D20512 CHANNEL  ; RK_13 U4_U #1移载Y轴轴正软限位
D20513 CHANNEL  ; RK_13 U4_U #1移载Y轴轴为PCU保留
D20514 CHANNEL  ; RK_13 U4_U #1移载Y轴轴为PCU保留
D20515 CHANNEL  ; RK_13 U4_U #1移载Y轴轴初始脉冲定义
D20600 CHANNEL  ; U6- 操作数据区域定义
D20601 CHANNEL  ; U6- 操作数据区域开始字
D20602 CHANNEL  ; U6- 轴参数定义
D20603 CHANNEL  ; U6- 未被使用
D20604 CHANNEL  ; RK_13 U6_X #2移载Y轴轴输入输出设定
D20605 CHANNEL  ; RK_13 U6_X #2移载Y轴轴操作模式选择
D20606 CHANNEL  ; RK_13 U6_X #2移载Y轴轴最高速度
D20607 CHANNEL  ; RK_13 U6_X #2移载Y轴轴最高速度
D20608 CHANNEL  ; RK_13 U6_X #2移载Y轴轴初始速度
D20609 CHANNEL  ; RK_13 U6_X #2移载Y轴轴初始速度
D20610 CHANNEL  ; RK_13 U6_X #2移载Y轴轴原点搜索高速
D20611 CHANNEL  ; RK_13 U6_X #2移载Y轴轴原点搜索高速
D20612 CHANNEL  ; RK_13 U6_X #2移载Y轴轴原点搜索接近速度
D20613 CHANNEL  ; RK_13 U6_X #2移载Y轴轴原点搜索接近速度
D20614 CHANNEL  ; RK_13 U6_X #2移载Y轴轴原点补偿值
D20615 CHANNEL  ; RK_13 U6_X #2移载Y轴轴原点补偿值
D20616 CHANNEL  ; RK_13 U6_X #2移载Y轴轴间隙补偿
D20617 CHANNEL  ; RK_13 U6_X #2移载Y轴轴间隙补偿速度
D20618 CHANNEL  ; RK_13 U6_X #2移载Y轴轴间隙补偿速度
D20619 CHANNEL  ; RK_13 U6_X #2移载Y轴轴加减速曲线
D20620 CHANNEL  ; RK_13 U6_X #2移载Y轴轴原点搜索加速时间
D20621 CHANNEL  ; RK_13 U6_X #2移载Y轴轴原点搜索加速时间
D20622 CHANNEL  ; RK_13 U6_X #2移载Y轴轴原点搜索减速时间
D20623 CHANNEL  ; RK_13 U6_X #2移载Y轴轴原点搜索减速时间
D20624 CHANNEL  ; RK_13 U6_X #2移载Y轴轴定位监测时间
D20625 CHANNEL  ; RK_13 U6_X #2移载Y轴轴负软限位
D20626 CHANNEL  ; RK_13 U6_X #2移载Y轴轴负软限位
D20627 CHANNEL  ; RK_13 U6_X #2移载Y轴轴正软限位
D20628 CHANNEL  ; RK_13 U6_X #2移载Y轴轴正软限位
D20629 CHANNEL  ; RK_13 U6_X #2移载Y轴轴为PCU保留
D20630 CHANNEL  ; RK_13 U6_X #2移载Y轴轴为PCU保留
D20631 CHANNEL  ; RK_13 U6_X #2移载Y轴轴初始脉冲定义
D20632 CHANNEL  ; RK_16 U6_Y 激光焊接X轴轴输入输出设定
D20633 CHANNEL  ; RK_16 U6_Y 激光焊接X轴轴操作模式选择
D20634 CHANNEL  ; RK_16 U6_Y 激光焊接X轴轴最高速度
D20635 CHANNEL  ; RK_16 U6_Y 激光焊接X轴轴最高速度
D20636 CHANNEL  ; RK_16 U6_Y 激光焊接X轴轴初始速度
D20637 CHANNEL  ; RK_16 U6_Y 激光焊接X轴轴初始速度
D20638 CHANNEL  ; RK_16 U6_Y 激光焊接X轴轴原点搜索高速
D20639 CHANNEL  ; RK_16 U6_Y 激光焊接X轴轴原点搜索高速
D20640 CHANNEL  ; RK_16 U6_Y 激光焊接X轴轴原点搜索接近速度
D20641 CHANNEL  ; RK_16 U6_Y 激光焊接X轴轴原点搜索接近速度
D20642 CHANNEL  ; RK_16 U6_Y 激光焊接X轴轴原点补偿值
D20643 CHANNEL  ; RK_16 U6_Y 激光焊接X轴轴原点补偿值
D20644 CHANNEL  ; RK_16 U6_Y 激光焊接X轴轴间隙补偿
D20645 CHANNEL  ; RK_16 U6_Y 激光焊接X轴轴间隙补偿速度
D20646 CHANNEL  ; RK_16 U6_Y 激光焊接X轴轴间隙补偿速度
D20647 CHANNEL  ; RK_16 U6_Y 激光焊接X轴轴加减速曲线
D20648 CHANNEL  ; RK_16 U6_Y 激光焊接X轴轴原点搜索加速时间
D20649 CHANNEL  ; RK_16 U6_Y 激光焊接X轴轴原点搜索加速时间
D20650 CHANNEL  ; RK_16 U6_Y 激光焊接X轴轴原点搜索减速时间
D20651 CHANNEL  ; RK_16 U6_Y 激光焊接X轴轴原点搜索减速时间
D20652 CHANNEL  ; RK_16 U6_Y 激光焊接X轴轴定位监测时间
D20653 CHANNEL  ; RK_16 U6_Y 激光焊接X轴轴负软限位
D20654 CHANNEL  ; RK_16 U6_Y 激光焊接X轴轴负软限位
D20655 CHANNEL  ; RK_16 U6_Y 激光焊接X轴轴正软限位
D20656 CHANNEL  ; RK_16 U6_Y 激光焊接X轴轴正软限位
D20657 CHANNEL  ; RK_16 U6_Y 激光焊接X轴轴为PCU保留
D20658 CHANNEL  ; RK_16 U6_Y 激光焊接X轴轴为PCU保留
D20659 CHANNEL  ; RK_16 U6_Y 激光焊接X轴轴初始脉冲定义
D20660 CHANNEL  ; RK_16 U6_Z 激光焊接Z轴轴输入输出设定
D20661 CHANNEL  ; RK_16 U6_Z 激光焊接Z轴轴操作模式选择
D20662 CHANNEL  ; RK_16 U6_Z 激光焊接Z轴轴最高速度
D20663 CHANNEL  ; RK_16 U6_Z 激光焊接Z轴轴最高速度
D20664 CHANNEL  ; RK_16 U6_Z 激光焊接Z轴轴初始速度
D20665 CHANNEL  ; RK_16 U6_Z 激光焊接Z轴轴初始速度
D20666 CHANNEL  ; RK_16 U6_Z 激光焊接Z轴轴原点搜索高速
D20667 CHANNEL  ; RK_16 U6_Z 激光焊接Z轴轴原点搜索高速
D20668 CHANNEL  ; RK_16 U6_Z 激光焊接Z轴轴原点搜索接近速度
D20669 CHANNEL  ; RK_16 U6_Z 激光焊接Z轴轴原点搜索接近速度
D20670 CHANNEL  ; RK_16 U6_Z 激光焊接Z轴轴原点补偿值
D20671 CHANNEL  ; RK_16 U6_Z 激光焊接Z轴轴原点补偿值
D20672 CHANNEL  ; RK_16 U6_Z 激光焊接Z轴轴间隙补偿
D20673 CHANNEL  ; RK_16 U6_Z 激光焊接Z轴轴间隙补偿速度
D20674 CHANNEL  ; RK_16 U6_Z 激光焊接Z轴轴间隙补偿速度
D20675 CHANNEL  ; RK_16 U6_Z 激光焊接Z轴轴加减速曲线
D20676 CHANNEL  ; RK_16 U6_Z 激光焊接Z轴轴原点搜索加速时间
D20677 CHANNEL  ; RK_16 U6_Z 激光焊接Z轴轴原点搜索加速时间
D20678 CHANNEL  ; RK_16 U6_Z 激光焊接Z轴轴原点搜索减速时间
D20679 CHANNEL  ; RK_16 U6_Z 激光焊接Z轴轴原点搜索减速时间
D20680 CHANNEL  ; RK_16 U6_Z 激光焊接Z轴轴定位监测时间
D20681 CHANNEL  ; RK_16 U6_Z 激光焊接Z轴轴负软限位
D20682 CHANNEL  ; RK_16 U6_Z 激光焊接Z轴轴负软限位
D20683 CHANNEL  ; RK_16 U6_Z 激光焊接Z轴轴正软限位
D20684 CHANNEL  ; RK_16 U6_Z 激光焊接Z轴轴正软限位
D20685 CHANNEL  ; RK_16 U6_Z 激光焊接Z轴轴为PCU保留
D20686 CHANNEL  ; RK_16 U6_Z 激光焊接Z轴轴为PCU保留
D20687 CHANNEL  ; RK_16 U6_Z 激光焊接Z轴轴初始脉冲定义
D20800 CHANNEL  ; U8- 操作数据区域定义
D20801 CHANNEL  ; U8- 操作数据区域开始字
D20802 CHANNEL  ; U8- 轴参数定义
D20803 CHANNEL  ; U8- 未被使用
D20804 CHANNEL  ; RK_06 U8_X 电池上下料X轴轴输入输出设定
D20805 CHANNEL  ; RK_06 U8_X 电池上下料X轴轴操作模式选择
D20806 CHANNEL  ; RK_06 U8_X 电池上下料X轴轴最高速度
D20807 CHANNEL  ; RK_06 U8_X 电池上下料X轴轴最高速度
D20808 CHANNEL  ; RK_06 U8_X 电池上下料X轴轴初始速度
D20809 CHANNEL  ; RK_06 U8_X 电池上下料X轴轴初始速度
D20810 CHANNEL  ; RK_06 U8_X 电池上下料X轴轴原点搜索高速
D20811 CHANNEL  ; RK_06 U8_X 电池上下料X轴轴原点搜索高速
D20812 CHANNEL  ; RK_06 U8_X 电池上下料X轴轴原点搜索接近速度
D20813 CHANNEL  ; RK_06 U8_X 电池上下料X轴轴原点搜索接近速度
D20814 CHANNEL  ; RK_06 U8_X 电池上下料X轴轴原点补偿值
D20815 CHANNEL  ; RK_06 U8_X 电池上下料X轴轴原点补偿值
D20816 CHANNEL  ; RK_06 U8_X 电池上下料X轴轴间隙补偿
D20817 CHANNEL  ; RK_06 U8_X 电池上下料X轴轴间隙补偿速度
D20818 CHANNEL  ; RK_06 U8_X 电池上下料X轴轴间隙补偿速度
D20819 CHANNEL  ; RK_06 U8_X 电池上下料X轴轴加减速曲线
D20820 CHANNEL  ; RK_06 U8_X 电池上下料X轴轴原点搜索加速时间
D20821 CHANNEL  ; RK_06 U8_X 电池上下料X轴轴原点搜索加速时间
D20822 CHANNEL  ; RK_06 U8_X 电池上下料X轴轴原点搜索减速时间
D20823 CHANNEL  ; RK_06 U8_X 电池上下料X轴轴原点搜索减速时间
D20824 CHANNEL  ; RK_06 U8_X 电池上下料X轴轴定位监测时间
D20825 CHANNEL  ; RK_06 U8_X 电池上下料X轴轴负软限位
D20826 CHANNEL  ; RK_06 U8_X 电池上下料X轴轴负软限位
D20827 CHANNEL  ; RK_06 U8_X 电池上下料X轴轴正软限位
D20828 CHANNEL  ; RK_06 U8_X 电池上下料X轴轴正软限位
D20829 CHANNEL  ; RK_06 U8_X 电池上下料X轴轴为PCU保留
D20830 CHANNEL  ; RK_06 U8_X 电池上下料X轴轴为PCU保留
D20831 CHANNEL  ; RK_06 U8_X 电池上下料X轴轴初始脉冲定义
D20832 CHANNEL  ; RK_07 U8_Y 铝壳进料X轴轴输入输出设定
D20833 CHANNEL  ; RK_07 U8_Y 铝壳进料X轴轴操作模式选择
D20834 CHANNEL  ; RK_07 U8_Y 铝壳进料X轴轴最高速度
D20835 CHANNEL  ; RK_07 U8_Y 铝壳进料X轴轴最高速度
D20836 CHANNEL  ; RK_07 U8_Y 铝壳进料X轴轴初始速度
D20837 CHANNEL  ; RK_07 U8_Y 铝壳进料X轴轴初始速度
D20838 CHANNEL  ; RK_07 U8_Y 铝壳进料X轴轴原点搜索高速
D20839 CHANNEL  ; RK_07 U8_Y 铝壳进料X轴轴原点搜索高速
D20840 CHANNEL  ; RK_07 U8_Y 铝壳进料X轴轴原点搜索接近速度
D20841 CHANNEL  ; RK_07 U8_Y 铝壳进料X轴轴原点搜索接近速度
D20842 CHANNEL  ; RK_07 U8_Y 铝壳进料X轴轴原点补偿值
D20843 CHANNEL  ; RK_07 U8_Y 铝壳进料X轴轴原点补偿值
D20844 CHANNEL  ; RK_07 U8_Y 铝壳进料X轴轴间隙补偿
D20845 CHANNEL  ; RK_07 U8_Y 铝壳进料X轴轴间隙补偿速度
D20846 CHANNEL  ; RK_07 U8_Y 铝壳进料X轴轴间隙补偿速度
D20847 CHANNEL  ; RK_07 U8_Y 铝壳进料X轴轴加减速曲线
D20848 CHANNEL  ; RK_07 U8_Y 铝壳进料X轴轴原点搜索加速时间
D20849 CHANNEL  ; RK_07 U8_Y 铝壳进料X轴轴原点搜索加速时间
D20850 CHANNEL  ; RK_07 U8_Y 铝壳进料X轴轴原点搜索减速时间
D20851 CHANNEL  ; RK_07 U8_Y 铝壳进料X轴轴原点搜索减速时间
D20852 CHANNEL  ; RK_07 U8_Y 铝壳进料X轴轴定位监测时间
D20853 CHANNEL  ; RK_07 U8_Y 铝壳进料X轴轴负软限位
D20854 CHANNEL  ; RK_07 U8_Y 铝壳进料X轴轴负软限位
D20855 CHANNEL  ; RK_07 U8_Y 铝壳进料X轴轴正软限位
D20856 CHANNEL  ; RK_07 U8_Y 铝壳进料X轴轴正软限位
D20857 CHANNEL  ; RK_07 U8_Y 铝壳进料X轴轴为PCU保留
D20858 CHANNEL  ; RK_07 U8_Y 铝壳进料X轴轴为PCU保留
D20859 CHANNEL  ; RK_07 U8_Y 铝壳进料X轴轴初始脉冲定义
D20860 CHANNEL  ; RK_07 U8_Z 铝壳上料移载Y轴轴输入输出设定
D20861 CHANNEL  ; RK_07 U8_Z 铝壳上料移载Y轴轴操作模式选择
D20862 CHANNEL  ; RK_07 U8_Z 铝壳上料移载Y轴轴最高速度
D20863 CHANNEL  ; RK_07 U8_Z 铝壳上料移载Y轴轴最高速度
D20864 CHANNEL  ; RK_07 U8_Z 铝壳上料移载Y轴轴初始速度
D20865 CHANNEL  ; RK_07 U8_Z 铝壳上料移载Y轴轴初始速度
D20866 CHANNEL  ; RK_07 U8_Z 铝壳上料移载Y轴轴原点搜索高速
D20867 CHANNEL  ; RK_07 U8_Z 铝壳上料移载Y轴轴原点搜索高速
D20868 CHANNEL  ; RK_07 U8_Z 铝壳上料移载Y轴轴原点搜索接近速度
D20869 CHANNEL  ; RK_07 U8_Z 铝壳上料移载Y轴轴原点搜索接近速度
D20870 CHANNEL  ; RK_07 U8_Z 铝壳上料移载Y轴轴原点补偿值
D20871 CHANNEL  ; RK_07 U8_Z 铝壳上料移载Y轴轴原点补偿值
D20872 CHANNEL  ; RK_07 U8_Z 铝壳上料移载Y轴轴间隙补偿
D20873 CHANNEL  ; RK_07 U8_Z 铝壳上料移载Y轴轴间隙补偿速度
D20874 CHANNEL  ; RK_07 U8_Z 铝壳上料移载Y轴轴间隙补偿速度
D20875 CHANNEL  ; RK_07 U8_Z 铝壳上料移载Y轴轴加减速曲线
D20876 CHANNEL  ; RK_07 U8_Z 铝壳上料移载Y轴轴原点搜索加速时间
D20877 CHANNEL  ; RK_07 U8_Z 铝壳上料移载Y轴轴原点搜索加速时间
D20878 CHANNEL  ; RK_07 U8_Z 铝壳上料移载Y轴轴原点搜索减速时间
D20879 CHANNEL  ; RK_07 U8_Z 铝壳上料移载Y轴轴原点搜索减速时间
D20880 CHANNEL  ; RK_07 U8_Z 铝壳上料移载Y轴轴定位监测时间
D20881 CHANNEL  ; RK_07 U8_Z 铝壳上料移载Y轴轴负软限位
D20882 CHANNEL  ; RK_07 U8_Z 铝壳上料移载Y轴轴负软限位
D20883 CHANNEL  ; RK_07 U8_Z 铝壳上料移载Y轴轴正软限位
D20884 CHANNEL  ; RK_07 U8_Z 铝壳上料移载Y轴轴正软限位
D20885 CHANNEL  ; RK_07 U8_Z 铝壳上料移载Y轴轴为PCU保留
D20886 CHANNEL  ; RK_07 U8_Z 铝壳上料移载Y轴轴为PCU保留
D20887 CHANNEL  ; RK_07 U8_Z 铝壳上料移载Y轴轴初始脉冲定义
D20888 CHANNEL  ; RK_10 U8_U 电池除尘上料X轴轴输入输出设定
D20889 CHANNEL  ; RK_10 U8_U 电池除尘上料X轴轴操作模式选择
D20890 CHANNEL  ; RK_10 U8_U 电池除尘上料X轴轴最高速度
D20891 CHANNEL  ; RK_10 U8_U 电池除尘上料X轴轴最高速度
D20892 CHANNEL  ; RK_10 U8_U 电池除尘上料X轴轴初始速度
D20893 CHANNEL  ; RK_10 U8_U 电池除尘上料X轴轴初始速度
D20894 CHANNEL  ; RK_10 U8_U 电池除尘上料X轴轴原点搜索高速
D20895 CHANNEL  ; RK_10 U8_U 电池除尘上料X轴轴原点搜索高速
D20896 CHANNEL  ; RK_10 U8_U 电池除尘上料X轴轴原点搜索接近速度
D20897 CHANNEL  ; RK_10 U8_U 电池除尘上料X轴轴原点搜索接近速度
D20898 CHANNEL  ; RK_10 U8_U 电池除尘上料X轴轴原点补偿值
D20899 CHANNEL  ; RK_10 U8_U 电池除尘上料X轴轴原点补偿值
D20900 CHANNEL  ; RK_10 U8_U 电池除尘上料X轴轴间隙补偿
D20901 CHANNEL  ; RK_10 U8_U 电池除尘上料X轴轴间隙补偿速度
D20902 CHANNEL  ; RK_10 U8_U 电池除尘上料X轴轴间隙补偿速度
D20903 CHANNEL  ; RK_10 U8_U 电池除尘上料X轴轴加减速曲线
D20904 CHANNEL  ; RK_10 U8_U 电池除尘上料X轴轴原点搜索加速时间
D20905 CHANNEL  ; RK_10 U8_U 电池除尘上料X轴轴原点搜索加速时间
D20906 CHANNEL  ; RK_10 U8_U 电池除尘上料X轴轴原点搜索减速时间
D20907 CHANNEL  ; RK_10 U8_U 电池除尘上料X轴轴原点搜索减速时间
D20908 CHANNEL  ; RK_10 U8_U 电池除尘上料X轴轴定位监测时间
D20909 CHANNEL  ; RK_10 U8_U 电池除尘上料X轴轴负软限位
D20910 CHANNEL  ; RK_10 U8_U 电池除尘上料X轴轴负软限位
D20911 CHANNEL  ; RK_10 U8_U 电池除尘上料X轴轴正软限位
D20912 CHANNEL  ; RK_10 U8_U 电池除尘上料X轴轴正软限位
D20913 CHANNEL  ; RK_10 U8_U 电池除尘上料X轴轴为PCU保留
D20914 CHANNEL  ; RK_10 U8_U 电池除尘上料X轴轴为PCU保留
D20915 CHANNEL  ; RK_10 U8_U 电池除尘上料X轴轴初始脉冲定义
D21 CHANNEL  ; 报警长延时
D2100 CHANNEL  ; Hipot检测仪读测试结果开始字
D2104 CHANNEL  ; Hipot检测仪测试电压
D2105 CHANNEL  ; Hipot检测仪测试电阻（低字）
D2106 CHANNEL  ; Hipot检测仪测试电阻（高字）
D2107 CHANNEL  ; Hipot检测仪测试电流（低字）
D2108 CHANNEL  ; Hipot检测仪测试电流（高字）
D2110 CHANNEL  ; Hipot检测仪读测试结果结束字
D2125 CHANNEL  ; Hipot检测仪测试电阻（Float）
D2127 CHANNEL  ; Hipot检测仪测试电流（Float）
D2130 CHANNEL  ; 倍率1000（Float）
D214 CHANNEL  ; d306
D2140 CHANNEL  ; Hipot检测仪查询结果开始字
D2144 CHANNEL  ; Hipot测试仪查询电压
D2145 CHANNEL  ; Hipot检测仪查询电阻（低字）
D2146 CHANNEL  ; Hipot检测仪查询电阻（高字）
D2147 CHANNEL  ; Hipot检测仪查询电流（低字）
D2148 CHANNEL  ; Hipot检测仪查询电流（高字）
D2149 CHANNEL  ; Hipot检测仪查询结果
D2150 CHANNEL  ; Hipot检测仪查询数据
D2151 CHANNEL  ; Hipot检测仪查询数据
D2152 CHANNEL  ; Hipot检测仪查询数据
D2153 CHANNEL  ; Hipot检测仪查询数据
D2154 CHANNEL  ; Hipot检测仪查询数据
D2159 CHANNEL  ; Hipot检测仪查询结果结束字
D2165 CHANNEL  ; Hipot检测仪查询电阻（Float）
D2167 CHANNEL  ; Hipot检测仪查询电流（Float）
D2170 CHANNEL  ; Hipot检测仪查询结果转换
D2171 CHANNEL  ; Hipot检测仪查询电阻下限高字
D2172 CHANNEL  ; Hipot检测仪查询电阻下限低字
D2173 CHANNEL  ; Hipot检测仪查询电阻上限高字
D2174 CHANNEL  ; Hipot检测仪查询电阻上限低字
D2175 CHANNEL  ; Hipot检测仪查询测试时间
D22 CHANNEL  ; 报警短延时
D2200 CHANNEL  ; RK_15 轮廓检测机构#1移载轮廓测量值上限（Float）
D2202 CHANNEL  ; RK_15 轮廓检测机构#1移载轮廓测量值下限（Float）
D2204 CHANNEL  ; RK_15 轮廓检测机构#1移载轮廓测量值上限设定（Float）
D2206 CHANNEL  ; RK_15 轮廓检测机构#1移载轮廓测量值下限设定（Float）
D2210 CHANNEL  ; RK_15 轮廓检测机构#2移载轮廓测量值上限（Float）
D2212 CHANNEL  ; RK_15 轮廓检测机构#2移载轮廓测量值下限（Float）
D2214 CHANNEL  ; RK_15 轮廓检测机构#2移载轮廓测量值上限设定（Float）
D2216 CHANNEL  ; RK_15 轮廓检测机构#2移载轮廓测量值下限设定（Float）
D23 CHANNEL  ; 伺服到位延时
D2300 CHANNEL  ; RK_15 轮廓检测机构#1移载#1轮廓测量值（Float）
D2302 CHANNEL  ; RK_15 轮廓检测机构#1移载#2轮廓测量值（Float）
D2304 CHANNEL  ; RK_15 轮廓检测机构#1移载#3轮廓测量值（Float）
D2306 CHANNEL  ; RK_15 轮廓检测机构#1移载#4轮廓测量值（Float）
D2307 CHANNEL  ; RK_15 轮廓检测机构#1移载#4轮廓测量值（Float）
D2310 CHANNEL  ; RK_15 轮廓检测机构#2移载#1轮廓测量值（Float）
D2312 CHANNEL  ; RK_15 轮廓检测机构#2移载#2轮廓测量值（Float）
D2314 CHANNEL  ; RK_15 轮廓检测机构#2移载#3轮廓测量值（Float）
D2316 CHANNEL  ; RK_15 轮廓检测机构#2移载#4轮廓测量值（Float）
D2317 CHANNEL  ; RK_15 轮廓检测机构#2移载#4轮廓测量值（Float）
D2320 CHANNEL  ; RK_15 轮廓检测机构#1移载#1轮廓测量值开始字（String）
D2329 CHANNEL  ; RK_15 轮廓检测机构#1移载#1轮廓测量值结束字（String）
D2330 CHANNEL  ; RK_15 轮廓检测机构#1移载#2轮廓测量值开始字（String）
D2339 CHANNEL  ; RK_15 轮廓检测机构#1移载#2轮廓测量值结束字（String）
D2340 CHANNEL  ; RK_15 轮廓检测机构#1移载#3轮廓测量值开始字（String）
D2349 CHANNEL  ; RK_15 轮廓检测机构#1移载#3轮廓测量值结束字（String）
D2350 CHANNEL  ; RK_15 轮廓检测机构#1移载#4轮廓测量值开始字（String）
D2359 CHANNEL  ; RK_15 轮廓检测机构#1移载#4轮廓测量值结束字（String）
D2360 CHANNEL  ; RK_15 轮廓检测机构#2移载#1轮廓测量值开始字（String）
D2369 CHANNEL  ; RK_15 轮廓检测机构#2移载#1轮廓测量值结束字（String）
D2370 CHANNEL  ; RK_15 轮廓检测机构#2移载#2轮廓测量值开始字（String）
D2379 CHANNEL  ; RK_15 轮廓检测机构#2移载#2轮廓测量值结束字（String）
D2380 CHANNEL  ; RK_15 轮廓检测机构#2移载#3轮廓测量值开始字（String）
D2389 CHANNEL  ; RK_15 轮廓检测机构#2移载#3轮廓测量值结束字（String）
D2390 CHANNEL  ; RK_15 轮廓检测机构#2移载#4轮廓测量值开始字（String）
D2399 CHANNEL  ; RK_15 轮廓检测机构#2移载#4轮廓测量值结束字（String）
D24 CHANNEL  ; 伺服启动延时
D25 CHANNEL  ; 轮廓检测机构测量读数据延时设定
D26 CHANNEL  ; 铝壳上下料感应异常提示延时设定
D2603 CHANNEL  ; Hipot检测仪参数组编号
D2604 CHANNEL  ; Hipot检测仪测试电压
D2605 CHANNEL  ; Hipot检测仪测试延时时间
D2606 CHANNEL  ; Hipot检测仪测试时间
D2608 CHANNEL  ; Hipot检测仪电阻下限
D2609 CHANNEL  ; Hipot检测仪电阻上限
D2610 CHANNEL  ; RK_09 Hipot检测机构测试完成放电延时参数设定
D2653 CHANNEL  ; Hipot检测仪参数组编号（HMI）
D2654 CHANNEL  ; Hipot检测仪测试电压（HMI）
D2655 CHANNEL  ; Hipot检测仪测试延时时间（HMI）
D2656 CHANNEL  ; Hipot检测仪测试时间（HMI）
D2658 CHANNEL  ; Hipot检测仪电阻下限（HMI）
D2659 CHANNEL  ; Hipot检测仪电阻上限（HMI）
D2660 CHANNEL  ; RK_09 Hipot检测机构测试完成放电延时设定
D2700 CHANNEL  ; Hipot检测仪参数发送（协议宏）
D2809 CHANNEL  ; Hipot检测仪测试结果
D300 CHANNEL  ; 良品数（DINT）
D302 CHANNEL  ; 不良品数（DINT）
D304 CHANNEL  ; 总计（DINT）
D306 CHANNEL  ; 合格率（Float）
D310 CHANNEL  ; #1出站不良品数（DINT）
D3100 CHANNEL  ; 电芯进料X轴&上料X轴当前总距离
D3102 CHANNEL  ; 电芯进料X轴&上料X轴两原点间距离设定值
D3104 CHANNEL  ; 电芯进料X轴&上料X轴距离计算值
D3106 CHANNEL  ; 电芯进料X轴&上料X轴距离最小安全值
D3108 CHANNEL  ; 电芯进料X轴&上料X轴最小安全距离设定值
D3110 CHANNEL  ; 电芯进料X轴允许去放料位安全设定值（参照电芯上料X轴当前位置）
D3112 CHANNEL  ; 电芯上料X轴允许去取料位安全设定值（参照电芯进料X轴当前位置）
D312 CHANNEL  ; #2出站不良品数（DINT）
D314 CHANNEL  ; 总计（Float）
D316 CHANNEL  ; 良品数（Float）
D3210 CHANNEL  ; 电芯上料X轴允许去取料位安全设定值（参照电芯进料X轴当前位置）
D3300 CHANNEL  ; 电芯除尘吹气延时设定值
D3400 CHANNEL  ; RK_05 入壳压力高报警SV
D350 CHANNEL  ; 电芯进料到入壳工位有电芯统计（BCD）
D351 CHANNEL  ; 电芯进料到入壳工位有电芯统计（BIN）
D360 CHANNEL  ; 铝壳进料到入壳工位有铝壳统计（BCD）
D3600 CHANNEL  ; 铝壳料盘列数设定（X轴）
D3602 CHANNEL  ; 铝壳料盘行数设定（Y轴）
D361 CHANNEL  ; 铝壳进料到入壳工位有铝壳统计（BIN）
D3610 CHANNEL  ; 铝壳料盘列间距设定（X轴）
D3612 CHANNEL  ; 铝壳料盘行间距设定（Y轴）
D3700 CHANNEL  ; 铝壳除尘吹气延时设定值
D3804 CHANNEL  ; #1Hipot检测仪测试电压（Int）
D3805 CHANNEL  ; #1Hipot测试仪测试电阻（Float）
D3806 CHANNEL  ; #1Hipot测试仪测试电阻（Float）
D3807 CHANNEL  ; #1Hipot检测仪测试电流（Float）
D3808 CHANNEL  ; #1Hipot检测仪测试电流（Float）
D3809 CHANNEL  ; #1Hipot检测仪测试结果（Int）
D3854 CHANNEL  ; #2Hipot检测仪测试电压（Int）
D3855 CHANNEL  ; #2Hipot测试仪测试电阻（Float）
D3856 CHANNEL  ; #2Hipot测试仪测试电阻（Float）
D3857 CHANNEL  ; #2Hipot检测仪测试电流（Float）
D3858 CHANNEL  ; #2Hipot检测仪测试电流（Float）
D3859 CHANNEL  ; #2Hipot检测仪测试结果（Int）
D3900 CHANNEL  ; 电池除尘上料X轴&预焊上下料X轴当前总距离
D3902 CHANNEL  ; 电池除尘上料X轴&预焊上下料X轴两原点间距离设定值
D3904 CHANNEL  ; 电池除尘上料X轴&预焊上下料X轴距离计算值
D3906 CHANNEL  ; 电池除尘上料X轴&预焊上下料X轴距离最小安全值
D3908 CHANNEL  ; 电池除尘上料X轴&预焊上下料X轴最小安全距离设定值
D3910 CHANNEL  ; 电池除尘上料X轴允许去电池除尘放料位安全设定值（参照预焊上下料X轴当前位置）
D3912 CHANNEL  ; 预焊上下料X轴允许去电池除尘取料位安全设定值（参照电池除尘上料X轴当前位置）
D4000 CHANNEL  ; 电池除尘吹气延时设定值
D4110 CHANNEL  ; 预焊上下料X轴允许去电池除尘取料位安全设定值（参照电池除尘上料X轴当前位置）
D4400 CHANNEL  ; RK_15 轮廓检测机构程序切换设定
D4410 CHANNEL  ; RK_15 轮廓检测机构程序切换字节数
D4411 CHANNEL  ; RK_15 轮廓检测机构程序切换开始字
D4419 CHANNEL  ; RK_15 轮廓检测机构程序切换结束字
D4420 CHANNEL  ; RK_15 轮廓检测机构轮廓测量字节数
D4421 CHANNEL  ; RK_15 轮廓检测机构轮廓测量结果开始字
D4426 CHANNEL  ; RK_15 轮廓检测机构轮廓测量值开始字
D4439 CHANNEL  ; RK_15 轮廓检测机构轮廓测量结果结束字
D4450 CHANNEL  ; RK_15 轮廓检测机构轮廓测量值开始字（String）
D4460 CHANNEL  ; RK_15 轮廓检测机构轮廓测量值开始字（Float）
D4470 CHANNEL  ; RK_15 轮廓检测机构轮廓测量值开始字（String）
D60 CHANNEL  ; 电芯进料接收条码数据字长度
D64 CHANNEL  ; 设定条码抽取开始位
D65 CHANNEL  ; 条码抽取开始位
D66 CHANNEL  ; 设定条码长度
D68 CHANNEL  ; 电芯进料接收条码字长度
D69 CHANNEL  ; 电芯进料接收条码字长度余数
D70 CHANNEL  ; 设定条码批次号
D71 CHANNEL  ; A设定条码批次号
D72 CHANNEL  ; A设定条码批次号
D73 CHANNEL  ; A设定条码批次号
D74 CHANNEL  ; A设定条码批次号
D75 CHANNEL  ; A设定条码批次号
D76 CHANNEL  ; A设定条码批次号
D77 CHANNEL  ; A设定条码批次号
D78 CHANNEL  ; A设定条码批次号
D79 CHANNEL  ; A设定条码批次号
D80 CHANNEL  ; 电芯进料接收条码长度
D900 CHANNEL  ; RK_05 #1入壳压力PV
D902 CHANNEL  ; RK_05 #1入壳压力补偿值
D910 CHANNEL  ; RK_05 #2入壳压力PV
D912 CHANNEL  ; RK_05 #2入壳压力补偿值
D998 CHANNEL  ; 数据零（Float）
D999 CHANNEL  ; 数据零（Float）
E0_4000 CHANNEL  ; RK_07 U8_Y 铝壳进料X轴取料基准位
E0_4020 CHANNEL  ; RK_07 U8_Z 铝壳上料移载Y轴铝壳取料基准位
E1_0 CHANNEL  ; NC433_0 数据传送写字数
E1_1 CHANNEL  ; NC433_0 数据传送写源区域
E1_10 CHANNEL  ; RK_01 U0_X 电芯来料Y轴轴直接操作速度
E1_100 CHANNEL  ; NC433_2 数据传送写字数
E1_1000 CHANNEL  ; RK_01 U0_X 电芯来料Y轴轴自动速度
E1_1001 CHANNEL  ; RK_01 U0_X 电芯来料Y轴轴自动速度
E1_1002 CHANNEL  ; RK_01 U0_X 电芯来料Y轴轴 Jog 高速
E1_1003 CHANNEL  ; RK_01 U0_X 电芯来料Y轴轴 Jog 高速
E1_1004 CHANNEL  ; RK_01 U0_X 电芯来料Y轴轴 Jog 低速
E1_1005 CHANNEL  ; RK_01 U0_X 电芯来料Y轴轴 Jog 低速
E1_1006 CHANNEL  ; RK_01 U0_X 电芯来料Y轴轴加减速时间
E1_1007 CHANNEL  ; RK_01 U0_X 电芯来料Y轴轴加减速时间
E1_1008 CHANNEL  ; RK_01 U0_X 电芯来料Y轴轴正软极限
E1_1009 CHANNEL  ; RK_01 U0_X 电芯来料Y轴轴正软极限
E1_101 CHANNEL  ; NC433_2 数据传送写源区域
E1_1010 CHANNEL  ; RK_01 U0_X 电芯来料Y轴轴负软极限
E1_1011 CHANNEL  ; RK_01 U0_X 电芯来料Y轴轴负软极限
E1_1012 CHANNEL  ; RK_01 U0_X 电芯来料Y轴轴原点偏移
E1_102 CHANNEL  ; NC433_2 数据传送定源字
E1_1020 CHANNEL  ; RK_01 U0_X 电芯来料Y轴待料位
E1_1021 CHANNEL  ; RK_01 U0_X 电芯来料Y轴待料位
E1_1022 CHANNEL  ; RK_01 U0_X 电芯来料Y轴上料位
E1_1023 CHANNEL  ; RK_01 U0_X 电芯来料Y轴上料位
E1_1024 CHANNEL  ; RK_01 U0_X 电芯来料Y轴扫码位
E1_1025 CHANNEL  ; RK_01 U0_X 电芯来料Y轴扫码位
E1_1026 CHANNEL  ; RK_01 U0_X 电芯来料Y轴下料位
E1_1027 CHANNEL  ; RK_01 U0_X 电芯来料Y轴下料位
E1_1028 CHANNEL  ; RK_01 U0_X 电芯来料Y轴轴5#位置
E1_1029 CHANNEL  ; RK_01 U0_X 电芯来料Y轴轴5#位置
E1_103 CHANNEL  ; NC433_2 数据传送定目标地址
E1_1030 CHANNEL  ; RK_01 U0_X 电芯来料Y轴轴6#位置
E1_1031 CHANNEL  ; RK_01 U0_X 电芯来料Y轴轴6#位置
E1_1032 CHANNEL  ; RK_01 U0_X 电芯来料Y轴轴7#位置
E1_1033 CHANNEL  ; RK_01 U0_X 电芯来料Y轴轴7#位置
E1_1034 CHANNEL  ; RK_01 U0_X 电芯来料Y轴轴8#位置
E1_1035 CHANNEL  ; RK_01 U0_X 电芯来料Y轴轴8#位置
E1_1036 CHANNEL  ; RK_01 U0_X 电芯来料Y轴轴9#位置
E1_1037 CHANNEL  ; RK_01 U0_X 电芯来料Y轴轴9#位置
E1_1038 CHANNEL  ; RK_01 U0_X 电芯来料Y轴轴10#位置
E1_1039 CHANNEL  ; RK_01 U0_X 电芯来料Y轴轴10#位置
E1_104 CHANNEL  ; NC433_2 数据传送读字数
E1_105 CHANNEL  ; NC433_2 数据传送读源区域
E1_106 CHANNEL  ; NC433_2 数据传送读目标区域
E1_107 CHANNEL  ; NC433_2 数据传送读目标字
E1_108 CHANNEL  ; RK_05 U2_X #1入壳Y轴轴直接操作位置
E1_109 CHANNEL  ; RK_05 U2_X #1入壳Y轴轴直接操作位置
E1_11 CHANNEL  ; RK_01 U0_X 电芯来料Y轴轴直接操作速度
E1_110 CHANNEL  ; RK_05 U2_X #1入壳Y轴轴直接操作速度
E1_1100 CHANNEL  ; RK_02 U0_Y 电芯进料X轴轴自动速度
E1_11000 CHANNEL  ; #4配方参数（伺服轴）
E1_1101 CHANNEL  ; RK_02 U0_Y 电芯进料X轴轴自动速度
E1_1102 CHANNEL  ; RK_02 U0_Y 电芯进料X轴轴 Jog 高速
E1_1103 CHANNEL  ; RK_02 U0_Y 电芯进料X轴轴 Jog 高速
E1_1104 CHANNEL  ; RK_02 U0_Y 电芯进料X轴轴 Jog 低速
E1_1105 CHANNEL  ; RK_02 U0_Y 电芯进料X轴轴 Jog 低速
E1_1106 CHANNEL  ; RK_02 U0_Y 电芯进料X轴轴加减速时间
E1_1107 CHANNEL  ; RK_02 U0_Y 电芯进料X轴轴加减速时间
E1_1108 CHANNEL  ; RK_02 U0_Y 电芯进料X轴轴正软极限
E1_1109 CHANNEL  ; RK_02 U0_Y 电芯进料X轴轴正软极限
E1_111 CHANNEL  ; RK_05 U2_X #1入壳Y轴轴直接操作速度
E1_1110 CHANNEL  ; RK_02 U0_Y 电芯进料X轴轴负软极限
E1_1111 CHANNEL  ; RK_02 U0_Y 电芯进料X轴轴负软极限
E1_1112 CHANNEL  ; RK_02 U0_Y 电芯进料X轴轴原点偏移
E1_112 CHANNEL  ; RK_05 U2_X #1入壳Y轴轴直接操作加速时间
E1_1120 CHANNEL  ; RK_02 U0_Y 电芯进料X轴待料位
E1_1121 CHANNEL  ; RK_02 U0_Y 电芯进料X轴待料位
E1_1122 CHANNEL  ; RK_02 U0_Y 电芯进料X轴取料位
E1_1123 CHANNEL  ; RK_02 U0_Y 电芯进料X轴取料位
E1_1124 CHANNEL  ; RK_02 U0_Y 电芯进料X轴扫码OK放料位
E1_1125 CHANNEL  ; RK_02 U0_Y 电芯进料X轴扫码OK放料位
E1_1126 CHANNEL  ; RK_02 U0_Y 电芯进料X轴扫码NG放料位
E1_1127 CHANNEL  ; RK_02 U0_Y 电芯进料X轴扫码NG放料位
E1_1128 CHANNEL  ; RK_02 U0_Y 电芯进料X轴轴5#位置
E1_1129 CHANNEL  ; RK_02 U0_Y 电芯进料X轴轴5#位置
E1_113 CHANNEL  ; RK_05 U2_X #1入壳Y轴X轴直接操作加速时间
E1_1130 CHANNEL  ; RK_02 U0_Y 电芯进料X轴轴6#位置
E1_1131 CHANNEL  ; RK_02 U0_Y 电芯进料X轴轴6#位置
E1_1132 CHANNEL  ; RK_02 U0_Y 电芯进料X轴轴7#位置
E1_1133 CHANNEL  ; RK_02 U0_Y 电芯进料X轴轴7#位置
E1_1134 CHANNEL  ; RK_02 U0_Y 电芯进料X轴轴8#位置
E1_1135 CHANNEL  ; RK_02 U0_Y 电芯进料X轴轴8#位置
E1_1136 CHANNEL  ; RK_02 U0_Y 电芯进料X轴轴9#位置
E1_1137 CHANNEL  ; RK_02 U0_Y 电芯进料X轴轴9#位置
E1_1138 CHANNEL  ; RK_02 U0_Y 电芯进料X轴轴10#位置
E1_1139 CHANNEL  ; RK_02 U0_Y 电芯进料X轴轴10#位置
E1_114 CHANNEL  ; RK_05 U2_X #1入壳Y轴轴直接操作减速时间
E1_115 CHANNEL  ; RK_05 U2_X #1入壳Y轴轴直接操作减速时间
E1_116 CHANNEL  ; RK_05 U2_X #1入壳Y轴轴存储器操作序列号
E1_117 CHANNEL  ; RK_05 U2_X #1入壳Y轴轴特殊操作Override
E1_118 CHANNEL  ; RK_05 U2_X #1入壳Y轴轴特殊操作示教地址
E1_119 CHANNEL  ; RK_05 U2_X #1入壳Y轴轴特殊操作预留
E1_12 CHANNEL  ; RK_01 U0_X 电芯来料Y轴轴直接操作加速时间
E1_120 CHANNEL  ; RK_05 U2_Y #2入壳Y轴轴直接操作位置
E1_1200 CHANNEL  ; RK_02 U0_Z 电芯进料Z轴轴自动速度
E1_1201 CHANNEL  ; RK_02 U0_Z 电芯进料Z轴轴自动速度
E1_1202 CHANNEL  ; RK_02 U0_Z 电芯进料Z轴轴 Jog 高速
E1_1203 CHANNEL  ; RK_02 U0_Z 电芯进料Z轴轴 Jog 高速
E1_1204 CHANNEL  ; RK_02 U0_Z 电芯进料Z轴轴 Jog 低速
E1_1205 CHANNEL  ; RK_02 U0_Z 电芯进料Z轴轴 Jog 低速
E1_1206 CHANNEL  ; RK_02 U0_Z 电芯进料Z轴轴加减速时间
E1_1207 CHANNEL  ; RK_02 U0_Z 电芯进料Z轴轴加减速时间
E1_1208 CHANNEL  ; RK_02 U0_Z 电芯进料Z轴轴正软极限
E1_1209 CHANNEL  ; RK_02 U0_Z 电芯进料Z轴轴正软极限
E1_121 CHANNEL  ; RK_05 U2_Y #2入壳Y轴轴直接操作位置
E1_1210 CHANNEL  ; RK_02 U0_Z 电芯进料Z轴轴负软极限
E1_1211 CHANNEL  ; RK_02 U0_Z 电芯进料Z轴轴负软极限
E1_1212 CHANNEL  ; RK_02 U0_Z 电芯进料Z轴轴原点偏移
E1_122 CHANNEL  ; RK_05 U2_Y #2入壳Y轴轴直接操作速度
E1_1220 CHANNEL  ; RK_02 U0_Z 电芯进料Z轴待料位（扫码）
E1_1221 CHANNEL  ; RK_02 U0_Z 电芯进料Z轴待料位（扫码）
E1_1222 CHANNEL  ; RK_02 U0_Z 电芯进料Z轴取料位
E1_1223 CHANNEL  ; RK_02 U0_Z 电芯进料Z轴取料位
E1_1224 CHANNEL  ; RK_02 U0_Z 电芯进料Z轴扫码OK放料位
E1_1225 CHANNEL  ; RK_02 U0_Z 电芯进料Z轴扫码OK放料位
E1_1226 CHANNEL  ; RK_02 U0_Z 电芯进料Z轴扫码NG放料位
E1_1227 CHANNEL  ; RK_02 U0_Z 电芯进料Z轴扫码NG放料位
E1_1228 CHANNEL  ; RK_02 U0_Z 电芯进料Z轴扫码位
E1_1229 CHANNEL  ; RK_02 U0_Z 电芯进料Z轴扫码位
E1_123 CHANNEL  ; RK_05 U2_Y #2入壳Y轴轴直接操作速度
E1_1230 CHANNEL  ; RK_02 U0_Z 电芯进料Z轴轴6#位置
E1_1231 CHANNEL  ; RK_02 U0_Z 电芯进料Z轴轴6#位置
E1_1232 CHANNEL  ; RK_02 U0_Z 电芯进料Z轴轴7#位置
E1_1233 CHANNEL  ; RK_02 U0_Z 电芯进料Z轴轴7#位置
E1_1234 CHANNEL  ; RK_02 U0_Z 电芯进料Z轴轴8#位置
E1_1235 CHANNEL  ; RK_02 U0_Z 电芯进料Z轴轴8#位置
E1_1236 CHANNEL  ; RK_02 U0_Z 电芯进料Z轴轴9#位置
E1_1237 CHANNEL  ; RK_02 U0_Z 电芯进料Z轴轴9#位置
E1_1238 CHANNEL  ; RK_02 U0_Z 电芯进料Z轴轴10#位置
E1_1239 CHANNEL  ; RK_02 U0_Z 电芯进料Z轴轴10#位置
E1_124 CHANNEL  ; RK_05 U2_Y #2入壳Y轴轴直接操作加速时间
E1_125 CHANNEL  ; RK_05 U2_Y #2入壳Y轴轴直接操作加速时间
E1_126 CHANNEL  ; RK_05 U2_Y #2入壳Y轴轴直接操作减速时间
E1_127 CHANNEL  ; RK_05 U2_Y #2入壳Y轴轴直接操作减速时间
E1_128 CHANNEL  ; RK_05 U2_Y #2入壳Y轴轴存储器操作序列号
E1_129 CHANNEL  ; RK_05 U2_Y #2入壳Y轴轴特殊操作Override
E1_13 CHANNEL  ; RK_01 U0_X 电芯来料Y轴X轴直接操作加速时间
E1_130 CHANNEL  ; RK_05 U2_Y #2入壳Y轴轴特殊操作示教地址
E1_1300 CHANNEL  ; RK_03 U0_U 电芯上料X轴轴自动速度
E1_13000 CHANNEL  ; #5配方参数（伺服轴）
E1_1301 CHANNEL  ; RK_03 U0_U 电芯上料X轴轴自动速度
E1_1302 CHANNEL  ; RK_03 U0_U 电芯上料X轴轴 Jog 高速
E1_1303 CHANNEL  ; RK_03 U0_U 电芯上料X轴轴 Jog 高速
E1_1304 CHANNEL  ; RK_03 U0_U 电芯上料X轴轴 Jog 低速
E1_1305 CHANNEL  ; RK_03 U0_U 电芯上料X轴轴 Jog 低速
E1_1306 CHANNEL  ; RK_03 U0_U 电芯上料X轴轴加减速时间
E1_1307 CHANNEL  ; RK_03 U0_U 电芯上料X轴轴加减速时间
E1_1308 CHANNEL  ; RK_03 U0_U 电芯上料X轴轴正软极限
E1_1309 CHANNEL  ; RK_03 U0_U 电芯上料X轴轴正软极限
E1_131 CHANNEL  ; RK_05 U2_Y #2入壳Y轴轴特殊操作预留
E1_1310 CHANNEL  ; RK_03 U0_U 电芯上料X轴轴负软极限
E1_1311 CHANNEL  ; RK_03 U0_U 电芯上料X轴轴负软极限
E1_1312 CHANNEL  ; RK_03 U0_U 电芯上料X轴轴原点偏移
E1_1320 CHANNEL  ; RK_03 U0_U 电芯上料X轴待料位
E1_1321 CHANNEL  ; RK_03 U0_U 电芯上料X轴待料位
E1_1322 CHANNEL  ; RK_03 U0_U 电芯上料X轴取料位
E1_1323 CHANNEL  ; RK_03 U0_U 电芯上料X轴取料位
E1_1324 CHANNEL  ; RK_03 U0_U 电芯上料X轴#1入壳放料位
E1_1325 CHANNEL  ; RK_03 U0_U 电芯上料X轴#1入壳放料位
E1_1326 CHANNEL  ; RK_03 U0_U 电芯上料X轴#2入壳放料位
E1_1327 CHANNEL  ; RK_03 U0_U 电芯上料X轴#2入壳放料位
E1_1328 CHANNEL  ; RK_03 U0_U 电芯上料X轴轴5#位置
E1_1329 CHANNEL  ; RK_03 U0_U 电芯上料X轴轴5#位置
E1_1330 CHANNEL  ; RK_03 U0_U 电芯上料X轴轴6#位置
E1_1331 CHANNEL  ; RK_03 U0_U 电芯上料X轴轴6#位置
E1_1332 CHANNEL  ; RK_03 U0_U 电芯上料X轴轴7#位置
E1_1333 CHANNEL  ; RK_03 U0_U 电芯上料X轴轴7#位置
E1_1334 CHANNEL  ; RK_03 U0_U 电芯上料X轴轴8#位置
E1_1335 CHANNEL  ; RK_03 U0_U 电芯上料X轴轴8#位置
E1_1336 CHANNEL  ; RK_03 U0_U 电芯上料X轴轴9#位置
E1_1337 CHANNEL  ; RK_03 U0_U 电芯上料X轴轴9#位置
E1_1338 CHANNEL  ; RK_03 U0_U 电芯上料X轴轴10#位置
E1_1339 CHANNEL  ; RK_03 U0_U 电芯上料X轴轴10#位置
E1_14 CHANNEL  ; RK_01 U0_X 电芯来料Y轴轴直接操作减速时间
E1_1400 CHANNEL  ; RK_05 U2_X #1入壳Y轴轴自动速度
E1_1401 CHANNEL  ; RK_05 U2_X #1入壳Y轴轴自动速度
E1_1402 CHANNEL  ; RK_05 U2_X #1入壳Y轴轴 Jog 高速
E1_1403 CHANNEL  ; RK_05 U2_X #1入壳Y轴轴 Jog 高速
E1_1404 CHANNEL  ; RK_05 U2_X #1入壳Y轴轴 Jog 低速
E1_1405 CHANNEL  ; RK_05 U2_X #1入壳Y轴轴 Jog 低速
E1_1406 CHANNEL  ; RK_05 U2_X #1入壳Y轴轴加减速时间
E1_1407 CHANNEL  ; RK_05 U2_X #1入壳Y轴轴加减速时间
E1_1408 CHANNEL  ; RK_05 U2_X #1入壳Y轴轴正软极限
E1_1409 CHANNEL  ; RK_05 U2_X #1入壳Y轴轴正软极限
E1_1410 CHANNEL  ; RK_05 U2_X #1入壳Y轴轴负软极限
E1_1411 CHANNEL  ; RK_05 U2_X #1入壳Y轴轴负软极限
E1_1412 CHANNEL  ; RK_05 U2_X #1入壳Y轴轴原点偏移
E1_1420 CHANNEL  ; RK_05 U2_X #1入壳Y轴待料位
E1_1421 CHANNEL  ; RK_05 U2_X #1入壳Y轴待料位
E1_1422 CHANNEL  ; RK_05 U2_X #1入壳Y轴滚轮压紧位
E1_1423 CHANNEL  ; RK_05 U2_X #1入壳Y轴滚轮压紧位
E1_1424 CHANNEL  ; RK_05 U2_X #1入壳Y轴滚轮松开位
E1_1425 CHANNEL  ; RK_05 U2_X #1入壳Y轴滚轮松开位
E1_1426 CHANNEL  ; RK_05 U2_X #1入壳Y轴入壳位
E1_1427 CHANNEL  ; RK_05 U2_X #1入壳Y轴入壳位
E1_1428 CHANNEL  ; RK_05 U2_X #1入壳Y轴电芯定位夹爪松开位
E1_1429 CHANNEL  ; RK_05 U2_X #1入壳Y轴电芯定位夹爪松开位
E1_1430 CHANNEL  ; RK_05 U2_X #1入壳Y轴轴6#位置
E1_1431 CHANNEL  ; RK_05 U2_X #1入壳Y轴轴6#位置
E1_1432 CHANNEL  ; RK_05 U2_X #1入壳Y轴轴7#位置
E1_1433 CHANNEL  ; RK_05 U2_X #1入壳Y轴轴7#位置
E1_1434 CHANNEL  ; RK_05 U2_X #1入壳Y轴轴8#位置
E1_1435 CHANNEL  ; RK_05 U2_X #1入壳Y轴轴8#位置
E1_1436 CHANNEL  ; RK_05 U2_X #1入壳Y轴轴9#位置
E1_1437 CHANNEL  ; RK_05 U2_X #1入壳Y轴轴9#位置
E1_1438 CHANNEL  ; RK_05 U2_X #1入壳Y轴轴10#位置
E1_1439 CHANNEL  ; RK_05 U2_X #1入壳Y轴轴10#位置
E1_15 CHANNEL  ; RK_01 U0_X 电芯来料Y轴轴直接操作减速时间
E1_1500 CHANNEL  ; RK_05 U2_Y #2入壳Y轴轴自动速度
E1_15000 CHANNEL  ; #6配方参数（伺服轴）
E1_1501 CHANNEL  ; RK_05 U2_Y #2入壳Y轴轴自动速度
E1_1502 CHANNEL  ; RK_05 U2_Y #2入壳Y轴轴 Jog 高速
E1_1503 CHANNEL  ; RK_05 U2_Y #2入壳Y轴轴 Jog 高速
E1_1504 CHANNEL  ; RK_05 U2_Y #2入壳Y轴轴 Jog 低速
E1_1505 CHANNEL  ; RK_05 U2_Y #2入壳Y轴轴 Jog 低速
E1_1506 CHANNEL  ; RK_05 U2_Y #2入壳Y轴轴加减速时间
E1_1507 CHANNEL  ; RK_05 U2_Y #2入壳Y轴轴加减速时间
E1_1508 CHANNEL  ; RK_05 U2_Y #2入壳Y轴轴正软极限
E1_1509 CHANNEL  ; RK_05 U2_Y #2入壳Y轴轴正软极限
E1_1510 CHANNEL  ; RK_05 U2_Y #2入壳Y轴轴负软极限
E1_1511 CHANNEL  ; RK_05 U2_Y #2入壳Y轴轴负软极限
E1_1512 CHANNEL  ; RK_05 U2_Y #2入壳Y轴轴原点偏移
E1_1520 CHANNEL  ; RK_05 U2_Y #2入壳Y轴待料位
E1_1521 CHANNEL  ; RK_05 U2_Y #2入壳Y轴待料位
E1_1522 CHANNEL  ; RK_05 U2_Y #2入壳Y轴滚轮压紧位
E1_1523 CHANNEL  ; RK_05 U2_Y #2入壳Y轴滚轮压紧位
E1_1524 CHANNEL  ; RK_05 U2_Y #2入壳Y轴滚轮松开位
E1_1525 CHANNEL  ; RK_05 U2_Y #2入壳Y轴滚轮松开位
E1_1526 CHANNEL  ; RK_05 U2_Y #2入壳Y轴入壳位
E1_1527 CHANNEL  ; RK_05 U2_Y #2入壳Y轴入壳位
E1_1528 CHANNEL  ; RK_05 U2_Y #2入壳Y轴电芯定位夹爪松开位
E1_1529 CHANNEL  ; RK_05 U2_Y #2入壳Y轴电芯定位夹爪松开位
E1_1530 CHANNEL  ; RK_05 U2_Y #2入壳Y轴轴6#位置
E1_1531 CHANNEL  ; RK_05 U2_Y #2入壳Y轴轴6#位置
E1_1532 CHANNEL  ; RK_05 U2_Y #2入壳Y轴轴7#位置
E1_1533 CHANNEL  ; RK_05 U2_Y #2入壳Y轴轴7#位置
E1_1534 CHANNEL  ; RK_05 U2_Y #2入壳Y轴轴8#位置
E1_1535 CHANNEL  ; RK_05 U2_Y #2入壳Y轴轴8#位置
E1_1536 CHANNEL  ; RK_05 U2_Y #2入壳Y轴轴9#位置
E1_1537 CHANNEL  ; RK_05 U2_Y #2入壳Y轴轴9#位置
E1_1538 CHANNEL  ; RK_05 U2_Y #2入壳Y轴轴10#位置
E1_1539 CHANNEL  ; RK_05 U2_Y #2入壳Y轴轴10#位置
E1_156 CHANNEL  ; RK_05 U2_X #1入壳Y轴轴当前位置
E1_157 CHANNEL  ; RK_05 U2_X #1入壳Y轴轴当前位置
E1_158 CHANNEL  ; RK_05 U2_X #1入壳Y轴轴存储器操作正被执行序列号
E1_159 CHANNEL  ; RK_05 U2_X #1入壳Y轴轴存储器操作正被执行序列号
E1_16 CHANNEL  ; RK_01 U0_X 电芯来料Y轴轴存储器操作序列号
E1_160 CHANNEL  ; RK_05 U2_Y #2入壳Y轴轴当前位置
E1_161 CHANNEL  ; RK_05 U2_Y #2入壳Y轴轴当前位置
E1_162 CHANNEL  ; RK_05 U2_Y #2入壳Y轴轴存储器操作正被执行序列号
E1_163 CHANNEL  ; RK_05 U2_Y #2入壳Y轴轴存储器操作正被执行序列号
E1_17 CHANNEL  ; RK_01 U0_X 电芯来料Y轴轴特殊操作Override
E1_17000 CHANNEL  ; #7配方参数（伺服轴）
E1_18 CHANNEL  ; RK_01 U0_X 电芯来料Y轴轴特殊操作示教地址
E1_1800 CHANNEL  ; RK_12 U4_X 预焊上下料X轴轴自动速度
E1_1801 CHANNEL  ; RK_12 U4_X 预焊上下料X轴轴自动速度
E1_1802 CHANNEL  ; RK_12 U4_X 预焊上下料X轴轴 Jog 高速
E1_1803 CHANNEL  ; RK_12 U4_X 预焊上下料X轴轴 Jog 高速
E1_1804 CHANNEL  ; RK_12 U4_X 预焊上下料X轴轴 Jog 低速
E1_1805 CHANNEL  ; RK_12 U4_X 预焊上下料X轴轴 Jog 低速
E1_1806 CHANNEL  ; RK_12 U4_X 预焊上下料X轴轴加减速时间
E1_1807 CHANNEL  ; RK_12 U4_X 预焊上下料X轴轴加减速时间
E1_1808 CHANNEL  ; RK_12 U4_X 预焊上下料X轴轴正软极限
E1_1809 CHANNEL  ; RK_12 U4_X 预焊上下料X轴轴正软极限
E1_1810 CHANNEL  ; RK_12 U4_X 预焊上下料X轴轴负软极限
E1_1811 CHANNEL  ; RK_12 U4_X 预焊上下料X轴轴负软极限
E1_1812 CHANNEL  ; RK_12 U4_X 预焊上下料X轴轴原点偏移
E1_1820 CHANNEL  ; RK_12 U4_X 预焊上下料X轴待料位
E1_1821 CHANNEL  ; RK_12 U4_X 预焊上下料X轴待料位
E1_1822 CHANNEL  ; RK_12 U4_X 预焊上下料X轴除尘取料位
E1_1823 CHANNEL  ; RK_12 U4_X 预焊上下料X轴除尘取料位
E1_1824 CHANNEL  ; RK_12 U4_X 预焊上下料X轴#1移载放料位
E1_1825 CHANNEL  ; RK_12 U4_X 预焊上下料X轴#1移载放料位
E1_1826 CHANNEL  ; RK_12 U4_X 预焊上下料X轴#2移载放料位
E1_1827 CHANNEL  ; RK_12 U4_X 预焊上下料X轴#2移载放料位
E1_1828 CHANNEL  ; RK_12 U4_X 预焊上下料X轴#1移载取料位
E1_1829 CHANNEL  ; RK_12 U4_X 预焊上下料X轴#1移载取料位
E1_1830 CHANNEL  ; RK_12 U4_X 预焊上下料X轴#2移载取料位
E1_1831 CHANNEL  ; RK_12 U4_X 预焊上下料X轴#2移载取料位
E1_1832 CHANNEL  ; RK_12 U4_X 预焊上下料X轴OK放料位
E1_1833 CHANNEL  ; RK_12 U4_X 预焊上下料X轴OK放料位
E1_1834 CHANNEL  ; RK_12 U4_X 预焊上下料X轴#1NG放料位
E1_1835 CHANNEL  ; RK_12 U4_X 预焊上下料X轴#1NG放料位
E1_1836 CHANNEL  ; RK_12 U4_X 预焊上下料X轴#2NG放料位
E1_1837 CHANNEL  ; RK_12 U4_X 预焊上下料X轴#2NG放料位
E1_1838 CHANNEL  ; RK_12 U4_X 预焊上下料X轴轴10#位置
E1_1839 CHANNEL  ; RK_12 U4_X 预焊上下料X轴轴10#位置
E1_19 CHANNEL  ; RK_01 U0_X 电芯来料Y轴轴特殊操作预留
E1_1900 CHANNEL  ; RK_12 U4_Y 预焊上料Z轴轴自动速度
E1_19000 CHANNEL  ; #8配方参数（伺服轴）
E1_1901 CHANNEL  ; RK_12 U4_Y 预焊上料Z轴轴自动速度
E1_1902 CHANNEL  ; RK_12 U4_Y 预焊上料Z轴轴 Jog 高速
E1_1903 CHANNEL  ; RK_12 U4_Y 预焊上料Z轴轴 Jog 高速
E1_1904 CHANNEL  ; RK_12 U4_Y 预焊上料Z轴轴 Jog 低速
E1_1905 CHANNEL  ; RK_12 U4_Y 预焊上料Z轴轴 Jog 低速
E1_1906 CHANNEL  ; RK_12 U4_Y 预焊上料Z轴轴加减速时间
E1_1907 CHANNEL  ; RK_12 U4_Y 预焊上料Z轴轴加减速时间
E1_1908 CHANNEL  ; RK_12 U4_Y 预焊上料Z轴轴正软极限
E1_1909 CHANNEL  ; RK_12 U4_Y 预焊上料Z轴轴正软极限
E1_1910 CHANNEL  ; RK_12 U4_Y 预焊上料Z轴轴负软极限
E1_1911 CHANNEL  ; RK_12 U4_Y 预焊上料Z轴轴负软极限
E1_1912 CHANNEL  ; RK_12 U4_Y 预焊上料Z轴轴原点偏移
E1_1920 CHANNEL  ; RK_12 U4_Y 预焊上料Z轴待料位
E1_1921 CHANNEL  ; RK_12 U4_Y 预焊上料Z轴待料位
E1_1922 CHANNEL  ; RK_12 U4_Y 预焊上料Z轴除尘取料位
E1_1923 CHANNEL  ; RK_12 U4_Y 预焊上料Z轴除尘取料位
E1_1924 CHANNEL  ; RK_12 U4_Y 预焊上料Z轴#1移载放料位
E1_1925 CHANNEL  ; RK_12 U4_Y 预焊上料Z轴#1移载放料位
E1_1926 CHANNEL  ; RK_12 U4_Y 预焊上料Z轴#2移载放料位
E1_1927 CHANNEL  ; RK_12 U4_Y 预焊上料Z轴#2移载放料位
E1_1928 CHANNEL  ; RK_12 U4_Y 预焊上料Z轴轴5#位置
E1_1929 CHANNEL  ; RK_12 U4_Y 预焊上料Z轴轴5#位置
E1_1930 CHANNEL  ; RK_12 U4_Y 预焊上料Z轴轴6#位置
E1_1931 CHANNEL  ; RK_12 U4_Y 预焊上料Z轴轴6#位置
E1_1932 CHANNEL  ; RK_12 U4_Y 预焊上料Z轴轴7#位置
E1_1933 CHANNEL  ; RK_12 U4_Y 预焊上料Z轴轴7#位置
E1_1934 CHANNEL  ; RK_12 U4_Y 预焊上料Z轴轴8#位置
E1_1935 CHANNEL  ; RK_12 U4_Y 预焊上料Z轴轴8#位置
E1_1936 CHANNEL  ; RK_12 U4_Y 预焊上料Z轴轴9#位置
E1_1937 CHANNEL  ; RK_12 U4_Y 预焊上料Z轴轴9#位置
E1_1938 CHANNEL  ; RK_12 U4_Y 预焊上料Z轴轴10#位置
E1_1939 CHANNEL  ; RK_12 U4_Y 预焊上料Z轴轴10#位置
E1_2 CHANNEL  ; NC433_0 数据传送定源字
E1_20 CHANNEL  ; RK_02 U0_Y 电芯进料X轴轴直接操作位置
E1_200 CHANNEL  ; NC433_4 数据传送写字数
E1_2000 CHANNEL  ; RK_12 U4_Z 预焊下料Z轴轴自动速度
E1_2001 CHANNEL  ; RK_12 U4_Z 预焊下料Z轴轴自动速度
E1_2002 CHANNEL  ; RK_12 U4_Z 预焊下料Z轴轴 Jog 高速
E1_2003 CHANNEL  ; RK_12 U4_Z 预焊下料Z轴轴 Jog 高速
E1_2004 CHANNEL  ; RK_12 U4_Z 预焊下料Z轴轴 Jog 低速
E1_2005 CHANNEL  ; RK_12 U4_Z 预焊下料Z轴轴 Jog 低速
E1_2006 CHANNEL  ; RK_12 U4_Z 预焊下料Z轴轴加减速时间
E1_2007 CHANNEL  ; RK_12 U4_Z 预焊下料Z轴轴加减速时间
E1_2008 CHANNEL  ; RK_12 U4_Z 预焊下料Z轴轴正软极限
E1_2009 CHANNEL  ; RK_12 U4_Z 预焊下料Z轴轴正软极限
E1_201 CHANNEL  ; NC433_4 数据传送写源区域
E1_2010 CHANNEL  ; RK_12 U4_Z 预焊下料Z轴轴负软极限
E1_2011 CHANNEL  ; RK_12 U4_Z 预焊下料Z轴轴负软极限
E1_2012 CHANNEL  ; RK_12 U4_Z 预焊下料Z轴轴原点偏移
E1_202 CHANNEL  ; NC433_4 数据传送定源字
E1_2020 CHANNEL  ; RK_12 U4_Z 预焊下料Z轴待料位
E1_2021 CHANNEL  ; RK_12 U4_Z 预焊下料Z轴待料位
E1_2022 CHANNEL  ; RK_12 U4_Z 预焊下料Z轴#1移载取料位
E1_2023 CHANNEL  ; RK_12 U4_Z 预焊下料Z轴#1移载取料位
E1_2024 CHANNEL  ; RK_12 U4_Z 预焊下料Z轴#2移载取料位
E1_2025 CHANNEL  ; RK_12 U4_Z 预焊下料Z轴#2移载取料位
E1_2026 CHANNEL  ; RK_12 U4_Z 预焊下料Z轴OK放料位
E1_2027 CHANNEL  ; RK_12 U4_Z 预焊下料Z轴OK放料位
E1_2028 CHANNEL  ; RK_12 U4_Z 预焊下料Z轴#1NG放料位
E1_2029 CHANNEL  ; RK_12 U4_Z 预焊下料Z轴#1NG放料位
E1_203 CHANNEL  ; NC433_4 数据传送定目标地址
E1_2030 CHANNEL  ; RK_12 U4_Z 预焊下料Z轴#2NG放料位
E1_2031 CHANNEL  ; RK_12 U4_Z 预焊下料Z轴#2NG放料位
E1_2032 CHANNEL  ; RK_12 U4_Z 预焊下料Z轴轴7#位置
E1_2033 CHANNEL  ; RK_12 U4_Z 预焊下料Z轴轴7#位置
E1_2034 CHANNEL  ; RK_12 U4_Z 预焊下料Z轴轴8#位置
E1_2035 CHANNEL  ; RK_12 U4_Z 预焊下料Z轴轴8#位置
E1_2036 CHANNEL  ; RK_12 U4_Z 预焊下料Z轴轴9#位置
E1_2037 CHANNEL  ; RK_12 U4_Z 预焊下料Z轴轴9#位置
E1_2038 CHANNEL  ; RK_12 U4_Z 预焊下料Z轴轴10#位置
E1_2039 CHANNEL  ; RK_12 U4_Z 预焊下料Z轴轴10#位置
E1_204 CHANNEL  ; NC433_4 数据传送读字数
E1_205 CHANNEL  ; NC433_4 数据传送读源区域
E1_206 CHANNEL  ; NC433_4 数据传送读目标区域
E1_207 CHANNEL  ; NC433_4 数据传送读目标字
E1_208 CHANNEL  ; RK_12 U4_X 预焊上下料X轴轴直接操作位置
E1_209 CHANNEL  ; RK_12 U4_X 预焊上下料X轴轴直接操作位置
E1_21 CHANNEL  ; RK_02 U0_Y 电芯进料X轴轴直接操作位置
E1_210 CHANNEL  ; RK_12 U4_X 预焊上下料X轴轴直接操作速度
E1_2100 CHANNEL  ; RK_13 U4_U #1移载Y轴轴自动速度
E1_21000 CHANNEL  ; #9配方参数（伺服轴）
E1_2101 CHANNEL  ; RK_13 U4_U #1移载Y轴轴自动速度
E1_2102 CHANNEL  ; RK_13 U4_U #1移载Y轴轴 Jog 高速
E1_2103 CHANNEL  ; RK_13 U4_U #1移载Y轴轴 Jog 高速
E1_2104 CHANNEL  ; RK_13 U4_U #1移载Y轴轴 Jog 低速
E1_2105 CHANNEL  ; RK_13 U4_U #1移载Y轴轴 Jog 低速
E1_2106 CHANNEL  ; RK_13 U4_U #1移载Y轴轴加减速时间
E1_2107 CHANNEL  ; RK_13 U4_U #1移载Y轴轴加减速时间
E1_2108 CHANNEL  ; RK_13 U4_U #1移载Y轴轴正软极限
E1_2109 CHANNEL  ; RK_13 U4_U #1移载Y轴轴正软极限
E1_211 CHANNEL  ; RK_12 U4_X 预焊上下料X轴轴直接操作速度
E1_2110 CHANNEL  ; RK_13 U4_U #1移载Y轴轴负软极限
E1_2111 CHANNEL  ; RK_13 U4_U #1移载Y轴轴负软极限
E1_2112 CHANNEL  ; RK_13 U4_U #1移载Y轴轴原点偏移
E1_212 CHANNEL  ; RK_12 U4_X 预焊上下料X轴轴直接操作加速时间
E1_2120 CHANNEL  ; RK_13 U4_U #1移载Y轴待料位
E1_2121 CHANNEL  ; RK_13 U4_U #1移载Y轴待料位
E1_2122 CHANNEL  ; RK_13 U4_U #1移载Y轴取放料位
E1_2123 CHANNEL  ; RK_13 U4_U #1移载Y轴取放料位
E1_2124 CHANNEL  ; RK_13 U4_U #1移载Y轴压装位
E1_2125 CHANNEL  ; RK_13 U4_U #1移载Y轴压装位
E1_2126 CHANNEL  ; RK_13 U4_U #1移载Y轴#1轮廓检测位
E1_2127 CHANNEL  ; RK_13 U4_U #1移载Y轴#1轮廓检测位
E1_2128 CHANNEL  ; RK_13 U4_U #1移载Y轴#2轮廓检测位
E1_2129 CHANNEL  ; RK_13 U4_U #1移载Y轴#2轮廓检测位
E1_213 CHANNEL  ; RK_12 U4_X 预焊上下料X轴X轴直接操作加速时间
E1_2130 CHANNEL  ; RK_13 U4_U #1移载Y轴激光焊接位
E1_2131 CHANNEL  ; RK_13 U4_U #1移载Y轴激光焊接位
E1_2132 CHANNEL  ; RK_13 U4_U #1移载Y轴轴7#位置
E1_2133 CHANNEL  ; RK_13 U4_U #1移载Y轴轴7#位置
E1_2134 CHANNEL  ; RK_13 U4_U #1移载Y轴轴8#位置
E1_2135 CHANNEL  ; RK_13 U4_U #1移载Y轴轴8#位置
E1_2136 CHANNEL  ; RK_13 U4_U #1移载Y轴轴9#位置
E1_2137 CHANNEL  ; RK_13 U4_U #1移载Y轴轴9#位置
E1_2138 CHANNEL  ; RK_13 U4_U #1移载Y轴轴10#位置
E1_2139 CHANNEL  ; RK_13 U4_U #1移载Y轴轴10#位置
E1_214 CHANNEL  ; RK_12 U4_X 预焊上下料X轴轴直接操作减速时间
E1_215 CHANNEL  ; RK_12 U4_X 预焊上下料X轴轴直接操作减速时间
E1_216 CHANNEL  ; RK_12 U4_X 预焊上下料X轴轴存储器操作序列号
E1_217 CHANNEL  ; RK_12 U4_X 预焊上下料X轴轴特殊操作Override
E1_218 CHANNEL  ; RK_12 U4_X 预焊上下料X轴轴特殊操作示教地址
E1_219 CHANNEL  ; RK_12 U4_X 预焊上下料X轴轴特殊操作预留
E1_22 CHANNEL  ; RK_02 U0_Y 电芯进料X轴轴直接操作速度
E1_220 CHANNEL  ; RK_12 U4_Y 预焊上料Z轴轴直接操作位置
E1_2200 CHANNEL  ; RK_13 U6_X #2移载Y轴轴自动速度
E1_2201 CHANNEL  ; RK_13 U6_X #2移载Y轴轴自动速度
E1_2202 CHANNEL  ; RK_13 U6_X #2移载Y轴轴 Jog 高速
E1_2203 CHANNEL  ; RK_13 U6_X #2移载Y轴轴 Jog 高速
E1_2204 CHANNEL  ; RK_13 U6_X #2移载Y轴轴 Jog 低速
E1_2205 CHANNEL  ; RK_13 U6_X #2移载Y轴轴 Jog 低速
E1_2206 CHANNEL  ; RK_13 U6_X #2移载Y轴轴加减速时间
E1_2207 CHANNEL  ; RK_13 U6_X #2移载Y轴轴加减速时间
E1_2208 CHANNEL  ; RK_13 U6_X #2移载Y轴轴正软极限
E1_2209 CHANNEL  ; RK_13 U6_X #2移载Y轴轴正软极限
E1_221 CHANNEL  ; RK_12 U4_Y 预焊上料Z轴轴直接操作位置
E1_2210 CHANNEL  ; RK_13 U6_X #2移载Y轴轴负软极限
E1_2211 CHANNEL  ; RK_13 U6_X #2移载Y轴轴负软极限
E1_2212 CHANNEL  ; RK_13 U6_X #2移载Y轴轴原点偏移
E1_222 CHANNEL  ; RK_12 U4_Y 预焊上料Z轴轴直接操作速度
E1_2220 CHANNEL  ; RK_13 U6_X #2移载Y轴待料位
E1_2221 CHANNEL  ; RK_13 U6_X #2移载Y轴待料位
E1_2222 CHANNEL  ; RK_13 U6_X #2移载Y轴取放料位
E1_2223 CHANNEL  ; RK_13 U6_X #2移载Y轴取放料位
E1_2224 CHANNEL  ; RK_13 U6_X #2移载Y轴压装位
E1_2225 CHANNEL  ; RK_13 U6_X #2移载Y轴压装位
E1_2226 CHANNEL  ; RK_13 U6_X #2移载Y轴#1轮廓检测位
E1_2227 CHANNEL  ; RK_13 U6_X #2移载Y轴#1轮廓检测位
E1_2228 CHANNEL  ; RK_13 U6_X #2移载Y轴#2轮廓检测位
E1_2229 CHANNEL  ; RK_13 U6_X #2移载Y轴#2轮廓检测位
E1_223 CHANNEL  ; RK_12 U4_Y 预焊上料Z轴轴直接操作速度
E1_2230 CHANNEL  ; RK_13 U6_X #2移载Y轴激光焊接位
E1_2231 CHANNEL  ; RK_13 U6_X #2移载Y轴激光焊接位
E1_2232 CHANNEL  ; RK_13 U6_X #2移载Y轴轴7#位置
E1_2233 CHANNEL  ; RK_13 U6_X #2移载Y轴轴7#位置
E1_2234 CHANNEL  ; RK_13 U6_X #2移载Y轴轴8#位置
E1_2235 CHANNEL  ; RK_13 U6_X #2移载Y轴轴8#位置
E1_2236 CHANNEL  ; RK_13 U6_X #2移载Y轴轴9#位置
E1_2237 CHANNEL  ; RK_13 U6_X #2移载Y轴轴9#位置
E1_2238 CHANNEL  ; RK_13 U6_X #2移载Y轴轴10#位置
E1_2239 CHANNEL  ; RK_13 U6_X #2移载Y轴轴10#位置
E1_224 CHANNEL  ; RK_12 U4_Y 预焊上料Z轴轴直接操作加速时间
E1_225 CHANNEL  ; RK_12 U4_Y 预焊上料Z轴轴直接操作加速时间
E1_226 CHANNEL  ; RK_12 U4_Y 预焊上料Z轴轴直接操作减速时间
E1_227 CHANNEL  ; RK_12 U4_Y 预焊上料Z轴轴直接操作减速时间
E1_228 CHANNEL  ; RK_12 U4_Y 预焊上料Z轴轴存储器操作序列号
E1_229 CHANNEL  ; RK_12 U4_Y 预焊上料Z轴轴特殊操作Override
E1_23 CHANNEL  ; RK_02 U0_Y 电芯进料X轴轴直接操作速度
E1_230 CHANNEL  ; RK_12 U4_Y 预焊上料Z轴轴特殊操作示教地址
E1_2300 CHANNEL  ; RK_16 U6_Y 激光焊接X轴轴自动速度
E1_2301 CHANNEL  ; RK_16 U6_Y 激光焊接X轴轴自动速度
E1_2302 CHANNEL  ; RK_16 U6_Y 激光焊接X轴轴 Jog 高速
E1_2303 CHANNEL  ; RK_16 U6_Y 激光焊接X轴轴 Jog 高速
E1_2304 CHANNEL  ; RK_16 U6_Y 激光焊接X轴轴 Jog 低速
E1_2305 CHANNEL  ; RK_16 U6_Y 激光焊接X轴轴 Jog 低速
E1_2306 CHANNEL  ; RK_16 U6_Y 激光焊接X轴轴加减速时间
E1_2307 CHANNEL  ; RK_16 U6_Y 激光焊接X轴轴加减速时间
E1_2308 CHANNEL  ; RK_16 U6_Y 激光焊接X轴轴正软极限
E1_2309 CHANNEL  ; RK_16 U6_Y 激光焊接X轴轴正软极限
E1_231 CHANNEL  ; RK_12 U4_Y 预焊上料Z轴轴特殊操作预留
E1_2310 CHANNEL  ; RK_16 U6_Y 激光焊接X轴轴负软极限
E1_2311 CHANNEL  ; RK_16 U6_Y 激光焊接X轴轴负软极限
E1_2312 CHANNEL  ; RK_16 U6_Y 激光焊接X轴轴原点偏移
E1_232 CHANNEL  ; RK_12 U4_Z 预焊下料Z轴轴直接操作位置
E1_2320 CHANNEL  ; RK_16 U6_Y 激光焊接X轴待机位
E1_2321 CHANNEL  ; RK_16 U6_Y 激光焊接X轴待机位
E1_2322 CHANNEL  ; RK_16 U6_Y 激光焊接X轴#1移载焊接位
E1_2323 CHANNEL  ; RK_16 U6_Y 激光焊接X轴#1移载焊接位
E1_2324 CHANNEL  ; RK_16 U6_Y 激光焊接X轴#2移载焊接位
E1_2325 CHANNEL  ; RK_16 U6_Y 激光焊接X轴#2移载焊接位
E1_2326 CHANNEL  ; RK_16 U6_Y 激光焊接X轴轴4#位置
E1_2327 CHANNEL  ; RK_16 U6_Y 激光焊接X轴轴4#位置
E1_2328 CHANNEL  ; RK_16 U6_Y 激光焊接X轴轴5#位置
E1_2329 CHANNEL  ; RK_16 U6_Y 激光焊接X轴轴5#位置
E1_233 CHANNEL  ; RK_12 U4_Z 预焊下料Z轴轴直接操作位置
E1_2330 CHANNEL  ; RK_16 U6_Y 激光焊接X轴轴6#位置
E1_2331 CHANNEL  ; RK_16 U6_Y 激光焊接X轴轴6#位置
E1_2332 CHANNEL  ; RK_16 U6_Y 激光焊接X轴轴7#位置
E1_2333 CHANNEL  ; RK_16 U6_Y 激光焊接X轴轴7#位置
E1_2334 CHANNEL  ; RK_16 U6_Y 激光焊接X轴轴8#位置
E1_2335 CHANNEL  ; RK_16 U6_Y 激光焊接X轴轴8#位置
E1_2336 CHANNEL  ; RK_16 U6_Y 激光焊接X轴轴9#位置
E1_2337 CHANNEL  ; RK_16 U6_Y 激光焊接X轴轴9#位置
E1_2338 CHANNEL  ; RK_16 U6_Y 激光焊接X轴轴10#位置
E1_2339 CHANNEL  ; RK_16 U6_Y 激光焊接X轴轴10#位置
E1_234 CHANNEL  ; RK_12 U4_Z 预焊下料Z轴轴直接操作速度
E1_235 CHANNEL  ; RK_12 U4_Z 预焊下料Z轴轴直接操作速度
E1_236 CHANNEL  ; RK_12 U4_Z 预焊下料Z轴轴直接操作加速时间
E1_237 CHANNEL  ; RK_12 U4_Z 预焊下料Z轴轴直接操作加速时间
E1_238 CHANNEL  ; RK_12 U4_Z 预焊下料Z轴轴直接操作减速时间
E1_239 CHANNEL  ; RK_12 U4_Z 预焊下料Z轴轴直接操作减速时间
E1_24 CHANNEL  ; RK_02 U0_Y 电芯进料X轴轴直接操作加速时间
E1_240 CHANNEL  ; RK_12 U4_Z 预焊下料Z轴轴存储器操作序列号
E1_2400 CHANNEL  ; RK_16 U6_Z 激光焊接Z轴轴自动速度
E1_2401 CHANNEL  ; RK_16 U6_Z 激光焊接Z轴轴自动速度
E1_2402 CHANNEL  ; RK_16 U6_Z 激光焊接Z轴轴 Jog 高速
E1_2403 CHANNEL  ; RK_16 U6_Z 激光焊接Z轴轴 Jog 高速
E1_2404 CHANNEL  ; RK_16 U6_Z 激光焊接Z轴轴 Jog 低速
E1_2405 CHANNEL  ; RK_16 U6_Z 激光焊接Z轴轴 Jog 低速
E1_2406 CHANNEL  ; RK_16 U6_Z 激光焊接Z轴轴加减速时间
E1_2407 CHANNEL  ; RK_16 U6_Z 激光焊接Z轴轴加减速时间
E1_2408 CHANNEL  ; RK_16 U6_Z 激光焊接Z轴轴正软极限
E1_2409 CHANNEL  ; RK_16 U6_Z 激光焊接Z轴轴正软极限
E1_241 CHANNEL  ; RK_12 U4_Z 预焊下料Z轴轴特殊操作Override
E1_2410 CHANNEL  ; RK_16 U6_Z 激光焊接Z轴轴负软极限
E1_2411 CHANNEL  ; RK_16 U6_Z 激光焊接Z轴轴负软极限
E1_2412 CHANNEL  ; RK_16 U6_Z 激光焊接Z轴轴原点偏移
E1_242 CHANNEL  ; RK_12 U4_Z 预焊下料Z轴轴特殊操作示教地址
E1_2420 CHANNEL  ; RK_16 U6_Z 激光焊接Z轴待机位
E1_2421 CHANNEL  ; RK_16 U6_Z 激光焊接Z轴待机位
E1_2422 CHANNEL  ; RK_16 U6_Z 激光焊接Z轴#1移载焊接位
E1_2423 CHANNEL  ; RK_16 U6_Z 激光焊接Z轴#1移载焊接位
E1_2424 CHANNEL  ; RK_16 U6_Z 激光焊接Z轴#2移载焊接位
E1_2425 CHANNEL  ; RK_16 U6_Z 激光焊接Z轴#2移载焊接位
E1_2426 CHANNEL  ; RK_16 U6_Z 激光焊接Z轴轴4#位置
E1_2427 CHANNEL  ; RK_16 U6_Z 激光焊接Z轴轴4#位置
E1_2428 CHANNEL  ; RK_16 U6_Z 激光焊接Z轴轴5#位置
E1_2429 CHANNEL  ; RK_16 U6_Z 激光焊接Z轴轴5#位置
E1_243 CHANNEL  ; RK_12 U4_Z 预焊下料Z轴轴特殊操作预留
E1_2430 CHANNEL  ; RK_16 U6_Z 激光焊接Z轴轴6#位置
E1_2431 CHANNEL  ; RK_16 U6_Z 激光焊接Z轴轴6#位置
E1_2432 CHANNEL  ; RK_16 U6_Z 激光焊接Z轴轴7#位置
E1_2433 CHANNEL  ; RK_16 U6_Z 激光焊接Z轴轴7#位置
E1_2434 CHANNEL  ; RK_16 U6_Z 激光焊接Z轴轴8#位置
E1_2435 CHANNEL  ; RK_16 U6_Z 激光焊接Z轴轴8#位置
E1_2436 CHANNEL  ; RK_16 U6_Z 激光焊接Z轴轴9#位置
E1_2437 CHANNEL  ; RK_16 U6_Z 激光焊接Z轴轴9#位置
E1_2438 CHANNEL  ; RK_16 U6_Z 激光焊接Z轴轴10#位置
E1_2439 CHANNEL  ; RK_16 U6_Z 激光焊接Z轴轴10#位置
E1_244 CHANNEL  ; RK_13 U4_U #1移载Y轴轴直接操作位置
E1_245 CHANNEL  ; RK_13 U4_U #1移载Y轴轴直接操作位置
E1_246 CHANNEL  ; RK_13 U4_U #1移载Y轴轴直接操作速度
E1_247 CHANNEL  ; RK_13 U4_U #1移载Y轴轴直接操作速度
E1_248 CHANNEL  ; RK_13 U4_U #1移载Y轴轴直接操作加速时间
E1_249 CHANNEL  ; RK_13 U4_U #1移载Y轴轴直接操作加速时间
E1_25 CHANNEL  ; RK_02 U0_Y 电芯进料X轴轴直接操作加速时间
E1_250 CHANNEL  ; RK_13 U4_U #1移载Y轴轴直接操作减速时间
E1_25000 CHANNEL  ; #1配方参数（Hipot）
E1_25010 CHANNEL  ; #2配方参数（Hipot）
E1_25020 CHANNEL  ; #3配方参数（Hipot）
E1_25030 CHANNEL  ; #4配方参数（Hipot）
E1_25040 CHANNEL  ; #5配方参数（Hipot）
E1_25050 CHANNEL  ; #6配方参数（Hipot）
E1_25060 CHANNEL  ; #7配方参数（Hipot）
E1_25070 CHANNEL  ; #8配方参数（Hipot）
E1_25080 CHANNEL  ; #9配方参数（Hipot）
E1_251 CHANNEL  ; RK_13 U4_U #1移载Y轴轴直接操作减速时间
E1_252 CHANNEL  ; RK_13 U4_U #1移载Y轴轴存储器操作序列号
E1_25200 CHANNEL  ; #1配方参数（Profile）
E1_25210 CHANNEL  ; #2配方参数（Profile）
E1_25220 CHANNEL  ; #3配方参数（Profile）
E1_25230 CHANNEL  ; #4配方参数（Profile）
E1_25240 CHANNEL  ; #5配方参数（Profile）
E1_25250 CHANNEL  ; #6配方参数（Profile）
E1_25260 CHANNEL  ; #7配方参数（Profile）
E1_25270 CHANNEL  ; #8配方参数（Profile）
E1_25280 CHANNEL  ; #9配方参数（Profile）
E1_253 CHANNEL  ; RK_13 U4_U #1移载Y轴轴特殊操作Override
E1_254 CHANNEL  ; RK_13 U4_U #1移载Y轴轴特殊操作示教地址
E1_25400 CHANNEL  ; #1配方参数（铝壳料盘列数）
E1_25410 CHANNEL  ; #2配方参数（铝壳料盘列数）
E1_25420 CHANNEL  ; #3配方参数（铝壳料盘列数）
E1_25430 CHANNEL  ; #4配方参数（铝壳料盘列数）
E1_25440 CHANNEL  ; #5配方参数（铝壳料盘列数）
E1_25450 CHANNEL  ; #6配方参数（铝壳料盘列数）
E1_25460 CHANNEL  ; #7配方参数（铝壳料盘列数）
E1_25470 CHANNEL  ; #8配方参数（铝壳料盘列数）
E1_25480 CHANNEL  ; #9配方参数（铝壳料盘列数）
E1_255 CHANNEL  ; RK_13 U4_U #1移载Y轴轴特殊操作预留
E1_25500 CHANNEL  ; #1配方参数（铝壳料盘列间距）
E1_25510 CHANNEL  ; #2配方参数（铝壳料盘列间距）
E1_25520 CHANNEL  ; #3配方参数（铝壳料盘列间距）
E1_25530 CHANNEL  ; #4配方参数（铝壳料盘列间距）
E1_25540 CHANNEL  ; #5配方参数（铝壳料盘列间距）
E1_25550 CHANNEL  ; #6配方参数（铝壳料盘列间距）
E1_25560 CHANNEL  ; #7配方参数（铝壳料盘列间距）
E1_25570 CHANNEL  ; #8配方参数（铝壳料盘列间距）
E1_25580 CHANNEL  ; #9配方参数（铝壳料盘列间距）
E1_256 CHANNEL  ; RK_12 U4_X 预焊上下料X轴轴当前位置
E1_257 CHANNEL  ; RK_12 U4_X 预焊上下料X轴轴当前位置
E1_258 CHANNEL  ; RK_12 U4_X 预焊上下料X轴轴存储器操作正被执行序列号
E1_259 CHANNEL  ; RK_12 U4_X 预焊上下料X轴轴存储器操作正被执行序列号
E1_26 CHANNEL  ; RK_02 U0_Y 电芯进料X轴轴直接操作减速时间
E1_260 CHANNEL  ; RK_12 U4_Y 预焊上料Z轴轴当前位置
E1_2600 CHANNEL  ; RK_06 U8_X 电池上下料X轴轴自动速度
E1_2601 CHANNEL  ; RK_06 U8_X 电池上下料X轴轴自动速度
E1_2602 CHANNEL  ; RK_06 U8_X 电池上下料X轴轴 Jog 高速
E1_2603 CHANNEL  ; RK_06 U8_X 电池上下料X轴轴 Jog 高速
E1_2604 CHANNEL  ; RK_06 U8_X 电池上下料X轴轴 Jog 低速
E1_2605 CHANNEL  ; RK_06 U8_X 电池上下料X轴轴 Jog 低速
E1_2606 CHANNEL  ; RK_06 U8_X 电池上下料X轴轴加减速时间
E1_2607 CHANNEL  ; RK_06 U8_X 电池上下料X轴轴加减速时间
E1_2608 CHANNEL  ; RK_06 U8_X 电池上下料X轴轴正软极限
E1_2609 CHANNEL  ; RK_06 U8_X 电池上下料X轴轴正软极限
E1_261 CHANNEL  ; RK_12 U4_Y 预焊上料Z轴轴当前位置
E1_2610 CHANNEL  ; RK_06 U8_X 电池上下料X轴轴负软极限
E1_2611 CHANNEL  ; RK_06 U8_X 电池上下料X轴轴负软极限
E1_2612 CHANNEL  ; RK_06 U8_X 电池上下料X轴轴原点偏移
E1_262 CHANNEL  ; RK_12 U4_Y 预焊上料Z轴轴存储器操作正被执行序列号
E1_2620 CHANNEL  ; RK_06 U8_X 电池上下料X轴待机位
E1_2621 CHANNEL  ; RK_06 U8_X 电池上下料X轴待机位
E1_2622 CHANNEL  ; RK_06 U8_X 电池上下料X轴铝壳除尘取料位
E1_2623 CHANNEL  ; RK_06 U8_X 电池上下料X轴铝壳除尘取料位
E1_2624 CHANNEL  ; RK_06 U8_X 电池上下料X轴#1入壳放料位
E1_2625 CHANNEL  ; RK_06 U8_X 电池上下料X轴#1入壳放料位
E1_2626 CHANNEL  ; RK_06 U8_X 电池上下料X轴#2入壳放料位
E1_2627 CHANNEL  ; RK_06 U8_X 电池上下料X轴#2入壳放料位
E1_2628 CHANNEL  ; RK_06 U8_X 电池上下料X轴#1入壳取料位
E1_2629 CHANNEL  ; RK_06 U8_X 电池上下料X轴#1入壳取料位
E1_263 CHANNEL  ; RK_12 U4_Y 预焊上料Z轴轴存储器操作正被执行序列号
E1_2630 CHANNEL  ; RK_06 U8_X 电池上下料X轴#2入壳取料位
E1_2631 CHANNEL  ; RK_06 U8_X 电池上下料X轴#2入壳取料位
E1_2632 CHANNEL  ; RK_06 U8_X 电池上下料X轴#1Hipot检测放料位
E1_2633 CHANNEL  ; RK_06 U8_X 电池上下料X轴#1Hipot检测放料位
E1_2634 CHANNEL  ; RK_06 U8_X 电池上下料X轴#2Hipot检测放料位
E1_2635 CHANNEL  ; RK_06 U8_X 电池上下料X轴#2Hipot检测放料位
E1_2636 CHANNEL  ; RK_06 U8_X 电池上下料X轴轴9#位置
E1_2637 CHANNEL  ; RK_06 U8_X 电池上下料X轴轴9#位置
E1_2638 CHANNEL  ; RK_06 U8_X 电池上下料X轴轴10#位置
E1_2639 CHANNEL  ; RK_06 U8_X 电池上下料X轴轴10#位置
E1_264 CHANNEL  ; RK_12 U4_Z 预焊下料Z轴轴当前位置
E1_265 CHANNEL  ; RK_12 U4_Z 预焊下料Z轴轴当前位置
E1_266 CHANNEL  ; RK_12 U4_Z 预焊下料Z轴轴存储器操作正被执行序列号
E1_267 CHANNEL  ; RK_12 U4_Z 预焊下料Z轴轴存储器操作正被执行序列号
E1_268 CHANNEL  ; RK_13 U4_U #1移载Y轴轴当前位置
E1_269 CHANNEL  ; RK_13 U4_U #1移载Y轴轴当前位置
E1_27 CHANNEL  ; RK_02 U0_Y 电芯进料X轴轴直接操作减速时间
E1_270 CHANNEL  ; RK_13 U4_U #1移载Y轴轴存储器操作正被执行序列号
E1_2700 CHANNEL  ; RK_07 U8_Y 铝壳进料X轴轴自动速度
E1_2701 CHANNEL  ; RK_07 U8_Y 铝壳进料X轴轴自动速度
E1_2702 CHANNEL  ; RK_07 U8_Y 铝壳进料X轴轴 Jog 高速
E1_2703 CHANNEL  ; RK_07 U8_Y 铝壳进料X轴轴 Jog 高速
E1_2704 CHANNEL  ; RK_07 U8_Y 铝壳进料X轴轴 Jog 低速
E1_2705 CHANNEL  ; RK_07 U8_Y 铝壳进料X轴轴 Jog 低速
E1_2706 CHANNEL  ; RK_07 U8_Y 铝壳进料X轴轴加减速时间
E1_2707 CHANNEL  ; RK_07 U8_Y 铝壳进料X轴轴加减速时间
E1_2708 CHANNEL  ; RK_07 U8_Y 铝壳进料X轴轴正软极限
E1_2709 CHANNEL  ; RK_07 U8_Y 铝壳进料X轴轴正软极限
E1_271 CHANNEL  ; RK_13 U4_U #1移载Y轴轴存储器操作正被执行序列号
E1_2710 CHANNEL  ; RK_07 U8_Y 铝壳进料X轴轴负软极限
E1_2711 CHANNEL  ; RK_07 U8_Y 铝壳进料X轴轴负软极限
E1_2712 CHANNEL  ; RK_07 U8_Y 铝壳进料X轴轴原点偏移
E1_2720 CHANNEL  ; RK_07 U8_Y 铝壳进料X轴等待位
E1_2721 CHANNEL  ; RK_07 U8_Y 铝壳进料X轴等待位
E1_2722 CHANNEL  ; RK_07 U8_Y 铝壳进料X轴取料位
E1_2723 CHANNEL  ; RK_07 U8_Y 铝壳进料X轴取料位
E1_2724 CHANNEL  ; RK_07 U8_Y 铝壳进料X轴放料位
E1_2725 CHANNEL  ; RK_07 U8_Y 铝壳进料X轴放料位
E1_2726 CHANNEL  ; RK_07 U8_Y 铝壳进料X轴轴4#位置
E1_2727 CHANNEL  ; RK_07 U8_Y 铝壳进料X轴轴4#位置
E1_2728 CHANNEL  ; RK_07 U8_Y 铝壳进料X轴轴5#位置
E1_2729 CHANNEL  ; RK_07 U8_Y 铝壳进料X轴轴5#位置
E1_2730 CHANNEL  ; RK_07 U8_Y 铝壳进料X轴轴6#位置
E1_2731 CHANNEL  ; RK_07 U8_Y 铝壳进料X轴轴6#位置
E1_2732 CHANNEL  ; RK_07 U8_Y 铝壳进料X轴轴7#位置
E1_2733 CHANNEL  ; RK_07 U8_Y 铝壳进料X轴轴7#位置
E1_2734 CHANNEL  ; RK_07 U8_Y 铝壳进料X轴轴8#位置
E1_2735 CHANNEL  ; RK_07 U8_Y 铝壳进料X轴轴8#位置
E1_2736 CHANNEL  ; RK_07 U8_Y 铝壳进料X轴轴9#位置
E1_2737 CHANNEL  ; RK_07 U8_Y 铝壳进料X轴轴9#位置
E1_2738 CHANNEL  ; RK_07 U8_Y 铝壳进料X轴轴10#位置
E1_2739 CHANNEL  ; RK_07 U8_Y 铝壳进料X轴轴10#位置
E1_2740 CHANNEL  ; RK_07 U8_Y 铝壳进料X轴#1取料位
E1_2741 CHANNEL  ; RK_07 U8_Y 铝壳进料X轴#1取料位
E1_2742 CHANNEL  ; RK_07 U8_Y 铝壳进料X轴#2取料位
E1_2743 CHANNEL  ; RK_07 U8_Y 铝壳进料X轴#2取料位
E1_2744 CHANNEL  ; RK_07 U8_Y 铝壳进料X轴#3取料位
E1_2745 CHANNEL  ; RK_07 U8_Y 铝壳进料X轴#3取料位
E1_2746 CHANNEL  ; RK_07 U8_Y 铝壳进料X轴#4取料位
E1_2747 CHANNEL  ; RK_07 U8_Y 铝壳进料X轴#4取料位
E1_2748 CHANNEL  ; RK_07 U8_Y 铝壳进料X轴#5取料位
E1_2749 CHANNEL  ; RK_07 U8_Y 铝壳进料X轴#5取料位
E1_28 CHANNEL  ; RK_02 U0_Y 电芯进料X轴轴存储器操作序列号
E1_2800 CHANNEL  ; RK_07 U8_Z 铝壳上料移载Y轴轴自动速度
E1_2801 CHANNEL  ; RK_07 U8_Z 铝壳上料移载Y轴轴自动速度
E1_2802 CHANNEL  ; RK_07 U8_Z 铝壳上料移载Y轴轴 Jog 高速
E1_2803 CHANNEL  ; RK_07 U8_Z 铝壳上料移载Y轴轴 Jog 高速
E1_2804 CHANNEL  ; RK_07 U8_Z 铝壳上料移载Y轴轴 Jog 低速
E1_2805 CHANNEL  ; RK_07 U8_Z 铝壳上料移载Y轴轴 Jog 低速
E1_2806 CHANNEL  ; RK_07 U8_Z 铝壳上料移载Y轴轴加减速时间
E1_2807 CHANNEL  ; RK_07 U8_Z 铝壳上料移载Y轴轴加减速时间
E1_2808 CHANNEL  ; RK_07 U8_Z 铝壳上料移载Y轴轴正软极限
E1_2809 CHANNEL  ; RK_07 U8_Z 铝壳上料移载Y轴轴正软极限
E1_2810 CHANNEL  ; RK_07 U8_Z 铝壳上料移载Y轴轴负软极限
E1_2811 CHANNEL  ; RK_07 U8_Z 铝壳上料移载Y轴轴负软极限
E1_2812 CHANNEL  ; RK_07 U8_Z 铝壳上料移载Y轴轴原点偏移
E1_2820 CHANNEL  ; RK_07 U8_Z 铝壳上料移载Y轴待料位
E1_2821 CHANNEL  ; RK_07 U8_Z 铝壳上料移载Y轴待料位
E1_2822 CHANNEL  ; RK_07 U8_Z 铝壳上料移载Y轴#1铝壳上料位
E1_2823 CHANNEL  ; RK_07 U8_Z 铝壳上料移载Y轴#1铝壳上料位
E1_2824 CHANNEL  ; RK_07 U8_Z 铝壳上料移载Y轴#2铝壳上料位
E1_2825 CHANNEL  ; RK_07 U8_Z 铝壳上料移载Y轴#2铝壳上料位
E1_2826 CHANNEL  ; RK_07 U8_Z 铝壳上料移载Y轴#3铝壳托盘下料位
E1_2827 CHANNEL  ; RK_07 U8_Z 铝壳上料移载Y轴#3铝壳托盘下料位
E1_2828 CHANNEL  ; RK_07 U8_Z 铝壳上料移载Y轴铝壳取料位
E1_2829 CHANNEL  ; RK_07 U8_Z 铝壳上料移载Y轴铝壳取料位
E1_2830 CHANNEL  ; RK_07 U8_Z 铝壳上料移载Y轴轴6#位置
E1_2831 CHANNEL  ; RK_07 U8_Z 铝壳上料移载Y轴轴6#位置
E1_2832 CHANNEL  ; RK_07 U8_Z 铝壳上料移载Y轴轴7#位置
E1_2833 CHANNEL  ; RK_07 U8_Z 铝壳上料移载Y轴轴7#位置
E1_2834 CHANNEL  ; RK_07 U8_Z 铝壳上料移载Y轴轴8#位置
E1_2835 CHANNEL  ; RK_07 U8_Z 铝壳上料移载Y轴轴8#位置
E1_2836 CHANNEL  ; RK_07 U8_Z 铝壳上料移载Y轴轴9#位置
E1_2837 CHANNEL  ; RK_07 U8_Z 铝壳上料移载Y轴轴9#位置
E1_2838 CHANNEL  ; RK_07 U8_Z 铝壳上料移载Y轴轴10#位置
E1_2839 CHANNEL  ; RK_07 U8_Z 铝壳上料移载Y轴轴10#位置
E1_2840 CHANNEL  ; RK_07 U8_Z 铝壳上料移载Y轴#1取料位
E1_2841 CHANNEL  ; RK_07 U8_Z 铝壳上料移载Y轴#1取料位
E1_2842 CHANNEL  ; RK_07 U8_Z 铝壳上料移载Y轴#2取料位
E1_2843 CHANNEL  ; RK_07 U8_Z 铝壳上料移载Y轴#2取料位
E1_2844 CHANNEL  ; RK_07 U8_Z 铝壳上料移载Y轴#3取料位
E1_2845 CHANNEL  ; RK_07 U8_Z 铝壳上料移载Y轴#3取料位
E1_29 CHANNEL  ; RK_02 U0_Y 电芯进料X轴轴特殊操作Override
E1_2900 CHANNEL  ; RK_10 U8_U 电池除尘上料X轴轴自动速度
E1_2901 CHANNEL  ; RK_10 U8_U 电池除尘上料X轴轴自动速度
E1_2902 CHANNEL  ; RK_10 U8_U 电池除尘上料X轴轴 Jog 高速
E1_2903 CHANNEL  ; RK_10 U8_U 电池除尘上料X轴轴 Jog 高速
E1_2904 CHANNEL  ; RK_10 U8_U 电池除尘上料X轴轴 Jog 低速
E1_2905 CHANNEL  ; RK_10 U8_U 电池除尘上料X轴轴 Jog 低速
E1_2906 CHANNEL  ; RK_10 U8_U 电池除尘上料X轴轴加减速时间
E1_2907 CHANNEL  ; RK_10 U8_U 电池除尘上料X轴轴加减速时间
E1_2908 CHANNEL  ; RK_10 U8_U 电池除尘上料X轴轴正软极限
E1_2909 CHANNEL  ; RK_10 U8_U 电池除尘上料X轴轴正软极限
E1_2910 CHANNEL  ; RK_10 U8_U 电池除尘上料X轴轴负软极限
E1_2911 CHANNEL  ; RK_10 U8_U 电池除尘上料X轴轴负软极限
E1_2912 CHANNEL  ; RK_10 U8_U 电池除尘上料X轴轴原点偏移
E1_2920 CHANNEL  ; RK_10 U8_U 电池除尘上料X轴待料位
E1_2921 CHANNEL  ; RK_10 U8_U 电池除尘上料X轴待料位
E1_2922 CHANNEL  ; RK_10 U8_U 电池除尘上料X轴#1Hipot检测取料位
E1_2923 CHANNEL  ; RK_10 U8_U 电池除尘上料X轴#1Hipot检测取料位
E1_2924 CHANNEL  ; RK_10 U8_U 电池除尘上料X轴#2Hipot检测取料位
E1_2925 CHANNEL  ; RK_10 U8_U 电池除尘上料X轴#2Hipot检测取料位
E1_2926 CHANNEL  ; RK_10 U8_U 电池除尘上料X轴Hipot OK放料位
E1_2927 CHANNEL  ; RK_10 U8_U 电池除尘上料X轴Hipot OK放料位
E1_2928 CHANNEL  ; RK_10 U8_U 电池除尘上料X轴Hipot NG放料位
E1_2929 CHANNEL  ; RK_10 U8_U 电池除尘上料X轴Hipot NG放料位
E1_2930 CHANNEL  ; RK_10 U8_U 电池除尘上料X轴轴6#位置
E1_2931 CHANNEL  ; RK_10 U8_U 电池除尘上料X轴轴6#位置
E1_2932 CHANNEL  ; RK_10 U8_U 电池除尘上料X轴轴7#位置
E1_2933 CHANNEL  ; RK_10 U8_U 电池除尘上料X轴轴7#位置
E1_2934 CHANNEL  ; RK_10 U8_U 电池除尘上料X轴轴8#位置
E1_2935 CHANNEL  ; RK_10 U8_U 电池除尘上料X轴轴8#位置
E1_2936 CHANNEL  ; RK_10 U8_U 电池除尘上料X轴轴9#位置
E1_2937 CHANNEL  ; RK_10 U8_U 电池除尘上料X轴轴9#位置
E1_2938 CHANNEL  ; RK_10 U8_U 电池除尘上料X轴轴10#位置
E1_2939 CHANNEL  ; RK_10 U8_U 电池除尘上料X轴轴10#位置
E1_299 CHANNEL  ; NC433_6 数据传送写字数
E1_3 CHANNEL  ; NC433_0 数据传送定目标地址
E1_30 CHANNEL  ; RK_02 U0_Y 电芯进料X轴轴特殊操作示教地址
E1_300 CHANNEL  ; NC433_6 数据传送写源区域
E1_301 CHANNEL  ; NC433_6 数据传送定源字
E1_302 CHANNEL  ; NC433_6 数据传送定目标地址
E1_303 CHANNEL  ; NC433_6 数据传送读字数
E1_304 CHANNEL  ; NC433_6 数据传送读源区域
E1_305 CHANNEL  ; NC433_6 数据传送读目标区域
E1_306 CHANNEL  ; NC433_6 数据传送读目标字
E1_307 CHANNEL  ; RK_13 U6_X #2移载Y轴轴直接操作位置
E1_308 CHANNEL  ; RK_13 U6_X #2移载Y轴轴直接操作位置
E1_309 CHANNEL  ; RK_13 U6_X #2移载Y轴轴直接操作速度
E1_31 CHANNEL  ; RK_02 U0_Y 电芯进料X轴轴特殊操作预留
E1_310 CHANNEL  ; RK_13 U6_X #2移载Y轴轴直接操作速度
E1_311 CHANNEL  ; RK_13 U6_X #2移载Y轴轴直接操作加速时间
E1_312 CHANNEL  ; RK_13 U6_X #2移载Y轴X轴直接操作加速时间
E1_313 CHANNEL  ; RK_13 U6_X #2移载Y轴轴直接操作减速时间
E1_314 CHANNEL  ; RK_13 U6_X #2移载Y轴轴直接操作减速时间
E1_315 CHANNEL  ; RK_13 U6_X #2移载Y轴轴存储器操作序列号
E1_316 CHANNEL  ; RK_13 U6_X #2移载Y轴轴特殊操作Override
E1_317 CHANNEL  ; RK_13 U6_X #2移载Y轴轴特殊操作示教地址
E1_318 CHANNEL  ; RK_13 U6_X #2移载Y轴轴特殊操作预留
E1_319 CHANNEL  ; RK_16 U6_Y 激光焊接X轴轴直接操作位置
E1_32 CHANNEL  ; RK_02 U0_Z 电芯进料Z轴轴直接操作位置
E1_320 CHANNEL  ; RK_16 U6_Y 激光焊接X轴轴直接操作位置
E1_321 CHANNEL  ; RK_16 U6_Y 激光焊接X轴轴直接操作速度
E1_322 CHANNEL  ; RK_16 U6_Y 激光焊接X轴轴直接操作速度
E1_323 CHANNEL  ; RK_16 U6_Y 激光焊接X轴轴直接操作加速时间
E1_324 CHANNEL  ; RK_16 U6_Y 激光焊接X轴轴直接操作加速时间
E1_325 CHANNEL  ; RK_16 U6_Y 激光焊接X轴轴直接操作减速时间
E1_326 CHANNEL  ; RK_16 U6_Y 激光焊接X轴轴直接操作减速时间
E1_327 CHANNEL  ; RK_16 U6_Y 激光焊接X轴轴存储器操作序列号
E1_328 CHANNEL  ; RK_16 U6_Y 激光焊接X轴轴特殊操作Override
E1_329 CHANNEL  ; RK_16 U6_Y 激光焊接X轴轴特殊操作示教地址
E1_33 CHANNEL  ; RK_02 U0_Z 电芯进料Z轴轴直接操作位置
E1_330 CHANNEL  ; RK_16 U6_Y 激光焊接X轴轴特殊操作预留
E1_331 CHANNEL  ; RK_16 U6_Z 激光焊接Z轴轴直接操作位置
E1_332 CHANNEL  ; RK_16 U6_Z 激光焊接Z轴轴直接操作位置
E1_333 CHANNEL  ; RK_16 U6_Z 激光焊接Z轴轴直接操作速度
E1_334 CHANNEL  ; RK_16 U6_Z 激光焊接Z轴轴直接操作速度
E1_335 CHANNEL  ; RK_16 U6_Z 激光焊接Z轴轴直接操作加速时间
E1_336 CHANNEL  ; RK_16 U6_Z 激光焊接Z轴轴直接操作加速时间
E1_337 CHANNEL  ; RK_16 U6_Z 激光焊接Z轴轴直接操作减速时间
E1_338 CHANNEL  ; RK_16 U6_Z 激光焊接Z轴轴直接操作减速时间
E1_339 CHANNEL  ; RK_16 U6_Z 激光焊接Z轴轴存储器操作序列号
E1_34 CHANNEL  ; RK_02 U0_Z 电芯进料Z轴轴直接操作速度
E1_340 CHANNEL  ; RK_16 U6_Z 激光焊接Z轴轴特殊操作Override
E1_341 CHANNEL  ; RK_16 U6_Z 激光焊接Z轴轴特殊操作示教地址
E1_342 CHANNEL  ; RK_16 U6_Z 激光焊接Z轴轴特殊操作预留
E1_35 CHANNEL  ; RK_02 U0_Z 电芯进料Z轴轴直接操作速度
E1_355 CHANNEL  ; RK_13 U6_X #2移载Y轴轴当前位置
E1_356 CHANNEL  ; RK_13 U6_X #2移载Y轴轴当前位置
E1_357 CHANNEL  ; RK_13 U6_X #2移载Y轴轴存储器操作正被执行序列号
E1_358 CHANNEL  ; RK_13 U6_X #2移载Y轴轴存储器操作正被执行序列号
E1_359 CHANNEL  ; RK_16 U6_Y 激光焊接X轴轴当前位置
E1_36 CHANNEL  ; RK_02 U0_Z 电芯进料Z轴轴直接操作加速时间
E1_360 CHANNEL  ; RK_16 U6_Y 激光焊接X轴轴当前位置
E1_361 CHANNEL  ; RK_16 U6_Y 激光焊接X轴轴存储器操作正被执行序列号
E1_362 CHANNEL  ; RK_16 U6_Y 激光焊接X轴轴存储器操作正被执行序列号
E1_363 CHANNEL  ; RK_16 U6_Z 激光焊接Z轴轴当前位置
E1_364 CHANNEL  ; RK_16 U6_Z 激光焊接Z轴轴当前位置
E1_365 CHANNEL  ; RK_16 U6_Z 激光焊接Z轴轴存储器操作正被执行序列号
E1_366 CHANNEL  ; RK_16 U6_Z 激光焊接Z轴轴存储器操作正被执行序列号
E1_37 CHANNEL  ; RK_02 U0_Z 电芯进料Z轴轴直接操作加速时间
E1_38 CHANNEL  ; RK_02 U0_Z 电芯进料Z轴轴直接操作减速时间
E1_39 CHANNEL  ; RK_02 U0_Z 电芯进料Z轴轴直接操作减速时间
E1_4 CHANNEL  ; NC433_0 数据传送读字数
E1_40 CHANNEL  ; RK_02 U0_Z 电芯进料Z轴轴存储器操作序列号
E1_400 CHANNEL  ; NC433_8 数据传送写字数
E1_401 CHANNEL  ; NC433_8 数据传送写源区域
E1_402 CHANNEL  ; NC433_8 数据传送定源字
E1_403 CHANNEL  ; NC433_8 数据传送定目标地址
E1_404 CHANNEL  ; NC433_8 数据传送读字数
E1_405 CHANNEL  ; NC433_8 数据传送读源区域
E1_406 CHANNEL  ; NC433_8 数据传送读目标区域
E1_407 CHANNEL  ; NC433_8 数据传送读目标字
E1_408 CHANNEL  ; RK_06 U8_X 电池上下料X轴轴直接操作位置
E1_409 CHANNEL  ; RK_06 U8_X 电池上下料X轴轴直接操作位置
E1_41 CHANNEL  ; RK_02 U0_Z 电芯进料Z轴轴特殊操作Override
E1_410 CHANNEL  ; RK_06 U8_X 电池上下料X轴轴直接操作速度
E1_411 CHANNEL  ; RK_06 U8_X 电池上下料X轴轴直接操作速度
E1_412 CHANNEL  ; RK_06 U8_X 电池上下料X轴轴直接操作加速时间
E1_413 CHANNEL  ; RK_06 U8_X 电池上下料X轴X轴直接操作加速时间
E1_414 CHANNEL  ; RK_06 U8_X 电池上下料X轴轴直接操作减速时间
E1_415 CHANNEL  ; RK_06 U8_X 电池上下料X轴轴直接操作减速时间
E1_416 CHANNEL  ; RK_06 U8_X 电池上下料X轴轴存储器操作序列号
E1_417 CHANNEL  ; RK_06 U8_X 电池上下料X轴轴特殊操作Override
E1_418 CHANNEL  ; RK_06 U8_X 电池上下料X轴轴特殊操作示教地址
E1_419 CHANNEL  ; RK_06 U8_X 电池上下料X轴轴特殊操作预留
E1_42 CHANNEL  ; RK_02 U0_Z 电芯进料Z轴轴特殊操作示教地址
E1_420 CHANNEL  ; RK_07 U8_Y 铝壳进料X轴轴直接操作位置
E1_421 CHANNEL  ; RK_07 U8_Y 铝壳进料X轴轴直接操作位置
E1_422 CHANNEL  ; RK_07 U8_Y 铝壳进料X轴轴直接操作速度
E1_423 CHANNEL  ; RK_07 U8_Y 铝壳进料X轴轴直接操作速度
E1_424 CHANNEL  ; RK_07 U8_Y 铝壳进料X轴轴直接操作加速时间
E1_425 CHANNEL  ; RK_07 U8_Y 铝壳进料X轴轴直接操作加速时间
E1_426 CHANNEL  ; RK_07 U8_Y 铝壳进料X轴轴直接操作减速时间
E1_427 CHANNEL  ; RK_07 U8_Y 铝壳进料X轴轴直接操作减速时间
E1_428 CHANNEL  ; RK_07 U8_Y 铝壳进料X轴轴存储器操作序列号
E1_429 CHANNEL  ; RK_07 U8_Y 铝壳进料X轴轴特殊操作Override
E1_43 CHANNEL  ; RK_02 U0_Z 电芯进料Z轴轴特殊操作预留
E1_430 CHANNEL  ; RK_07 U8_Y 铝壳进料X轴轴特殊操作示教地址
E1_431 CHANNEL  ; RK_07 U8_Y 铝壳进料X轴轴特殊操作预留
E1_432 CHANNEL  ; RK_07 U8_Z 铝壳上料移载Y轴轴直接操作位置
E1_433 CHANNEL  ; RK_07 U8_Z 铝壳上料移载Y轴轴直接操作位置
E1_434 CHANNEL  ; RK_07 U8_Z 铝壳上料移载Y轴轴直接操作速度
E1_435 CHANNEL  ; RK_07 U8_Z 铝壳上料移载Y轴轴直接操作速度
E1_436 CHANNEL  ; RK_07 U8_Z 铝壳上料移载Y轴轴直接操作加速时间
E1_437 CHANNEL  ; RK_07 U8_Z 铝壳上料移载Y轴轴直接操作加速时间
E1_438 CHANNEL  ; RK_07 U8_Z 铝壳上料移载Y轴轴直接操作减速时间
E1_439 CHANNEL  ; RK_07 U8_Z 铝壳上料移载Y轴轴直接操作减速时间
E1_44 CHANNEL  ; RK_03 U0_U 电芯上料X轴轴直接操作位置
E1_440 CHANNEL  ; RK_07 U8_Z 铝壳上料移载Y轴轴存储器操作序列号
E1_441 CHANNEL  ; RK_07 U8_Z 铝壳上料移载Y轴轴特殊操作Override
E1_442 CHANNEL  ; RK_07 U8_Z 铝壳上料移载Y轴轴特殊操作示教地址
E1_443 CHANNEL  ; RK_07 U8_Z 铝壳上料移载Y轴轴特殊操作预留
E1_444 CHANNEL  ; RK_10 U8_U 电池除尘上料X轴轴直接操作位置
E1_445 CHANNEL  ; RK_10 U8_U 电池除尘上料X轴轴直接操作位置
E1_446 CHANNEL  ; RK_10 U8_U 电池除尘上料X轴轴直接操作速度
E1_447 CHANNEL  ; RK_10 U8_U 电池除尘上料X轴轴直接操作速度
E1_448 CHANNEL  ; RK_10 U8_U 电池除尘上料X轴轴直接操作加速时间
E1_449 CHANNEL  ; RK_10 U8_U 电池除尘上料X轴轴直接操作加速时间
E1_45 CHANNEL  ; RK_03 U0_U 电芯上料X轴轴直接操作位置
E1_450 CHANNEL  ; RK_10 U8_U 电池除尘上料X轴轴直接操作减速时间
E1_451 CHANNEL  ; RK_10 U8_U 电池除尘上料X轴轴直接操作减速时间
E1_452 CHANNEL  ; RK_10 U8_U 电池除尘上料X轴轴存储器操作序列号
E1_453 CHANNEL  ; RK_10 U8_U 电池除尘上料X轴轴特殊操作Override
E1_454 CHANNEL  ; RK_10 U8_U 电池除尘上料X轴轴特殊操作示教地址
E1_455 CHANNEL  ; RK_10 U8_U 电池除尘上料X轴轴特殊操作预留
E1_456 CHANNEL  ; RK_06 U8_X 电池上下料X轴轴当前位置
E1_457 CHANNEL  ; RK_06 U8_X 电池上下料X轴轴当前位置
E1_458 CHANNEL  ; RK_06 U8_X 电池上下料X轴轴存储器操作正被执行序列号
E1_459 CHANNEL  ; RK_06 U8_X 电池上下料X轴轴存储器操作正被执行序列号
E1_46 CHANNEL  ; RK_03 U0_U 电芯上料X轴轴直接操作速度
E1_460 CHANNEL  ; RK_07 U8_Y 铝壳进料X轴轴当前位置
E1_461 CHANNEL  ; RK_07 U8_Y 铝壳进料X轴轴当前位置
E1_462 CHANNEL  ; RK_07 U8_Y 铝壳进料X轴轴存储器操作正被执行序列号
E1_463 CHANNEL  ; RK_07 U8_Y 铝壳进料X轴轴存储器操作正被执行序列号
E1_464 CHANNEL  ; RK_07 U8_Z 铝壳上料移载Y轴轴当前位置
E1_465 CHANNEL  ; RK_07 U8_Z 铝壳上料移载Y轴轴当前位置
E1_466 CHANNEL  ; RK_07 U8_Z 铝壳上料移载Y轴轴存储器操作正被执行序列号
E1_467 CHANNEL  ; RK_07 U8_Z 铝壳上料移载Y轴轴存储器操作正被执行序列号
E1_468 CHANNEL  ; RK_10 U8_U 电池除尘上料X轴轴当前位置
E1_469 CHANNEL  ; RK_10 U8_U 电池除尘上料X轴轴当前位置
E1_47 CHANNEL  ; RK_03 U0_U 电芯上料X轴轴直接操作速度
E1_470 CHANNEL  ; RK_10 U8_U 电池除尘上料X轴轴存储器操作正被执行序列号
E1_471 CHANNEL  ; RK_10 U8_U 电池除尘上料X轴轴存储器操作正被执行序列号
E1_48 CHANNEL  ; RK_03 U0_U 电芯上料X轴轴直接操作加速时间
E1_49 CHANNEL  ; RK_03 U0_U 电芯上料X轴轴直接操作加速时间
E1_5 CHANNEL  ; NC433_0 数据传送读源区域
E1_50 CHANNEL  ; RK_03 U0_U 电芯上料X轴轴直接操作减速时间
E1_5000 CHANNEL  ; #1配方参数（伺服轴）
E1_51 CHANNEL  ; RK_03 U0_U 电芯上料X轴轴直接操作减速时间
E1_52 CHANNEL  ; RK_03 U0_U 电芯上料X轴轴存储器操作序列号
E1_53 CHANNEL  ; RK_03 U0_U 电芯上料X轴轴特殊操作Override
E1_54 CHANNEL  ; RK_03 U0_U 电芯上料X轴轴特殊操作示教地址
E1_55 CHANNEL  ; RK_03 U0_U 电芯上料X轴轴特殊操作预留
E1_56 CHANNEL  ; RK_01 U0_X 电芯来料Y轴轴当前位置
E1_57 CHANNEL  ; RK_01 U0_X 电芯来料Y轴轴当前位置
E1_58 CHANNEL  ; RK_01 U0_X 电芯来料Y轴轴存储器操作正被执行序列号
E1_59 CHANNEL  ; RK_01 U0_X 电芯来料Y轴轴存储器操作正被执行序列号
E1_6 CHANNEL  ; NC433_0 数据传送读目标区域
E1_60 CHANNEL  ; RK_02 U0_Y 电芯进料X轴轴当前位置
E1_61 CHANNEL  ; RK_02 U0_Y 电芯进料X轴轴当前位置
E1_62 CHANNEL  ; RK_02 U0_Y 电芯进料X轴轴存储器操作正被执行序列号
E1_63 CHANNEL  ; RK_02 U0_Y 电芯进料X轴轴存储器操作正被执行序列号
E1_64 CHANNEL  ; RK_02 U0_Z 电芯进料Z轴轴当前位置
E1_65 CHANNEL  ; RK_02 U0_Z 电芯进料Z轴轴当前位置
E1_66 CHANNEL  ; RK_02 U0_Z 电芯进料Z轴轴存储器操作正被执行序列号
E1_67 CHANNEL  ; RK_02 U0_Z 电芯进料Z轴轴存储器操作正被执行序列号
E1_68 CHANNEL  ; RK_03 U0_U 电芯上料X轴轴当前位置
E1_69 CHANNEL  ; RK_03 U0_U 电芯上料X轴轴当前位置
E1_7 CHANNEL  ; NC433_0 数据传送读目标字
E1_70 CHANNEL  ; RK_03 U0_U 电芯上料X轴轴存储器操作正被执行序列号
E1_7000 CHANNEL  ; #2配方参数（伺服轴）
E1_71 CHANNEL  ; RK_03 U0_U 电芯上料X轴轴存储器操作正被执行序列号
E1_8 CHANNEL  ; RK_01 U0_X 电芯来料Y轴轴直接操作位置
E1_9 CHANNEL  ; RK_01 U0_X 电芯来料Y轴轴直接操作位置
E1_9000 CHANNEL  ; #3配方参数（伺服轴）
E2_10000 CHANNEL  ; PC&PLC通讯心跳检测
E2_10001.00 BOOL  ; 设备上电状态
E2_10001.01 BOOL  ; 设备复位状态
E2_10001.02 BOOL  ; 设备自动状态
E2_10001.03 BOOL  ; 设备停止状态
E2_10001.04 BOOL  ; 设备启动状态
E2_10001.05 BOOL  ; 设备待料状态
E2_10001.06 BOOL  ; 设备手动状态
E2_10001.07 BOOL  ; 设备故障状态
E2_10001.08 BOOL  ; 设备急停状态
E2_10001.09 BOOL  ; 设备关电状态
E2_10030 CHANNEL  ; 整机工艺参数变更通知
E2_10031 CHANNEL  ; 整机工艺参数变更确认
E2_10040 CHANNEL  ; RK_02 电芯进料机构MES入站就绪通知
E2_10050 CHANNEL  ; RK_02 电芯进料机构MES入站就绪确认
E2_10060 CHANNEL  ; RK_11 电池除尘上料机构MES出站就绪通知
E2_10061 CHANNEL  ; RK_12 电池上下料机构MES出站就绪通知
E2_10070 CHANNEL  ; RK_11 电池除尘上料机构MES出站就绪确认
E2_10071 CHANNEL  ; RK_12 电池上下料机构MES出站就绪确认
E2_10080 CHANNEL  ; #1出站工位编号（MES）
E2_10081 CHANNEL  ; #2出站工位编号（MES）
E2_10100 CHANNEL  ; RK_02 电芯进料机构MES入站读取条码开始字
E2_10129 CHANNEL  ; RK_02 电芯进料机构MES入站读取条码结束字
E2_10200 CHANNEL  ; #1出站生产数据条码开始字（MES）
E2_10229 CHANNEL  ; #1出站生产数据条码结束字（MES）
E2_10300 CHANNEL  ; #2出站生产数据条码开始字（MES）
E2_10329 CHANNEL  ; #2出站生产数据条码结束字（MES）
E2_10400 CHANNEL  ; #1移载轮廓检测上限（MES）
E2_10401 CHANNEL  ; #1移载轮廓检测上限（MES）
E2_10402 CHANNEL  ; #1移载轮廓检测下限（MES）
E2_10403 CHANNEL  ; #1移载轮廓检测下限（MES）
E2_10404 CHANNEL  ; #2移载轮廓检测上限（MES）
E2_10405 CHANNEL  ; #2移载轮廓检测上限（MES）
E2_10406 CHANNEL  ; #2移载轮廓检测下限（MES）
E2_10407 CHANNEL  ; #2移载轮廓检测下限（MES）
E2_10408 CHANNEL  ; 短路检测参数组号（MES）
E2_10409 CHANNEL  ; 短路检测测试电压（MES）
E2_10410 CHANNEL  ; 短路检测延时时间（MES）
E2_10411 CHANNEL  ; 短路检测测试时间（MES）
E2_10412 CHANNEL  ; 短路检测电阻下限（MES）
E2_10413 CHANNEL  ; 短路检测电阻上限（MES）
E2_10414 CHANNEL  ; 短路检测放电时间（MES）
E2_10500 CHANNEL  ; #1出站生产数据短路检测电阻（MES）
E2_10501 CHANNEL  ; #1出站生产数据短路检测电阻（MES）
E2_10502 CHANNEL  ; #1出站生产数据短路检测电流（MES）
E2_10503 CHANNEL  ; #1出站生产数据短路检测电流（MES）
E2_10504 CHANNEL  ; #1出站生产数据短路检测电压（MES）
E2_10505 CHANNEL  ; #1出站生产数据短路检测结果（MES）
E2_10506 CHANNEL  ; #1出站生产数据工位编号（MES）
E2_10600 CHANNEL  ; #2出站生产数据短路检测电阻（MES）
E2_10601 CHANNEL  ; #2出站生产数据短路检测电阻（MES）
E2_10602 CHANNEL  ; #2出站生产数据短路检测电流（MES）
E2_10603 CHANNEL  ; #2出站生产数据短路检测电流（MES）
E2_10604 CHANNEL  ; #2出站生产数据#1点轮廓检测值（MES）
E2_10605 CHANNEL  ; #2出站生产数据#1点轮廓检测值（MES）
E2_10606 CHANNEL  ; #2出站生产数据#2点轮廓检测值（MES）
E2_10607 CHANNEL  ; #2出站生产数据#2点轮廓检测值（MES）
E2_10608 CHANNEL  ; #2出站生产数据#3点轮廓检测值（MES）
E2_10609 CHANNEL  ; #2出站生产数据#3点轮廓检测值（MES）
E2_10610 CHANNEL  ; #2出站生产数据#4点轮廓检测值（MES）
E2_10611 CHANNEL  ; #2出站生产数据#4点轮廓检测值（MES）
E2_10612 CHANNEL  ; #2出站生产数据短路检测电压（MES）
E2_10613 CHANNEL  ; #2出站生产数据短路检测结果（MES）
E2_10614 CHANNEL  ; #2出站生产数据轮廓检测结果（MES）
E2_10615 CHANNEL  ; #2出站生产数据工位编号（MES）
E2_11000 CHANNEL  ; RK_05 #1入壳压力PV报警值
E2_11002 CHANNEL  ; RK_05 #2入壳压力PV报警值
E2_1201 CHANNEL  ; RK_02 电芯进料机构条码开始字
E2_1230 CHANNEL  ; RK_02 电芯进料机构条码结束字
E2_1300 CHANNEL  ; RK_04 电芯除尘机构数据传递工位编号
E2_1301 CHANNEL  ; RK_03 电芯除尘机构条码开始字
E2_1399 CHANNEL  ; RK_04 电芯除尘机构数据传递结束字
E2_1400 CHANNEL  ; RK_03 电芯上料机构数据传递工位编号
E2_1401 CHANNEL  ; RK_03 电芯上料机构条码开始字
E2_1499 CHANNEL  ; RK_03 电芯上料机构数据传递结束字
E2_1500 CHANNEL  ; RK_05 #1入壳机构电芯数据传递工位编号
E2_1501 CHANNEL  ; RK_05 #1入壳机构电芯条码开始字
E2_1599 CHANNEL  ; RK_05 #1入壳机构电芯数据传递结束字
E2_1600 CHANNEL  ; RK_05 #2入壳机构电芯数据传递工位编号
E2_1601 CHANNEL  ; RK_05 #2入壳机构电芯条码开始字
E2_1699 CHANNEL  ; RK_05 #2入壳机构电芯数据传递结束字
E2_1700 CHANNEL  ; RK_06 电池上下料机构下料夹爪数据传递工位编号
E2_1701 CHANNEL  ; RK_06 电池上下料机构下料夹爪条码开始字
E2_1799 CHANNEL  ; RK_06 电池上下料机构下料夹爪数据传递结束字
E2_1800 CHANNEL  ; RK_09 #1Hipot检测机构数据传递工位编号
E2_1800.02 BOOL  ; #1Hipot检测工位编号标志
E2_1801 CHANNEL  ; RK_09 #1Hipot检测机构条码开始字
E2_1838 CHANNEL  ; RK_09 #1Hipot测试仪测试电阻传递（Float）
E2_1840 CHANNEL  ; RK_09 #1Hipot检测仪测试电流传递（Float）
E2_1842 CHANNEL  ; RK_09 #1Hipot检测仪测试电压传递（Int）
E2_1843 CHANNEL  ; RK_09 #1Hipot检测仪测试结果传递（Int）
E2_1899 CHANNEL  ; RK_09 #1Hipot检测机构数据传递结束字
E2_1900 CHANNEL  ; RK_09 #2Hipot检测机构数据传递工位编号
E2_1900.03 BOOL  ; #2Hipot检测工位编号标志
E2_1901 CHANNEL  ; RK_09 #2Hipot检测机构条码开始字
E2_1938 CHANNEL  ; RK_09 #2Hipot测试仪测试电阻传递（Float）
E2_1940 CHANNEL  ; RK_09 #2Hipot检测仪测试电流传递（Float）
E2_1942 CHANNEL  ; RK_09 #2Hipot检测仪测试电压传递（Int）
E2_1943 CHANNEL  ; RK_09 #2Hipot检测仪测试结果传递（Int）
E2_1999 CHANNEL  ; RK_09 #2Hipot检测机构数据传递结束字
E2_2000 CHANNEL  ; RK_10 电池除尘上料机构数据传递工位编号
E2_2001 CHANNEL  ; RK_10 电池除尘上料机构条码开始字
E2_2038 CHANNEL  ; RK_10 电池除尘上料机构测试电阻传递（Float）
E2_2099 CHANNEL  ; RK_10 电池除尘上料机构数据传递结束字
E2_2100 CHANNEL  ; RK_11 电池除尘机构数据传递工位编号
E2_2101 CHANNEL  ; RK_11 电池除尘机构条码开始字
E2_2138 CHANNEL  ; RK_11 电池除尘机构测试电阻传递（Float）
E2_2199 CHANNEL  ; RK_11 电池除尘机构数据传递结束字
E2_2200 CHANNEL  ; RK_12 预焊上下料机构上料夹爪数据传递工位编号
E2_2201 CHANNEL  ; RK_12 预焊上下料机构上料夹爪条码开始字
E2_2238 CHANNEL  ; RK_12 预焊上下料机构上料夹爪测试电阻传递（Float）
E2_2299 CHANNEL  ; RK_12 预焊上下料机构上料夹爪数据传递结束字
E2_2300 CHANNEL  ; RK_13 #1移载机构数据传递工位编号
E2_2300.04 BOOL  ; #1移载工位编号标志
E2_2301 CHANNEL  ; RK_13 #1移载机构条码开始字
E2_2338 CHANNEL  ; RK_13 #1移载机构测试电阻传递（Float）
E2_2348 CHANNEL  ; RK_13 #1移载机构#1轮廓测量值传递（Float）
E2_2350 CHANNEL  ; RK_13 #1移载机构#2轮廓测量值传递（Float）
E2_2352 CHANNEL  ; RK_13 #1移载机构#3轮廓测量值传递（Float）
E2_2354 CHANNEL  ; RK_13 #1移载机构#4轮廓测量值传递（Float）
E2_2356 CHANNEL  ; RK_13 #1移载机构轮廓测量最终结果传递（Int）
E2_2399 CHANNEL  ; RK_13 #1移载机构数据传递结束字
E2_2400 CHANNEL  ; RK_13 #2移载机构数据传递工位编号
E2_2400.05 BOOL  ; #2移载工位编号标志
E2_2401 CHANNEL  ; RK_13 #2移载机构条码开始字
E2_2438 CHANNEL  ; RK_13 #2移载机构测试电阻传递（Float）
E2_2448 CHANNEL  ; RK_13 #2移载机构#1轮廓测量值传递（Float）
E2_2450 CHANNEL  ; RK_13 #2移载机构#2轮廓测量值传递（Float）
E2_2452 CHANNEL  ; RK_13 #2移载机构#3轮廓测量值传递（Float）
E2_2454 CHANNEL  ; RK_13 #2移载机构#4轮廓测量值传递（Float）
E2_2456 CHANNEL  ; RK_13 #2移载机构轮廓测量最终结果传递（Int）
E2_2499 CHANNEL  ; RK_13 #2移载机构数据传递结束字
E2_2500 CHANNEL  ; RK_12 预焊上下料机构下料夹爪数据传递工位编号
E2_2501 CHANNEL  ; RK_12 预焊上下料机构下料夹爪条码开始字
E2_2538 CHANNEL  ; RK_12 预焊上下料机构下料夹爪测试电阻传递（Float）
E2_2548 CHANNEL  ; RK_12 预焊上下料机构下料夹爪#1轮廓测量值传递（Float）
E2_2550 CHANNEL  ; RK_13 预焊上下料机构下料夹爪#2轮廓测量值传递（Float）
E2_2552 CHANNEL  ; RK_13 预焊上下料机构下料夹爪#3轮廓测量值传递（Float）
E2_2554 CHANNEL  ; RK_13 预焊上下料机构下料夹爪#4轮廓测量值传递（Float）
E2_2556 CHANNEL  ; RK_13 预焊上下料机构下料夹爪轮廓测量最终结果传递（Int）
E2_2599 CHANNEL  ; RK_12 预焊上下料机构下料夹爪数据传递结束字
E2_2700 CHANNEL  ; RK_05 #1入壳机构电池数据传递工位编号
E2_2700.00 BOOL  ; #1入壳工位编号标志
E2_2701 CHANNEL  ; RK_05 #1入壳机构电池条码开始字
E2_2799 CHANNEL  ; RK_05 #1入壳机构电池数据传递结束字
E2_2800 CHANNEL  ; RK_05 #2入壳机构电池数据传递工位编号
E2_2800.01 BOOL  ; #2入壳工位编号标志
E2_2801 CHANNEL  ; RK_05 #2入壳机构电池条码开始字
E2_2899 CHANNEL  ; RK_05 #2入壳机构电池数据传递结束字
E2_5000 CHANNEL  ; 扫码完成信号监控
H0.07 BOOL  ; 电脑屏蔽-HMI
H100.00 BOOL  ; RK_13 U4_U #1移载Y轴回原点记忆
H101.00 BOOL  ; RK_13 #1移载机构有料记忆
H101.01 BOOL  ; RK_13 #1移载机构有OK料记忆
H101.02 BOOL  ; RK_13 #1移载机构有NG料记忆
H101.03 BOOL  ; RK_13 #1移载机构有压装完成料记忆
H101.04 BOOL  ; RK_13 #1移载机构有轮廓检测完成料记忆
H101.05 BOOL  ; RK_13 #1移载机构有轮廓检测#1点完成料记忆
H101.06 BOOL  ; RK_13 #1移载机构有轮廓检测#2点完成料记忆
H101.07 BOOL  ; RK_13 #1移载机构有轮廓检测#3点完成料记忆
H101.08 BOOL  ; RK_13 #1移载机构有轮廓检测#4点完成料记忆
H101.09 BOOL  ; RK_13 #1移载机构有焊接完成料记忆
H101.10 BOOL  ; RK_13 #1移载机构进料记忆
H101.11 BOOL  ; RK_13 #1移载机构出料记忆
H105.00 BOOL  ; RK_13 U6_X #2移载Y轴回原点记忆
H106.00 BOOL  ; RK_13 #2移载机构有料记忆
H106.01 BOOL  ; RK_13 #2移载机构有OK料记忆
H106.02 BOOL  ; RK_13 #2移载机构有NG料记忆
H106.03 BOOL  ; RK_13 #2移载机构有压装完成料记忆
H106.04 BOOL  ; RK_13 #2移载机构有轮廓检测完成料记忆
H106.05 BOOL  ; RK_13 #2移载机构有轮廓检测#1点完成料记忆
H106.06 BOOL  ; RK_13 #2移载机构有轮廓检测#2点完成料记忆
H106.07 BOOL  ; RK_13 #2移载机构有轮廓检测#3点完成料记忆
H106.08 BOOL  ; RK_13 #2移载机构有轮廓检测#4点完成料记忆
H106.09 BOOL  ; RK_13 #2移载机构有焊接完成料记忆
H106.10 BOOL  ; RK_13 #2移载机构进料记忆
H106.11 BOOL  ; RK_13 #2移载机构出料记忆
H10.00 BOOL  ; RK_01 U0_X 电芯来料Y轴回原点记忆
H110.00 BOOL  ; RK_14 #1压装机构压装完成记忆
H110.10 BOOL  ; RK_14 #1压装机构压装中记忆
H111.10 BOOL  ; RK_14 #1压装机构吸盘立真空记忆
H115.00 BOOL  ; RK_14 #2压装机构压装完成记忆
H115.10 BOOL  ; RK_14 #2压装机构压装中记忆
H116.10 BOOL  ; RK_14 #2压装机构吸盘立真空记忆
H11.00 BOOL  ; RK_01 电芯来料机构有料记忆
H121.00 BOOL  ; RK_15 轮廓检测机构#1移载轮廓检测完成记忆
H121.01 BOOL  ; RK_15 轮廓检测机构#2移载轮廓检测完成记忆
H121.02 BOOL  ; RK_15 轮廓检测机构1移载轮廓检测OK记忆
H121.03 BOOL  ; RK_15 轮廓检测机构1移载轮廓检测NG记忆
H121.05 BOOL  ; RK_15 轮廓检测机构轮廓检测#1点完成记忆
H121.06 BOOL  ; RK_15 轮廓检测机构轮廓检测#2点完成记忆
H121.07 BOOL  ; RK_15 轮廓检测机构轮廓检测#3点完成记忆
H121.08 BOOL  ; RK_15 轮廓检测机构轮廓检测#4点完成记忆
H121.10 BOOL  ; RK_15 轮廓检测机构#1移载轮廓检测中记忆
H121.11 BOOL  ; RK_15 轮廓检测机构#2移载轮廓检测中记忆
H121.12 BOOL  ; RK_15 轮廓检测机构2移载轮廓检测OK记忆
H121.13 BOOL  ; RK_15 轮廓检测机构2移载轮廓检测NG记忆
H122.00 BOOL  ; RK_15 轮廓检测机构#1移载#1点测量OK记忆
H122.01 BOOL  ; RK_15 轮廓检测机构#1移载#1点测量NG记忆
H122.02 BOOL  ; RK_15 轮廓检测机构#1移载#2点测量OK记忆
H122.03 BOOL  ; RK_15 轮廓检测机构#1移载#2点测量NG记忆
H122.04 BOOL  ; RK_15 轮廓检测机构#1移载#3点测量OK记忆
H122.05 BOOL  ; RK_15 轮廓检测机构#1移载#3点测量NG记忆
H122.06 BOOL  ; RK_15 轮廓检测机构#1移载#4点测量OK记忆
H122.07 BOOL  ; RK_15 轮廓检测机构#1移载#4点测量NG记忆
H123.00 BOOL  ; RK_15 轮廓检测机构#2移载#1点测量OK记忆
H123.01 BOOL  ; RK_15 轮廓检测机构#2移载#1点测量NG记忆
H123.02 BOOL  ; RK_15 轮廓检测机构#2移载#2点测量OK记忆
H123.03 BOOL  ; RK_15 轮廓检测机构#2移载#2点测量NG记忆
H123.04 BOOL  ; RK_15 轮廓检测机构#2移载#3点测量OK记忆
H123.05 BOOL  ; RK_15 轮廓检测机构#2移载#3点测量NG记忆
H123.06 BOOL  ; RK_15 轮廓检测机构#2移载#4点测量OK记忆
H123.07 BOOL  ; RK_15 轮廓检测机构#2移载#4点测量NG记忆
H125.00 BOOL  ; RK_16 U6_Y 激光焊接X轴回原点记忆
H125.01 BOOL  ; RK_16 U6_Z 激光焊接Z轴回原点记忆
H126.00 BOOL  ; RK_16 焊接机构#1移载激光焊接完成记忆
H126.01 BOOL  ; RK_16 焊接机构#2移载激光焊接完成记忆
H126.10 BOOL  ; RK_16 焊接机构#1移载激光焊接中记忆
H126.11 BOOL  ; RK_16 焊接机构#2移载激光焊接中记忆
H15.00 BOOL  ; RK_02 U0_Y 电芯进料X轴回原点记忆
H15.01 BOOL  ; RK_02 U0_Z 电芯进料Z轴回原点记忆
H16.00 BOOL  ; RK_02 电芯进料机构夹爪有料记忆
H16.01 BOOL  ; RK_02 电芯进料机构夹爪有OK料记忆
H16.02 BOOL  ; RK_02 电芯进料机构夹爪有NG料记忆
H16.03 BOOL  ; RK_02 电芯进料机构扫码完成记忆
H16.04 BOOL  ; RK_02 电芯进料机构夹爪有扫码OK料记忆
H16.05 BOOL  ; RK_02 电芯进料机构夹爪有扫码NG料记忆
H16.06 BOOL  ; RK_02 电芯进料机构MES校验完成记忆
H16.07 BOOL  ; RK_02 电芯进料机构MES校验OK料记忆
H16.08 BOOL  ; RK_02 电芯进料机构MES校验NG料记忆
H17.00 BOOL  ; RK_02 扫码NG拉带放料位有料记忆
H17.10 BOOL  ; RK_02 扫码NG拉带放料位放料中记忆
H20.00 BOOL  ; RK_03 U0_U 电芯上料X轴回原点记忆
H21.00 BOOL  ; RK_03 电芯上料机构夹爪有料记忆
H26.00 BOOL  ; RK_04 电芯除尘机构有料记忆
H26.01 BOOL  ; RK_04 电芯除尘机构除尘完成记忆
H2.00 BOOL  ; 铝壳料盘配方参数屏蔽
H30.00 BOOL  ; RK_05 U2_X #1入壳Y轴回原点记忆
H31.00 BOOL  ; RK_05 #1入壳机构有电池记忆
H31.01 BOOL  ; RK_05 #1入壳机构有电芯记忆
H31.02 BOOL  ; RK_05 #1入壳机构有铝壳记忆
H31.03 BOOL  ; RK_05 #1入壳机构入壳完成记忆
H31.04 BOOL  ; RK_05 #1入壳机构入壳中记忆
H31.06 BOOL  ; RK_05 #1入壳机构Y轴滚轮压紧位记忆
H31.07 BOOL  ; RK_05 #1入壳机构Y轴滚轮松开位记忆
H31.08 BOOL  ; RK_05 #1入壳机构Y轴滚轮入壳位记忆
H31.09 BOOL  ; RK_05 #1入壳机构Y轴电芯定位夹爪松开位记忆
H31.10 BOOL  ; RK_05 #1入壳机构立真空记忆
H35.00 BOOL  ; RK_05 U2_Y #2入壳Y轴回原点记忆
H36.00 BOOL  ; RK_05 #2入壳机构有电池记忆
H36.01 BOOL  ; RK_05 #2入壳机构有电芯记忆
H36.02 BOOL  ; RK_05 #2入壳机构有铝壳记忆
H36.03 BOOL  ; RK_05 #2入壳机构入壳完成记忆
H36.04 BOOL  ; RK_05 #2入壳机构入壳中记忆
H36.06 BOOL  ; RK_05 #2入壳机构Y轴滚轮压紧位记忆
H36.07 BOOL  ; RK_05 #2入壳机构Y轴滚轮松开位记忆
H36.08 BOOL  ; RK_05 #2入壳机构Y轴滚轮入壳位记忆
H36.09 BOOL  ; RK_05 #2入壳机构Y轴电芯定位夹爪松开位记忆
H36.10 BOOL  ; RK_05 #2入壳机构立真空记忆
H40.00 BOOL  ; RK_06 U8_X 电池上下料X轴回原点记忆
H41.00 BOOL  ; RK_06 电池上下料机构上料夹爪有料记忆
H41.01 BOOL  ; RK_06 电池上下料机构下料夹爪有料记忆
H45.00 BOOL  ; RK_07 U8_Y 铝壳进料X轴回原点记忆
H46.00 BOOL  ; RK_07 铝壳进料机构夹爪有料记忆
H46.10 BOOL  ; RK_07 铝壳进料机构吸盘立真空记忆
H47 CHANNEL  ; RK_07 铝壳进料机构取料位序号
H50.00 BOOL  ; RK_07 U8_Z 铝壳上料移载Y轴回原点记忆
H50.10 BOOL  ; RK_07 铝壳上料移载机构吸盘立真空记忆
H51.00 BOOL  ; RK_07 铝壳上料移载机构有料记忆
H51.01 BOOL  ; RK_07 铝壳上料移载机构料盘#1行取料完成记忆
H51.02 BOOL  ; RK_07 铝壳上料移载机构料盘#2行取料完成记忆
H51.03 BOOL  ; RK_07 铝壳上料移载机构料盘#3行取料完成记忆
H51.10 BOOL  ; RK_07 铝壳上料移载机构有托盘记忆
H52 CHANNEL  ; RK_07 铝壳上料移载机构取料位序号
H53.01 BOOL  ; RK_07 铝壳上料移载机构X1Y1有料记忆
H53.02 BOOL  ; RK_07 铝壳上料移载机构X2Y1有料记忆
H53.03 BOOL  ; RK_07 铝壳上料移载机构X3Y1有料记忆
H53.04 BOOL  ; RK_07 铝壳上料移载机构X4Y1有料记忆
H53.05 BOOL  ; RK_07 铝壳上料移载机构X5Y1有料记忆
H53.06 BOOL  ; RK_07 铝壳上料移载机构X1Y2有料记忆
H53.07 BOOL  ; RK_07 铝壳上料移载机构X2Y2有料记忆
H53.08 BOOL  ; RK_07 铝壳上料移载机构X3Y2有料记忆
H53.09 BOOL  ; RK_07 铝壳上料移载机构X4Y2有料记忆
H53.10 BOOL  ; RK_07 铝壳上料移载机构X5Y2有料记忆
H53.11 BOOL  ; RK_07 铝壳上料移载机构X1Y3有料记忆
H53.12 BOOL  ; RK_07 铝壳上料移载机构X2Y3有料记忆
H53.13 BOOL  ; RK_07 铝壳上料移载机构X3Y3有料记忆
H53.14 BOOL  ; RK_07 铝壳上料移载机构X4Y3有料记忆
H53.15 BOOL  ; RK_07 铝壳上料移载机构X5Y3有料记忆
H55.00 BOOL  ; RK_07 #1铝壳上料升降机构手动上料记忆
H56.00 BOOL  ; RK_07 #1铝壳上料升降机构有料记忆
H56.01 BOOL  ; RK_07 #1铝壳上料升降机构自动上料记忆
H60.00 BOOL  ; RK_07 #2铝壳上料升降机构手动上料记忆
H61.00 BOOL  ; RK_07 #2铝壳上料升降机构有料记忆
H61.01 BOOL  ; RK_07 #2铝壳上料升降机构自动上料记忆
H65.00 BOOL  ; RK_07 铝壳托盘下料升降机构手动下料记忆
H66.00 BOOL  ; RK_07 铝壳托盘下料升降机构有料记忆
H71.00 BOOL  ; RK_08 铝壳除尘机构有料记忆
H71.01 BOOL  ; RK_08 铝壳除尘机构除尘完成记忆
H76.00 BOOL  ; RK_09 #1Hipot检测机构有料记忆
H76.01 BOOL  ; RK_09 #1Hipot检测机构有OK料记忆
H76.02 BOOL  ; RK_09 #1Hipot检测机构有NG料记忆
H76.03 BOOL  ; RK_09 #1Hipot检测机构检测完成记忆
H76.04 BOOL  ; RK_09 #1Hipot检测机构检测中记忆
H7.00 BOOL  ; 扫码屏蔽
H7.01 BOOL  ; Hipot检测仪屏蔽
H7.02 BOOL  ; 轮廓仪屏蔽
H7.03 BOOL  ; #1入壳机构屏蔽
H7.04 BOOL  ; #2入壳机构屏蔽
H7.05 BOOL  ; #1Hipot检测屏蔽
H7.06 BOOL  ; #2Hipot检测屏蔽
H7.07 BOOL  ; #1铝壳上料升降机构屏蔽
H7.08 BOOL  ; #2铝壳上料升降机构屏蔽
H7.09 BOOL  ; #1移载机构屏蔽
H7.10 BOOL  ; #2移载机构屏蔽
H7.11 BOOL  ; #1轮廓NG槽屏蔽
H7.12 BOOL  ; #2轮廓NG槽屏蔽
H7.13 BOOL  ; 激光焊机屏蔽
H7.15 BOOL  ; 空跑程序
H81.00 BOOL  ; RK_09 #2Hipot检测机构有料记忆
H81.01 BOOL  ; RK_09 #2Hipot检测机构有OK料记忆
H81.02 BOOL  ; RK_09 #2Hipot检测机构有NG料记忆
H81.03 BOOL  ; RK_09 #2Hipot检测机构检测完成记忆
H81.04 BOOL  ; RK_09 #2Hipot检测机构检测中记忆
H85.00 BOOL  ; RK_10 U8_U 电池除尘上料X轴回原点记忆
H86.00 BOOL  ; RK_10 电池除尘上料机构夹爪有料记忆
H86.01 BOOL  ; RK_10 电池除尘上料机构夹爪有OK料记忆
H86.02 BOOL  ; RK_10 电池除尘上料机构夹爪有NG料记忆
H86.03 BOOL  ; RK_10 电池除尘上料机构MES校验完成记忆
H87.00 BOOL  ; RK_10 Hipot检测NG拉带放料位有料记忆
H87.10 BOOL  ; RK_10 Hipot检测NG拉带放料位放料中记忆
H8.00 BOOL  ; 电芯进料机构重复扫码模式选择（0=使用/1=屏蔽）
H91.00 BOOL  ; RK_11 电池除尘机构有料记忆
H91.01 BOOL  ; RK_11 电池除尘机构除尘完成记忆
H95.00 BOOL  ; RK_12 U4_X 预焊上下料X轴回原点记忆
H95.01 BOOL  ; RK_12 U4_Y 预焊上料Z轴回原点记忆
H95.02 BOOL  ; RK_12 U4_Z 预焊下料Z轴回原点记忆
H96.00 BOOL  ; RK_12 预焊上下料机构上料夹爪有料记忆
H96.01 BOOL  ; RK_12 预焊上下料机构下料夹爪有料记忆
H96.02 BOOL  ; RK_12 预焊上下料机构下料夹爪有OK料记忆
H96.03 BOOL  ; RK_12 预焊上下料机构下料夹爪有NG料记忆
H96.04 BOOL  ; RK_12 预焊上下料机构下料MES校验完成记忆
H96.05 BOOL  ; RK_12 预焊上下料机构下料夹爪有MES校验完成OK料记忆
H96.06 BOOL  ; RK_12 预焊上下料机构下料夹爪有MES校验完成NG料记忆
H97.00 BOOL  ; RK_12 轮廓检测NG槽#1放料位有料记忆
H97.01 BOOL  ; RK_12 轮廓检测NG槽#2放料位有料记忆
H97.02 BOOL  ; RK_12 OK出料拉带放料位有料记忆
H9.00 BOOL  ; 电芯进料X轴&电芯上料X轴伺服限制距离PLC默认值屏蔽（0=PLC默认值有效，1=HMI设定值有效）
H9.01 BOOL  ; 电池除尘上料X轴&预焊上下料X轴伺服限制距离PLC默认值屏蔽（0=PLC默认值有效，1=HMI设定值有效）
T0000 BOOL  ; PLC上电延时100ms
T0001 BOOL  ; 手动模式延时
T0002 BOOL  ; 自动模式延时
T0006 BOOL  ; 复位延时
T0007 BOOL  ; 自动停止完成延时
T0008 BOOL  ; 启动按钮按下1s延时
T0009 BOOL  ; 停止按钮按下延时
T0010 BOOL  ; PLC上电气缸延时输出触发
T0019 BOOL  ; 清料停止完成延时
T0020 BOOL  ; 设备待料状态延时
T0021 BOOL  ; 整机在初始位延时
T0022 BOOL  ; 蜂鸣器屏蔽时间
T0030 BOOL  ; RK_07 #1铝壳上料托盘到位有感应异常提示延时
T0031 BOOL  ; RK_07 #1铝壳上料托盘到位无感应异常提示延时
T0032 BOOL  ; RK_07 #2铝壳上料托盘到位有感应异常提示延时
T0033 BOOL  ; RK_07 #2铝壳上料托盘到位无感应异常提示延时
T0034 BOOL  ; RK_07 #3托盘下料上升到位有感应异常提示延时
T0035 BOOL  ; RK_07 #3托盘下料上升到位无感应异常提示延时
T0036 BOOL  ; RK_07 #3托盘下料下降到位有感应异常提示延时
T0037 BOOL  ; RK_07 #3托盘下料下降到位无感应异常提示延时
T0038 BOOL  ; RK_07 铝壳上料移载托盘到位有感应异常提示延时
T0045 BOOL  ; 扫码枪通信异常
T0046 BOOL  ; 轮廓仪通信异常
T0047 BOOL  ; Hipot检测仪通信异常
T0050 BOOL  ; PC&PLC通讯心跳检测异常延时
T0061 BOOL  ; 参数保存显示延时
T0062 BOOL  ; 参数调出显示延时
T0080 BOOL  ; RK_12 轮廓检测NG料槽#1没料感应延时
T0081 BOOL  ; RK_12 轮廓检测NG料槽#2没料感应延时
T0100 BOOL  ; RK_02 电芯进料机械手夹爪气缸夹紧延时[A]
T0101 BOOL  ; RK_02 电芯进料机械手夹爪气缸张开延时[A]
T0102 BOOL  ; RK_02 电芯进料机械手压紧气缸伸出延时[A]
T0103 BOOL  ; RK_02 电芯进料机械手压紧气缸缩回延时[A]
T0104 BOOL  ; RK_03 电芯上料机械手夹爪气缸夹紧延时[A]
T0105 BOOL  ; RK_03 电芯上料机械手夹爪气缸张开延时[A]
T0106 BOOL  ; RK_03 电芯上料机械手压紧气缸伸出延时[A]
T0107 BOOL  ; RK_03 电芯上料机械手压紧气缸缩回延时[A]
T0108 BOOL  ; RK_03 电芯上料升降气缸下降延时[A]
T0109 BOOL  ; RK_03 电芯上料升降气缸上升延时[A]
T0110 BOOL  ; RK_04 电芯除尘伸缩气缸缩回延时[A]
T0111 BOOL  ; RK_04 电芯除尘伸缩气缸伸出延时[A]
T0112 BOOL  ; RK_05 #1入壳滚轮夹紧气缸伸出延时[A]
T0113 BOOL  ; RK_05 #1入壳滚轮夹紧气缸缩回延时[A]
T0114 BOOL  ; RK_05 #1入壳铝壳定位平台伸缩气缸缩回延时[A]
T0115 BOOL  ; RK_05 #1入壳铝壳定位平台伸缩气缸伸出延时[A]
T0116 BOOL  ; RK_05 #1入壳铝壳定位平台升降气缸上升延时[A]
T0117 BOOL  ; RK_05 #1入壳铝壳定位平台升降气缸下降延时[A]
T0118 BOOL  ; RK_05 #1入壳铝壳定位伸缩气缸缩回延时[A]
T0119 BOOL  ; RK_05 #1入壳铝壳定位伸缩气缸伸出延时[A]
T0120 BOOL  ; RK_05 #1入壳铝壳定位夹爪气缸夹紧延时[A]
T0121 BOOL  ; RK_05 #1入壳铝壳定位夹爪气缸张开延时[A]
T0122 BOOL  ; RK_05 #2入壳滚轮夹紧气缸伸出延时[A]
T0123 BOOL  ; RK_05 #2入壳滚轮夹紧气缸缩回延时[A]
T0124 BOOL  ; RK_05 #2入壳铝壳定位平台伸缩气缸缩回延时[A]
T0125 BOOL  ; RK_05 #2入壳铝壳定位平台伸缩气缸伸出延时[A]
T0126 BOOL  ; RK_05 #2入壳铝壳定位平台升降气缸上升延时[A]
T0127 BOOL  ; RK_05 #2入壳铝壳定位平台升降气缸下降延时[A]
T0128 BOOL  ; RK_05 #2入壳铝壳定位伸缩气缸缩回延时[A]
T0129 BOOL  ; RK_05 #2入壳铝壳定位伸缩气缸伸出延时[A]
T0130 BOOL  ; RK_05 #2入壳铝壳定位夹爪气缸夹紧延时[A]
T0131 BOOL  ; RK_05 #2入壳铝壳定位夹爪气缸张开延时[A]
T0132 BOOL  ; RK_01 U0_X 电芯来料Y轴报警复位延时[A]
T0133 BOOL  ; RK_01 U0_X 电芯来料Y轴使能延时[A]
T0134 BOOL  ; RK_02 U0_Y 电芯进料X轴报警复位延时[A]
T0135 BOOL  ; RK_02 U0_Y 电芯进料X轴使能延时[A]
T0136 BOOL  ; RK_02 U0_Z 电芯进料Z轴报警复位延时[A]
T0137 BOOL  ; RK_02 U0_Z 电芯进料Z轴使能延时[A]
T0138 BOOL  ; RK_03 U0_U 电芯上料X轴报警复位延时[A]
T0139 BOOL  ; RK_03 U0_U 电芯上料X轴使能延时[A]
T0140 BOOL  ; RK_05 U2_X #1入壳Y轴报警复位延时[A]
T0141 BOOL  ; RK_05 U2_X #1入壳Y轴使能延时[A]
T0142 BOOL  ; RK_05 U2_Y #2入壳Y轴报警复位延时[A]
T0143 BOOL  ; RK_05 U2_Y #2入壳Y轴使能延时[A]
T0144 BOOL  ; RK_02 电芯进料Z轴刹车使能延时[A]
T0145 BOOL  ; RK_05 #1入壳定位陶瓷棒夹紧气缸伸出延时[A]
T0146 BOOL  ; RK_05 #1入壳定位陶瓷棒夹紧气缸缩回延时[A]
T0147 BOOL  ; RK_05 #2入壳定位陶瓷棒夹紧气缸伸出延时[A]
T0148 BOOL  ; RK_05 #2入壳定位陶瓷棒夹紧气缸缩回延时[A]
T0149 BOOL  ; RK_04 电芯除尘吹气阀开延时[A]
T0150 BOOL  ; RK_02 扫码NG拉带启动延时[A]
T0151 BOOL  ; RK_05 #1入壳吸盘立真空延时[A]
T0152 BOOL  ; RK_05 #2入壳吸盘立真空延时[A]
T0153 BOOL  ; RK_05 #1入壳吸盘伸缩气缸伸出延时[A]
T0154 BOOL  ; RK_05 #1入壳吸盘伸缩气缸缩回延时[A]
T0155 BOOL  ; RK_05 #2入壳吸盘伸缩气缸伸出延时[A]
T0156 BOOL  ; RK_05 #2入壳吸盘伸缩气缸缩回延时[A]
T0157 BOOL  ; 前端设备对接输出信号（公共）延时[A]
T0158 BOOL  ; 后端设备对接输出信号（公共）延时[A]
T0159 BOOL  ; RK_05 #1入壳电芯定位夹爪气缸伸出延时[A]
T0160 BOOL  ; RK_05 #1入壳电芯定位夹爪气缸缩回延时[A]
T0161 BOOL  ; RK_05 #2入壳电芯定位夹爪气缸伸出延时[A]
T0162 BOOL  ; RK_05 #2入壳电芯定位夹爪气缸缩回延时[A]
T0163 BOOL  ; RK_05 #3入壳电芯定位夹爪气缸伸出延时[A]
T0165 BOOL  ; RK_05 #4入壳电芯定位夹爪气缸伸出延时[A]
T0167 BOOL  ; RK_05 #5入壳电芯定位夹爪气缸伸出延时[A]
T0228 BOOL  ; RK_11 电池除尘旋转伸缩气缸缩回延时[A]
T0229 BOOL  ; RK_11 电池除尘旋转伸缩气缸伸出延时[A]
T0230 BOOL  ; RK_11 电池除尘伸缩气缸伸出延时[A]
T0231 BOOL  ; RK_11 电池除尘伸缩气缸缩回延时[A]
T0232 BOOL  ; RK_11 电池除尘夹爪气缸夹紧延时[A]
T0233 BOOL  ; RK_11 电池除尘夹爪气缸张开延时[A]
T0234 BOOL  ; RK_12 预焊上料机械手夹爪气缸夹紧延时[A]
T0235 BOOL  ; RK_12 预焊上料机械手夹爪气缸张开延时[A]
T0236 BOOL  ; RK_12 预焊下料机械手夹爪气缸夹紧延时[A]
T0237 BOOL  ; RK_12 预焊下料机械手夹爪气缸张开延时[A]
T0238 BOOL  ; RK_13 #1移载升降气缸上升延时[A]
T0239 BOOL  ; RK_13 #1移载升降气缸下降延时[A]
T0240 BOOL  ; RK_13 #1移载定位#1伸缩气缸缩回延时[A]
T0241 BOOL  ; RK_13 #1移载定位#1伸缩气缸伸出延时[A]
T0242 BOOL  ; RK_13 #1移载定位#2伸缩气缸缩回延时[A]
T0243 BOOL  ; RK_13 #1移载定位#2伸缩气缸伸出延时[A]
T0244 BOOL  ; RK_13 #1移载导向#1伸缩气缸伸出延时[A]
T0245 BOOL  ; RK_13 #1移载导向#1伸缩气缸缩回延时[A]
T0246 BOOL  ; RK_13 #1移载导向#2伸缩气缸伸出延时[A]
T0247 BOOL  ; RK_13 #1移载导向#2伸缩气缸缩回延时[A]
T0248 BOOL  ; RK_13 #1移载左右定位伸缩气缸伸出延时[A]
T0249 BOOL  ; RK_13 #1移载左右定位伸缩气缸缩回延时[A]
T0250 BOOL  ; RK_13 #2移载升降气缸上升延时[A]
T0251 BOOL  ; RK_13 #2移载升降气缸下降延时[A]
T0252 BOOL  ; RK_13 #2移载定位#1伸缩气缸缩回延时[A]
T0253 BOOL  ; RK_13 #2移载定位#1伸缩气缸伸出延时[A]
T0254 BOOL  ; RK_13 #2移载定位#2伸缩气缸缩回延时[A]
T0255 BOOL  ; RK_13 #2移载定位#2伸缩气缸伸出延时[A]
T0256 BOOL  ; RK_13 #2移载导向#1伸缩气缸伸出延时[A]
T0257 BOOL  ; RK_13 #2移载导向#1伸缩气缸缩回延时[A]
T0258 BOOL  ; RK_13 #2移载导向#2伸缩气缸伸出延时[A]
T0259 BOOL  ; RK_13 #2移载导向#2伸缩气缸缩回延时[A]
T0260 BOOL  ; RK_13 #2移载左右定位伸缩气缸伸出延时[A]
T0261 BOOL  ; RK_13 #2移载左右定位伸缩气缸缩回延时[A]
T0262 BOOL  ; RK_14 #1压装升降气缸下降延时[A]
T0263 BOOL  ; RK_14 #1压装升降气缸上升延时[A]
T0264 BOOL  ; RK_14 #1压装#1吸盘升降气缸下降延时[A]
T0265 BOOL  ; RK_14 #1压装#1吸盘升降气缸上升延时[A]
T0266 BOOL  ; RK_14 #1压装#2吸盘升降气缸下降延时[A]
T0267 BOOL  ; RK_14 #1压装#2吸盘升降气缸上升延时[A]
T0268 BOOL  ; RK_14 #2压装升降气缸下降延时[A]
T0269 BOOL  ; RK_14 #2压装升降气缸上升延时[A]
T0270 BOOL  ; RK_14 #2压装#1吸盘升降气缸下降延时[A]
T0271 BOOL  ; RK_14 #2压装#1吸盘升降气缸上升延时[A]
T0272 BOOL  ; RK_14 #2压装#2吸盘升降气缸下降延时[A]
T0273 BOOL  ; RK_14 #2压装#2吸盘升降气缸上升延时[A]
T0274 BOOL  ; RK_15 轮廓检测#1伸缩气缸伸出延时[A]
T0275 BOOL  ; RK_15 轮廓检测#1伸缩气缸缩回延时[A]
T0276 BOOL  ; RK_15 轮廓检测#2伸缩气缸伸出延时[A]
T0277 BOOL  ; RK_15 轮廓检测#2伸缩气缸缩回延时[A]
T0278 BOOL  ; RK_12 轮廓检测NG拨料气缸伸出延时[A]
T0279 BOOL  ; RK_12 轮廓检测NG拨料气缸缩回延时[A]
T0280 BOOL  ; RK_11 电池除尘吹气阀开延时[A]
T0281 BOOL  ; 0延时[A]
T0282 BOOL  ; 0延时[A]
T0283 BOOL  ; RK_16 激光焊接触发延时[A]
T0284 BOOL  ; RK_16 PLC急停输出到激光设备延时[A]
T0285 BOOL  ; RK_16 #1移载激光焊任务选择延时[A]
T0286 BOOL  ; RK_16 #2移载激光焊任务选择延时[A]
T0287 BOOL  ; RK_16 集尘器启动延时[A]
T0288 BOOL  ; 0延时[A]
T0289 BOOL  ; 0延时[A]
T0290 BOOL  ; RK_14 #1压装吸盘立真空延时[A]
T0291 BOOL  ; RK_14 #2压装吸盘立真空延时[A]
T0292 BOOL  ; RK_12 U4_X 预焊上下料X轴报警复位延时[A]
T0293 BOOL  ; RK_12 U4_X 预焊上下料X轴使能延时[A]
T0294 BOOL  ; RK_12 U4_Y 预焊上料Z轴报警复位延时[A]
T0295 BOOL  ; RK_12 U4_Y 预焊上料Z轴使能延时[A]
T0296 BOOL  ; RK_12 U4_Z 预焊下料Z轴报警复位延时[A]
T0297 BOOL  ; RK_12 U4_Z 预焊下料Z轴使能延时[A]
T0298 BOOL  ; RK_13 U4_U #1移载Y轴报警复位延时[A]
T0299 BOOL  ; RK_13 U4_U #1移载Y轴使能延时[A]
T0300 BOOL  ; RK_13 U6_X #2移载Y轴报警复位延时[A]
T0301 BOOL  ; RK_13 U6_X #2移载Y轴使能延时[A]
T0302 BOOL  ; RK_16 U6_Y 激光焊接X轴报警复位延时[A]
T0303 BOOL  ; RK_16 U6_Y 激光焊接X轴使能延时[A]
T0304 BOOL  ; RK_16 U6_Z 激光焊接Z轴报警复位延时[A]
T0305 BOOL  ; RK_16 U6_Z 激光焊接Z轴使能延时[A]
T0306 BOOL  ; RK_12 预焊上料Z轴刹车使能延时[A]
T0307 BOOL  ; RK_12 预焊下料Z轴刹车使能延时[A]
T0308 BOOL  ; RK_16 激光焊接Z轴刹车使能延时[A]
T0309 BOOL  ; 0延时[A]
T0310 BOOL  ; 0延时[A]
T0311 BOOL  ; 0延时[A]
T0313 BOOL  ; RK_12 OK出料拉带启动延时[A]
T0314 BOOL  ; 0延时[A]
T0315 BOOL  ; 0延时[A]
T0316 BOOL  ; 0延时[A]
T0317 BOOL  ; RK_07 #1铝壳上料电机刹车使能延时[A]
T0318 BOOL  ; RK_07 #2铝壳上料电机刹车使能延时[A]
T0319 BOOL  ; RK_07 #3托盘下料电机刹车使能延时[A]
T0320 BOOL  ; 三色灯_红（公共）延时[A]
T0321 BOOL  ; 三色灯_绿（公共）延时[A]
T0322 BOOL  ; 三色灯_黄（公共）延时[A]
T0323 BOOL  ; 蜂鸣器（公共）延时[A]
T0324 BOOL  ; RK_06 铝壳上料升降气缸下降延时[A]
T0325 BOOL  ; RK_06 铝壳上料升降气缸上升延时[A]
T0326 BOOL  ; RK_06 电池下料升降气缸下降延时[A]
T0327 BOOL  ; RK_06 电池下料升降气缸上升延时[A]
T0328 BOOL  ; RK_06 铝壳上料夹爪气缸夹紧延时[A]
T0329 BOOL  ; RK_06 铝壳上料夹爪气缸张开延时[A]
T0330 BOOL  ; RK_06 电池下料夹爪气缸夹紧延时[A]
T0331 BOOL  ; RK_06 电池下料夹爪气缸张开延时[A]
T0332 BOOL  ; RK_07 #1铝壳上料车定位升降气缸上升延时[A]
T0333 BOOL  ; RK_07 #1铝壳上料车定位升降气缸下降延时[A]
T0334 BOOL  ; RK_07 #2铝壳上料车定位升降气缸上升延时[A]
T0335 BOOL  ; RK_07 #2铝壳上料车定位升降气缸下降延时[A]
T0336 BOOL  ; RK_07 #3托盘下料车定位升降气缸上升延时[A]
T0337 BOOL  ; RK_07 #3托盘下料车定位升降气缸下降延时[A]
T0338 BOOL  ; RK_07 铝壳进料机械手升降气缸下降延时[A]
T0339 BOOL  ; RK_07 铝壳进料机械手升降气缸上升延时[A]
T0340 BOOL  ; RK_08 铝壳除尘旋转伸缩气缸缩回延时[A]
T0341 BOOL  ; RK_08 铝壳除尘旋转伸缩气缸伸出延时[A]
T0342 BOOL  ; RK_08 铝壳除尘伸缩气缸伸出延时[A]
T0343 BOOL  ; RK_08 铝壳除尘伸缩气缸缩回延时[A]
T0344 BOOL  ; RK_08 铝壳除尘夹爪气缸夹紧延时[A]
T0345 BOOL  ; RK_08 铝壳除尘夹爪气缸张开延时[A]
T0346 BOOL  ; RK_09 #1Hipot测试旋转伸缩气缸伸出延时[A]
T0347 BOOL  ; RK_09 #1Hipot测试旋转伸缩气缸缩回延时[A]
T0348 BOOL  ; RK_09 #1Hipot测试平台伸缩气缸缩回延时[A]
T0349 BOOL  ; RK_09 #1Hipot测试平台伸缩气缸伸出延时[A]
T0350 BOOL  ; RK_09 #1Hipot测试伸缩气缸伸出延时[A]
T0351 BOOL  ; RK_09 #1Hipot测试伸缩气缸缩回延时[A]
T0352 BOOL  ; RK_09 #2Hipot测试旋转伸缩气缸伸出延时[A]
T0353 BOOL  ; RK_09 #2Hipot测试旋转伸缩气缸缩回延时[A]
T0354 BOOL  ; RK_09 #2Hipot测试平台伸缩气缸缩回延时[A]
T0355 BOOL  ; RK_09 #2Hipot测试平台伸缩气缸伸出延时[A]
T0356 BOOL  ; RK_09 #2Hipot测试伸缩气缸伸出延时[A]
T0357 BOOL  ; RK_09 #2Hipot测试伸缩气缸缩回延时[A]
T0358 BOOL  ; RK_10 电池除尘上料机械手升降气缸下降延时[A]
T0359 BOOL  ; RK_10 电池除尘上料机械手升降气缸上升延时[A]
T0360 BOOL  ; RK_10 电池除尘上料机械手夹爪气缸夹紧延时[A]
T0361 BOOL  ; RK_10 电池除尘上料机械手夹爪气缸张开延时[A]
T0362 BOOL  ; RK_06 U8_X 电池上下料X轴报警复位延时[A]
T0363 BOOL  ; RK_06 U8_X 电池上下料X轴使能延时[A]
T0364 BOOL  ; RK_07 U8_Y 铝壳进料X轴报警复位延时[A]
T0365 BOOL  ; RK_07 U8_Y 铝壳进料X轴使能延时[A]
T0366 BOOL  ; RK_07 U8_Z 铝壳上料移载Y轴报警复位延时[A]
T0367 BOOL  ; RK_07 U8_Z 铝壳上料移载Y轴使能延时[A]
T0368 BOOL  ; RK_10 U8_U 电池除尘上料X轴报警复位延时[A]
T0369 BOOL  ; RK_10 U8_U 电池除尘上料X轴使能延时[A]
T0370 BOOL  ; RK_09 Hipot测试仪远程使能（取消）延时[A]
T0371 BOOL  ; RK_07 #1铝壳上料启动指示延时[A]
T0372 BOOL  ; RK_07 #2铝壳上料启动指示延时[A]
T0373 BOOL  ; RK_07 #3托盘下料启动指示延时[A]
T0374 BOOL  ; RK_07 铝壳上料移载吸盘立真空延时[A]
T0375 BOOL  ; RK_07 铝壳进料吸盘立真空延时[A]
T0376 BOOL  ; RK_07 #1铝壳上料电机正转延时[A]
T0377 BOOL  ; RK_07 #1铝壳上料电机反转延时[A]
T0378 BOOL  ; RK_10 Hipot检测NG拉带启动延时[A]
T0379 BOOL  ; RK_08 铝壳除尘吹气阀开延时[A]
T0380 BOOL  ; 0延时[A]
T0381 BOOL  ; RK_07 #2铝壳上料电机正转延时[A]
T0382 BOOL  ; RK_07 #2铝壳上料电机反转延时[A]
T0383 BOOL  ; 启动指示_绿（公共）延时[A]
T0384 BOOL  ; 停止指示_红（公共）延时[A]
T0385 BOOL  ; 复位指示_黄（公共）延时[A]
T0386 BOOL  ; RK_07 #3托盘下料电机正转延时[A]
T0387 BOOL  ; RK_07 #3托盘下料电机反转延时[A]
T0440 BOOL  ; RK_11 电池除尘吹气阀关延时[A]
T0450 BOOL  ; RK_14 #1压装吸盘破真空延时[A]
T0451 BOOL  ; RK_14 #2压装吸盘破真空延时[A]
T0469 BOOL  ; RK_04 电芯除尘吹气阀关延时[A]
T0470 BOOL  ; RK_02 扫码NG拉带停止延时[A]
T0471 BOOL  ; RK_05 #1入壳吸盘破真空延时[A]
T0472 BOOL  ; RK_05 #2入壳吸盘破真空延时[A]
T0473 BOOL  ; RK_12 OK出料拉带停止延时[A]
T0534 BOOL  ; RK_07 铝壳上料移载吸盘破真空延时[A]
T0535 BOOL  ; RK_07 铝壳进料吸盘破真空延时[A]
T0536 BOOL  ; RK_07 #1铝壳上料电机停止延时[A]
T0538 BOOL  ; RK_10 Hipot检测NG拉带停止延时[A]
T0539 BOOL  ; RK_08 铝壳除尘吹气阀关延时[A]
T0541 BOOL  ; RK_07 #2铝壳上料电机停止延时[A]
T0546 BOOL  ; RK_07 #3托盘下料电机停止延时[A]
T0600 BOOL  ; RK_01 U0_X 电芯来料Y轴待料位延时[A]
T0601 BOOL  ; RK_01 U0_X 电芯来料Y轴上料位延时[A]
T0602 BOOL  ; RK_01 U0_X 电芯来料Y轴扫码位延时[A]
T0603 BOOL  ; RK_01 U0_X 电芯来料Y轴下料位延时[A]
T0610 BOOL  ; RK_02 U0_Y 电芯进料X轴待料位延时[A]
T0611 BOOL  ; RK_02 U0_Y 电芯进料X轴取料位延时[A]
T0612 BOOL  ; RK_02 U0_Y 电芯进料X轴扫码OK放料位延时[A]
T0613 BOOL  ; RK_02 U0_Y 电芯进料X轴扫码NG放料位延时[A]
T0620 BOOL  ; RK_02 U0_Z 电芯进料Z轴待料位（扫码）延时[A]
T0621 BOOL  ; RK_02 U0_Z 电芯进料Z轴取料位延时[A]
T0622 BOOL  ; RK_02 U0_Z 电芯进料Z轴扫码OK放料位延时[A]
T0623 BOOL  ; RK_02 U0_Z 电芯进料Z轴扫码NG放料位延时[A]
T0624 BOOL  ; RK_02 U0_Z 电芯进料Z轴扫码位延时[A]
T0630 BOOL  ; RK_03 U0_U 电芯上料X轴待料位延时[A]
T0631 BOOL  ; RK_03 U0_U 电芯上料X轴取料位延时[A]
T0632 BOOL  ; RK_03 U0_U 电芯上料X轴#1入壳放料位延时[A]
T0633 BOOL  ; RK_03 U0_U 电芯上料X轴#2入壳放料位延时[A]
T0640 BOOL  ; RK_05 U2_X #1入壳Y轴待料位延时[A]
T0641 BOOL  ; RK_05 U2_X #1入壳Y轴滚轮压紧位延时[A]
T0642 BOOL  ; RK_05 U2_X #1入壳Y轴滚轮松开位延时[A]
T0643 BOOL  ; RK_05 U2_X #1入壳Y轴入壳位延时[A]
T0644 BOOL  ; RK_05 U2_X #1入壳Y轴电芯定位夹爪松开位延时[A]
T0650 BOOL  ; RK_05 U2_Y #2入壳Y轴待料位延时[A]
T0651 BOOL  ; RK_05 U2_Y #2入壳Y轴滚轮压紧位延时[A]
T0652 BOOL  ; RK_05 U2_Y #2入壳Y轴滚轮松开位延时[A]
T0653 BOOL  ; RK_05 U2_Y #2入壳Y轴入壳位延时[A]
T0654 BOOL  ; RK_05 U2_Y #2入壳Y轴电芯定位夹爪松开位延时[A]
T0660 BOOL  ; RK_12 U4_X 预焊上下料X轴待料位延时[A]
T0661 BOOL  ; RK_12 U4_X 预焊上下料X轴除尘取料位延时[A]
T0662 BOOL  ; RK_12 U4_X 预焊上下料X轴#1移载放料位延时[A]
T0663 BOOL  ; RK_12 U4_X 预焊上下料X轴#2移载放料位延时[A]
T0664 BOOL  ; RK_12 U4_X 预焊上下料X轴#1移载取料位延时[A]
T0665 BOOL  ; RK_12 U4_X 预焊上下料X轴#2移载取料位延时[A]
T0666 BOOL  ; RK_12 U4_X 预焊上下料X轴OK放料位延时[A]
T0667 BOOL  ; RK_12 U4_X 预焊上下料X轴#1NG放料位延时[A]
T0668 BOOL  ; RK_12 U4_X 预焊上下料X轴#2NG放料位延时[A]
T0670 BOOL  ; RK_12 U4_Y 预焊上料Z轴待料位延时[A]
T0671 BOOL  ; RK_12 U4_Y 预焊上料Z轴除尘取料位延时[A]
T0672 BOOL  ; RK_12 U4_Y 预焊上料Z轴#1移载放料位延时[A]
T0673 BOOL  ; RK_12 U4_Y 预焊上料Z轴#2移载放料位延时[A]
T0680 BOOL  ; RK_12 U4_Z 预焊下料Z轴待料位延时[A]
T0681 BOOL  ; RK_12 U4_Z 预焊下料Z轴#1移载取料位延时[A]
T0682 BOOL  ; RK_12 U4_Z 预焊下料Z轴#2移载取料位延时[A]
T0683 BOOL  ; RK_12 U4_Z 预焊下料Z轴OK放料位延时[A]
T0684 BOOL  ; RK_12 U4_Z 预焊下料Z轴#1NG放料位延时[A]
T0685 BOOL  ; RK_12 U4_Z 预焊下料Z轴#2NG放料位延时[A]
T0690 BOOL  ; RK_13 U4_U #1移载Y轴待料位延时[A]
T0691 BOOL  ; RK_13 U4_U #1移载Y轴取放料位延时[A]
T0692 BOOL  ; RK_13 U4_U #1移载Y轴压装位延时[A]
T0693 BOOL  ; RK_13 U4_U #1移载Y轴#1轮廓检测位延时[A]
T0694 BOOL  ; RK_13 U4_U #1移载Y轴#2轮廓检测位延时[A]
T0695 BOOL  ; RK_13 U4_U #1移载Y轴激光焊接位延时[A]
T0700 BOOL  ; RK_13 U6_X #2移载Y轴待料位延时[A]
T0701 BOOL  ; RK_13 U6_X #2移载Y轴取放料位延时[A]
T0702 BOOL  ; RK_13 U6_X #2移载Y轴压装位延时[A]
T0703 BOOL  ; RK_13 U6_X #2移载Y轴#1轮廓检测位延时[A]
T0704 BOOL  ; RK_13 U6_X #2移载Y轴#2轮廓检测位延时[A]
T0705 BOOL  ; RK_13 U6_X #2移载Y轴激光焊接位延时[A]
T0710 BOOL  ; RK_16 U6_Y 激光焊接X轴待机位延时[A]
T0711 BOOL  ; RK_16 U6_Y 激光焊接X轴#1移载焊接位延时[A]
T0712 BOOL  ; RK_16 U6_Y 激光焊接X轴#2移载焊接位延时[A]
T0720 BOOL  ; RK_16 U6_Z 激光焊接Z轴待机位延时[A]
T0721 BOOL  ; RK_16 U6_Z 激光焊接Z轴#1移载焊接位延时[A]
T0722 BOOL  ; RK_16 U6_Z 激光焊接Z轴#2移载焊接位延时[A]
T0730 BOOL  ; RK_06 U8_X 电池上下料X轴待机位延时[A]
T0731 BOOL  ; RK_06 U8_X 电池上下料X轴铝壳除尘取料位延时[A]
T0732 BOOL  ; RK_06 U8_X 电池上下料X轴#1入壳放料位延时[A]
T0733 BOOL  ; RK_06 U8_X 电池上下料X轴#2入壳放料位延时[A]
T0734 BOOL  ; RK_06 U8_X 电池上下料X轴#1入壳取料位延时[A]
T0735 BOOL  ; RK_06 U8_X 电池上下料X轴#2入壳取料位延时[A]
T0736 BOOL  ; RK_06 U8_X 电池上下料X轴#1Hipot检测放料位延时[A]
T0737 BOOL  ; RK_06 U8_X 电池上下料X轴#2Hipot检测放料位延时[A]
T0740 BOOL  ; RK_07 U8_Y 铝壳进料X轴等待位延时[A]
T0741 BOOL  ; RK_07 U8_Y 铝壳进料X轴取料位延时[A]
T0742 BOOL  ; RK_07 U8_Y 铝壳进料X轴放料位延时[A]
T0750 BOOL  ; RK_07 U8_Z 铝壳上料移载Y轴待料位延时[A]
T0751 BOOL  ; RK_07 U8_Z 铝壳上料移载Y轴#1铝壳上料位延时[A]
T0752 BOOL  ; RK_07 U8_Z 铝壳上料移载Y轴#2铝壳上料位延时[A]
T0753 BOOL  ; RK_07 U8_Z 铝壳上料移载Y轴#3铝壳托盘下料位延时[A]
T0754 BOOL  ; RK_07 U8_Z 铝壳上料移载Y轴铝壳取料位延时[A]
T0760 BOOL  ; RK_10 U8_U 电池除尘上料X轴待料位延时[A]
T0761 BOOL  ; RK_10 U8_U 电池除尘上料X轴#1Hipot检测取料位延时[A]
T0762 BOOL  ; RK_10 U8_U 电池除尘上料X轴#2Hipot检测取料位延时[A]
T0763 BOOL  ; RK_10 U8_U 电池除尘上料X轴Hipot OK放料位延时[A]
T0764 BOOL  ; RK_10 U8_U 电池除尘上料X轴Hipot NG放料位延时[A]
T0800 BOOL  ; RK_01 U0_X 电芯来料Y轴待料位感应延时
T0801 BOOL  ; RK_01 U0_X 电芯来料Y轴上料位感应延时
T0802 BOOL  ; RK_01 U0_X 电芯来料Y轴扫码位感应延时
T0803 BOOL  ; RK_01 U0_X 电芯来料Y轴下料位感应延时
T0810 BOOL  ; RK_02 U0_Y 电芯进料X轴待料位感应延时
T0811 BOOL  ; RK_02 U0_Y 电芯进料X轴取料位感应延时
T0812 BOOL  ; RK_02 U0_Y 电芯进料X轴扫码OK放料位感应延时
T0813 BOOL  ; RK_02 U0_Y 电芯进料X轴扫码NG放料位感应延时
T0820 BOOL  ; RK_02 U0_Z 电芯进料Z轴待料位（扫码）感应延时
T0821 BOOL  ; RK_02 U0_Z 电芯进料Z轴取料位感应延时
T0822 BOOL  ; RK_02 U0_Z 电芯进料Z轴扫码OK放料位感应延时
T0823 BOOL  ; RK_02 U0_Z 电芯进料Z轴扫码NG放料位感应延时
T0824 BOOL  ; RK_02 U0_Z 电芯进料Z轴扫码位感应延时
T0830 BOOL  ; RK_03 U0_U 电芯上料X轴待料位感应延时
T0831 BOOL  ; RK_03 U0_U 电芯上料X轴取料位感应延时
T0832 BOOL  ; RK_03 U0_U 电芯上料X轴#1入壳放料位感应延时
T0833 BOOL  ; RK_03 U0_U 电芯上料X轴#2入壳放料位感应延时
T0840 BOOL  ; RK_05 U2_X #1入壳Y轴待料位感应延时
T0841 BOOL  ; RK_05 U2_X #1入壳Y轴滚轮压紧位感应延时
T0842 BOOL  ; RK_05 U2_X #1入壳Y轴滚轮松开位感应延时
T0843 BOOL  ; RK_05 U2_X #1入壳Y轴入壳位感应延时
T0844 BOOL  ; RK_05 U2_X #1入壳Y轴电芯定位夹爪松开位感应延时
T0850 BOOL  ; RK_05 U2_Y #2入壳Y轴待料位感应延时
T0851 BOOL  ; RK_05 U2_Y #2入壳Y轴滚轮压紧位感应延时
T0852 BOOL  ; RK_05 U2_Y #2入壳Y轴滚轮松开位感应延时
T0853 BOOL  ; RK_05 U2_Y #2入壳Y轴入壳位感应延时
T0854 BOOL  ; RK_05 U2_Y #2入壳Y轴电芯定位夹爪松开位感应延时
T0860 BOOL  ; RK_12 U4_X 预焊上下料X轴待料位感应延时
T0861 BOOL  ; RK_12 U4_X 预焊上下料X轴除尘取料位感应延时
T0862 BOOL  ; RK_12 U4_X 预焊上下料X轴#1移载放料位感应延时
T0863 BOOL  ; RK_12 U4_X 预焊上下料X轴#2移载放料位感应延时
T0864 BOOL  ; RK_12 U4_X 预焊上下料X轴#1移载取料位感应延时
T0865 BOOL  ; RK_12 U4_X 预焊上下料X轴#2移载取料位感应延时
T0866 BOOL  ; RK_12 U4_X 预焊上下料X轴OK放料位感应延时
T0867 BOOL  ; RK_12 U4_X 预焊上下料X轴#1NG放料位感应延时
T0868 BOOL  ; RK_12 U4_X 预焊上下料X轴#2NG放料位感应延时
T0870 BOOL  ; RK_12 U4_Y 预焊上料Z轴待料位感应延时
T0871 BOOL  ; RK_12 U4_Y 预焊上料Z轴除尘取料位感应延时
T0872 BOOL  ; RK_12 U4_Y 预焊上料Z轴#1移载放料位感应延时
T0873 BOOL  ; RK_12 U4_Y 预焊上料Z轴#2移载放料位感应延时
T0880 BOOL  ; RK_12 U4_Z 预焊下料Z轴待料位感应延时
T0881 BOOL  ; RK_12 U4_Z 预焊下料Z轴#1移载取料位感应延时
T0882 BOOL  ; RK_12 U4_Z 预焊下料Z轴#2移载取料位感应延时
T0883 BOOL  ; RK_12 U4_Z 预焊下料Z轴OK放料位感应延时
T0884 BOOL  ; RK_12 U4_Z 预焊下料Z轴#1NG放料位感应延时
T0885 BOOL  ; RK_12 U4_Z 预焊下料Z轴#2NG放料位感应延时
T0890 BOOL  ; RK_13 U4_U #1移载Y轴待料位感应延时
T0891 BOOL  ; RK_13 U4_U #1移载Y轴取放料位感应延时
T0892 BOOL  ; RK_13 U4_U #1移载Y轴压装位感应延时
T0893 BOOL  ; RK_13 U4_U #1移载Y轴#1轮廓检测位感应延时
T0894 BOOL  ; RK_13 U4_U #1移载Y轴#2轮廓检测位感应延时
T0895 BOOL  ; RK_13 U4_U #1移载Y轴激光焊接位感应延时
T0900 BOOL  ; RK_13 U6_X #2移载Y轴待料位感应延时
T0901 BOOL  ; RK_13 U6_X #2移载Y轴取放料位感应延时
T0902 BOOL  ; RK_13 U6_X #2移载Y轴压装位感应延时
T0903 BOOL  ; RK_13 U6_X #2移载Y轴#1轮廓检测位感应延时
T0904 BOOL  ; RK_13 U6_X #2移载Y轴#2轮廓检测位感应延时
T0905 BOOL  ; RK_13 U6_X #2移载Y轴激光焊接位感应延时
T0910 BOOL  ; RK_16 U6_Y 激光焊接X轴待机位感应延时
T0911 BOOL  ; RK_16 U6_Y 激光焊接X轴#1移载焊接位感应延时
T0912 BOOL  ; RK_16 U6_Y 激光焊接X轴#2移载焊接位感应延时
T0920 BOOL  ; RK_16 U6_Z 激光焊接Z轴待机位感应延时
T0921 BOOL  ; RK_16 U6_Z 激光焊接Z轴#1移载焊接位感应延时
T0922 BOOL  ; RK_16 U6_Z 激光焊接Z轴#2移载焊接位感应延时
T0930 BOOL  ; RK_06 U8_X 电池上下料X轴待机位感应延时
T0931 BOOL  ; RK_06 U8_X 电池上下料X轴铝壳除尘取料位感应延时
T0932 BOOL  ; RK_06 U8_X 电池上下料X轴#1入壳放料位感应延时
T0933 BOOL  ; RK_06 U8_X 电池上下料X轴#2入壳放料位感应延时
T0934 BOOL  ; RK_06 U8_X 电池上下料X轴#1入壳取料位感应延时
T0935 BOOL  ; RK_06 U8_X 电池上下料X轴#2入壳取料位感应延时
T0936 BOOL  ; RK_06 U8_X 电池上下料X轴#1Hipot检测放料位感应延时
T0937 BOOL  ; RK_06 U8_X 电池上下料X轴#2Hipot检测放料位感应延时
T0940 BOOL  ; RK_07 U8_Y 铝壳进料X轴等待位感应延时
T0941 BOOL  ; RK_07 U8_Y 铝壳进料X轴取料位感应延时
T0942 BOOL  ; RK_07 U8_Y 铝壳进料X轴放料位感应延时
T0950 BOOL  ; RK_07 U8_Z 铝壳上料移载Y轴待料位感应延时
T0951 BOOL  ; RK_07 U8_Z 铝壳上料移载Y轴#1铝壳上料位感应延时
T0952 BOOL  ; RK_07 U8_Z 铝壳上料移载Y轴#2铝壳上料位感应延时
T0953 BOOL  ; RK_07 U8_Z 铝壳上料移载Y轴#3铝壳托盘下料位感应延时
T0954 BOOL  ; RK_07 U8_Z 铝壳上料移载Y轴铝壳取料位感应延时
T0960 BOOL  ; RK_10 U8_U 电池除尘上料X轴待料位感应延时
T0961 BOOL  ; RK_10 U8_U 电池除尘上料X轴#1Hipot检测取料位感应延时
T0962 BOOL  ; RK_10 U8_U 电池除尘上料X轴#2Hipot检测取料位感应延时
T0963 BOOL  ; RK_10 U8_U 电池除尘上料X轴Hipot OK放料位感应延时
T0964 BOOL  ; RK_10 U8_U 电池除尘上料X轴Hipot NG放料位感应延时
T1000 BOOL  ; RK_02 电芯进料机械手夹爪气缸夹紧位感应延时[0000.00]
T1001 BOOL  ; RK_02 电芯进料机械手夹爪气缸张开位感应延时[0000.01]
T1002 BOOL  ; RK_02 电芯进料机械手#1压紧气缸松开位感应延时[0000.02]
T1003 BOOL  ; RK_02 电芯进料机械手#2压紧气缸松开位感应延时[0000.03]
T1004 BOOL  ; RK_03 电芯上料机械手夹爪气缸夹紧位感应延时[0000.04]
T1005 BOOL  ; RK_03 电芯上料机械手夹爪气缸张开位感应延时[0000.05]
T1006 BOOL  ; RK_03 电芯上料机械手#1压紧气缸松开位感应延时[0000.06]
T1007 BOOL  ; RK_03 电芯上料机械手#2压紧气缸松开位感应延时[0000.07]
T1008 BOOL  ; RK_03 电芯上料升降气缸下降位感应延时[0000.08]
T1009 BOOL  ; RK_03 电芯上料升降气缸上升位感应延时[0000.09]
T1010 BOOL  ; RK_04 电芯除尘伸缩气缸缩回位感应延时[0000.10]
T1011 BOOL  ; RK_04 电芯除尘伸缩气缸伸出位感应延时[0000.11]
T1012 BOOL  ; RK_05 #1入壳滚轮夹紧气缸夹紧位感应延时[0000.12]
T1013 BOOL  ; RK_05 #1入壳滚轮夹紧气缸松开位感应延时[0000.13]
T1014 BOOL  ; RK_05 #1入壳铝壳定位平台伸缩气缸缩回位感应延时[0000.14]
T1015 BOOL  ; RK_05 #1入壳铝壳定位平台伸缩气缸伸出位感应延时[0000.15]
T1016 BOOL  ; RK_05 #1入壳铝壳定位平台升降气缸上升位感应延时[0001.00]
T1017 BOOL  ; RK_05 #1入壳铝壳定位平台升降气缸下降位感应延时[0001.01]
T1018 BOOL  ; RK_05 #1入壳铝壳定位伸缩气缸缩回位感应延时[0001.02]
T1019 BOOL  ; RK_05 #1入壳铝壳定位伸缩气缸伸出位感应延时[0001.03]
T1020 BOOL  ; RK_05 #1入壳铝壳定位夹爪气缸夹紧位感应延时[0001.04]
T1021 BOOL  ; RK_05 #1入壳铝壳定位夹爪气缸张开位感应延时[0001.05]
T1022 BOOL  ; RK_05 #2入壳滚轮夹紧气缸夹紧位感应延时[0001.06]
T1023 BOOL  ; RK_05 #2入壳滚轮夹紧气缸松开位感应延时[0001.07]
T1024 BOOL  ; RK_05 #2入壳铝壳定位平台伸缩气缸缩回位感应延时[0001.08]
T1025 BOOL  ; RK_05 #2入壳铝壳定位平台伸缩气缸伸出位感应延时[0001.09]
T1026 BOOL  ; RK_05 #2入壳铝壳定位平台升降气缸上升位感应延时[0001.10]
T1027 BOOL  ; RK_05 #2入壳铝壳定位平台升降气缸下降位感应延时[0001.11]
T1028 BOOL  ; RK_05 #2入壳铝壳定位伸缩气缸缩回位感应延时[0001.12]
T1029 BOOL  ; RK_05 #2入壳铝壳定位伸缩气缸伸出位感应延时[0001.13]
T1030 BOOL  ; RK_05 #2入壳铝壳定位夹爪气缸夹紧位感应延时[0001.14]
T1031 BOOL  ; RK_05 #2入壳铝壳定位夹爪气缸张开位感应延时[0001.15]
T1032 BOOL  ; RK_01 U0_X 电芯来料Y轴报警信号感应延时[0002.00]
T1033 BOOL  ; RK_01 U0_X 电芯来料Y轴准备好了信号感应延时[0002.01]
T1034 BOOL  ; RK_02 U0_Y 电芯进料X轴报警信号感应延时[0002.02]
T1035 BOOL  ; RK_02 U0_Y 电芯进料X轴准备好了信号感应延时[0002.03]
T1036 BOOL  ; RK_02 U0_Z 电芯进料Z轴报警信号感应延时[0002.04]
T1037 BOOL  ; RK_02 U0_Z 电芯进料Z轴准备好了信号感应延时[0002.05]
T1038 BOOL  ; RK_03 U0_U 电芯上料X轴报警信号感应延时[0002.06]
T1039 BOOL  ; RK_03 U0_U 电芯上料X轴准备好了信号感应延时[0002.07]
T1040 BOOL  ; RK_05 U2_X #1入壳Y轴报警信号感应延时[0002.08]
T1041 BOOL  ; RK_05 U2_X #1入壳Y轴准备好了信号感应延时[0002.09]
T1042 BOOL  ; RK_05 U2_Y #2入壳Y轴报警信号感应延时[0002.10]
T1043 BOOL  ; RK_05 U2_Y #2入壳Y轴准备好了信号感应延时[0002.11]
T1044 BOOL  ; 0感应延时[0002.12]
T1045 BOOL  ; RK_05 #1入壳定位陶瓷棒上#1夹紧气缸伸出位感应延时[0002.13]
T1046 BOOL  ; RK_05 #1入壳定位陶瓷棒上#2夹紧气缸伸出位感应延时[0002.14]
T1047 BOOL  ; RK_05 #1入壳定位陶瓷棒下#1夹紧气缸伸出位感应延时[0002.15]
T1048 BOOL  ; RK_05 #1入壳定位陶瓷棒下#2夹紧气缸伸出位感应延时[0003.00]
T1049 BOOL  ; RK_05 #1入壳定位陶瓷棒上#1夹紧气缸缩回位感应延时[0003.01]
T1050 BOOL  ; RK_05 #1入壳定位陶瓷棒上#2夹紧气缸缩回位感应延时[0003.02]
T1051 BOOL  ; RK_05 #1入壳定位陶瓷棒下#1夹紧气缸缩回位感应延时[0003.03]
T1052 BOOL  ; RK_05 #1入壳定位陶瓷棒下#2夹紧气缸缩回位感应延时[0003.04]
T1053 BOOL  ; RK_05 #1入壳吸盘上#1伸缩气缸缩回位感应延时[0003.05]
T1054 BOOL  ; RK_05 #1入壳吸盘上#2伸缩气缸缩回位感应延时[0003.06]
T1055 BOOL  ; RK_05 #1入壳吸盘上#3伸缩气缸缩回位感应延时[0003.07]
T1056 BOOL  ; RK_05 #1入壳吸盘下#1伸缩气缸缩回位感应延时[0003.08]
T1057 BOOL  ; RK_05 #1入壳吸盘下#2伸缩气缸缩回位感应延时[0003.09]
T1058 BOOL  ; RK_05 #1入壳吸盘下#3伸缩气缸缩回位感应延时[0003.10]
T1059 BOOL  ; RK_05 #1入壳电芯#1定位夹爪气缸松开位感应延时[0003.11]
T1060 BOOL  ; RK_05 #1入壳电芯#2定位夹爪气缸松开位感应延时[0003.12]
T1061 BOOL  ; RK_05 #1入壳电芯#1定位夹爪气缸夹紧位感应延时[0003.13]
T1062 BOOL  ; RK_05 #1入壳电芯#2定位夹爪气缸夹紧位感应延时[0003.14]
T1063 BOOL  ; RK_05 #2入壳定位陶瓷棒上#1夹紧气缸伸出位感应延时[0003.15]
T1064 BOOL  ; RK_05 #2入壳定位陶瓷棒上#2夹紧气缸伸出位感应延时[0004.00]
T1065 BOOL  ; RK_05 #2入壳定位陶瓷棒下#1夹紧气缸伸出位感应延时[0004.01]
T1066 BOOL  ; RK_05 #2入壳定位陶瓷棒下#2夹紧气缸伸出位感应延时[0004.02]
T1067 BOOL  ; RK_05 #2入壳定位陶瓷棒上#1夹紧气缸缩回位感应延时[0004.03]
T1068 BOOL  ; RK_05 #2入壳定位陶瓷棒上#2夹紧气缸缩回位感应延时[0004.04]
T1069 BOOL  ; RK_05 #2入壳定位陶瓷棒下#1夹紧气缸缩回位感应延时[0004.05]
T1070 BOOL  ; RK_05 #2入壳定位陶瓷棒下#2夹紧气缸缩回位感应延时[0004.06]
T1071 BOOL  ; RK_05 #2入壳吸盘上#1伸缩气缸缩回位感应延时[0004.07]
T1072 BOOL  ; RK_05 #2入壳吸盘上#2伸缩气缸缩回位感应延时[0004.08]
T1073 BOOL  ; RK_05 #2入壳吸盘上#3伸缩气缸缩回位感应延时[0004.09]
T1074 BOOL  ; RK_05 #2入壳吸盘下#1伸缩气缸缩回位感应延时[0004.10]
T1075 BOOL  ; RK_05 #2入壳吸盘下#2伸缩气缸缩回位感应延时[0004.11]
T1076 BOOL  ; RK_05 #2入壳吸盘下#3伸缩气缸缩回位感应延时[0004.12]
T1077 BOOL  ; RK_05 #2入壳电芯#1定位夹爪气缸松开位感应延时[0004.13]
T1078 BOOL  ; RK_05 #2入壳电芯#2定位夹爪气缸松开位感应延时[0004.14]
T1079 BOOL  ; RK_05 #2入壳电芯#1定位夹爪气缸夹紧位感应延时[0004.15]
T1080 BOOL  ; RK_05 #2入壳电芯#2定位夹爪气缸夹紧位感应延时[0005.00]
T1081 BOOL  ; RK_01 电芯来料有料感应感应延时[0005.01]
T1082 BOOL  ; RK_02 电芯进料机械手夹爪柔性报警感应延时[0005.02]
T1083 BOOL  ; RK_03 电芯上料机械手夹爪柔性报警感应延时[0005.03]
T1084 BOOL  ; RK_04 电芯除尘有料感应感应延时[0005.04]
T1085 BOOL  ; RK_02 扫码NG拉带有料感应#1感应延时[0005.05]
T1086 BOOL  ; RK_02 扫码NG拉带有料感应#2感应延时[0005.06]
T1087 BOOL  ; RK_02 扫码NG拉带料满感应感应延时[0005.07]
T1088 BOOL  ; RK_05 #1入壳电芯有料感应感应延时[0005.08]
T1089 BOOL  ; RK_05 #1入壳铝壳有料感应感应延时[0005.09]
T1090 BOOL  ; RK_05 #2入壳电芯有料感应感应延时[0005.10]
T1091 BOOL  ; RK_05 #2入壳铝壳有料感应感应延时[0005.11]
T1092 BOOL  ; RK_05 #1入壳吸盘真空感应延时[0005.12]
T1093 BOOL  ; RK_05 #2入壳吸盘真空感应延时[0005.13]
T1094 BOOL  ; 前端设备对接输入信号（公共）感应延时[0005.14]
T1095 BOOL  ; 后端设备对接输入信号（公共）感应延时[0005.15]
T1096 BOOL  ; 小屏插入信号（公共）感应延时[0006.00]
T1097 BOOL  ; NC433模块DC5V电源信号（公共）感应延时[0006.01]
T1098 BOOL  ; DC24V伺服刹车电源信号（公共）感应延时[0006.02]
T1099 BOOL  ; 出料端急停（公共）感应延时[0006.03]
T1100 BOOL  ; 小移动屏急停（公共）感应延时[0006.04]
T1101 BOOL  ; A机架#1门磁（公共）感应延时[0006.05]
T1102 BOOL  ; A机架#2门磁（公共）感应延时[0006.06]
T1103 BOOL  ; A机架#3门磁（公共）感应延时[0006.07]
T1104 BOOL  ; A机架#4门磁（公共）感应延时[0006.08]
T1105 BOOL  ; A机架#5门磁（公共）感应延时[0006.09]
T1106 BOOL  ; A机架#6门磁（公共）感应延时[0006.10]
T1107 BOOL  ; A机架#7门磁（公共）感应延时[0006.11]
T1108 BOOL  ; A机架#8门磁（公共）感应延时[0006.12]
T1109 BOOL  ; A机架#9门磁（公共）感应延时[0006.13]
T1110 BOOL  ; RK_01 电芯来料上料位有料感应感应延时[0006.14]
T1111 BOOL  ; 0感应延时[0006.15]
T1112 BOOL  ; 0感应延时[0007.00]
T1113 BOOL  ; 0感应延时[0007.01]
T1114 BOOL  ; 0感应延时[0007.02]
T1115 BOOL  ; 0感应延时[0007.03]
T1116 BOOL  ; 0感应延时[0007.04]
T1117 BOOL  ; 0感应延时[0007.05]
T1118 BOOL  ; 0感应延时[0007.06]
T1119 BOOL  ; 0感应延时[0007.07]
T1120 BOOL  ; 0感应延时[0007.08]
T1121 BOOL  ; 0感应延时[0007.09]
T1122 BOOL  ; 0感应延时[0007.10]
T1123 BOOL  ; 0感应延时[0007.11]
T1124 BOOL  ; 0感应延时[0007.12]
T1125 BOOL  ; 0感应延时[0007.13]
T1126 BOOL  ; 0感应延时[0007.14]
T1127 BOOL  ; 0感应延时[0007.15]
T1128 BOOL  ; RK_11 电池除尘旋转伸缩气缸到位感应延时[0008.00]
T1129 BOOL  ; RK_11 电池除尘旋转伸缩气缸原位感应延时[0008.01]
T1130 BOOL  ; RK_11 电池除尘伸缩气缸伸出位感应延时[0008.02]
T1131 BOOL  ; RK_11 电池除尘伸缩气缸缩回位感应延时[0008.03]
T1132 BOOL  ; RK_11 电池除尘夹爪气缸夹紧位感应延时[0008.04]
T1133 BOOL  ; RK_11 电池除尘夹爪气缸张开位感应延时[0008.05]
T1134 BOOL  ; RK_12 预焊上料机械手夹爪气缸夹紧位感应延时[0008.06]
T1135 BOOL  ; RK_12 预焊上料机械手夹爪气缸张开位感应延时[0008.07]
T1136 BOOL  ; RK_12 预焊下料机械手夹爪气缸夹紧位感应延时[0008.08]
T1137 BOOL  ; RK_12 预焊下料机械手夹爪气缸张开位感应延时[0008.09]
T1138 BOOL  ; RK_13 #1移载升降气缸上升位感应延时[0008.10]
T1139 BOOL  ; RK_13 #1移载升降气缸下降位感应延时[0008.11]
T1140 BOOL  ; RK_13 #1移载定位#1伸缩气缸缩回位感应延时[0008.12]
T1141 BOOL  ; RK_13 #1移载定位#1伸缩气缸伸出位感应延时[0008.13]
T1142 BOOL  ; RK_13 #1移载定位#2伸缩气缸缩回位感应延时[0008.14]
T1143 BOOL  ; RK_13 #1移载定位#2伸缩气缸伸出位感应延时[0008.15]
T1144 BOOL  ; RK_13 #1移载导向#1伸缩气缸伸出位感应延时[0009.00]
T1145 BOOL  ; RK_13 #1移载导向#1伸缩气缸缩回位感应延时[0009.01]
T1146 BOOL  ; RK_13 #1移载导向#2伸缩气缸伸出位感应延时[0009.02]
T1147 BOOL  ; RK_13 #1移载导向#2伸缩气缸缩回位感应延时[0009.03]
T1148 BOOL  ; RK_13 #1移载左右定位伸缩气缸伸出位感应延时[0009.04]
T1149 BOOL  ; RK_13 #1移载左右定位伸缩气缸缩回位感应延时[0009.05]
T1150 BOOL  ; RK_13 #2移载升降气缸上升位感应延时[0009.06]
T1151 BOOL  ; RK_13 #2移载升降气缸下降位感应延时[0009.07]
T1152 BOOL  ; RK_13 #2移载定位#1伸缩气缸缩回位感应延时[0009.08]
T1153 BOOL  ; RK_13 #2移载定位#1伸缩气缸伸出位感应延时[0009.09]
T1154 BOOL  ; RK_13 #2移载定位#2伸缩气缸缩回位感应延时[0009.10]
T1155 BOOL  ; RK_13 #2移载定位#2伸缩气缸伸出位感应延时[0009.11]
T1156 BOOL  ; RK_13 #2移载导向#1伸缩气缸伸出位感应延时[0009.12]
T1157 BOOL  ; RK_13 #2移载导向#1伸缩气缸缩回位感应延时[0009.13]
T1158 BOOL  ; RK_13 #2移载导向#2伸缩气缸伸出位感应延时[0009.14]
T1159 BOOL  ; RK_13 #2移载导向#2伸缩气缸缩回位感应延时[0009.15]
T1160 BOOL  ; RK_13 #2移载左右定位伸缩气缸伸出位感应延时[0010.00]
T1161 BOOL  ; RK_13 #2移载左右定位伸缩气缸缩回位感应延时[0010.01]
T1162 BOOL  ; RK_14 #1压装升降气缸下降位感应延时[0010.02]
T1163 BOOL  ; RK_14 #1压装升降气缸上升位感应延时[0010.03]
T1164 BOOL  ; RK_14 #1压装#1吸盘升降气缸下降位感应延时[0010.04]
T1165 BOOL  ; RK_14 #1压装#1吸盘升降气缸上升位感应延时[0010.05]
T1166 BOOL  ; RK_14 #1压装#2吸盘升降气缸下降位感应延时[0010.06]
T1167 BOOL  ; RK_14 #1压装#2吸盘升降气缸上升位感应延时[0010.07]
T1168 BOOL  ; RK_14 #2压装升降气缸下降位感应延时[0010.08]
T1169 BOOL  ; RK_14 #2压装升降气缸上升位感应延时[0010.09]
T1170 BOOL  ; RK_14 #2压装#1吸盘升降气缸下降位感应延时[0010.10]
T1171 BOOL  ; RK_14 #2压装#1吸盘升降气缸上升位感应延时[0010.11]
T1172 BOOL  ; RK_14 #2压装#2吸盘升降气缸下降位感应延时[0010.12]
T1173 BOOL  ; RK_14 #2压装#2吸盘升降气缸上升位感应延时[0010.13]
T1174 BOOL  ; RK_15 轮廓检测#1伸缩气缸伸出位感应延时[0010.14]
T1175 BOOL  ; RK_15 轮廓检测#1伸缩气缸缩回位感应延时[0010.15]
T1176 BOOL  ; RK_15 轮廓检测#2伸缩气缸伸出位感应延时[0011.00]
T1177 BOOL  ; RK_15 轮廓检测#2伸缩气缸缩回位感应延时[0011.01]
T1178 BOOL  ; RK_12 轮廓检测NG拨料气缸伸出位感应延时[0011.02]
T1179 BOOL  ; RK_12 轮廓检测NG拨料气缸缩回位感应延时[0011.03]
T1180 BOOL  ; RK_11 电池除尘有料感应感应延时[0011.04]
T1181 BOOL  ; RK_12 预焊上料机械手夹爪柔性报警感应延时[0011.05]
T1182 BOOL  ; RK_12 预焊下料机械手夹爪柔性报警感应延时[0011.06]
T1183 BOOL  ; RK_16 激光焊接完成信号感应延时[0011.07]
T1184 BOOL  ; RK_16 激光焊机故障信号感应延时[0011.08]
T1185 BOOL  ; RK_13 #1移载电池顶盖超高检测感应延时[0011.09]
T1186 BOOL  ; RK_16 激光焊机急停信号感应延时[0011.10]
T1187 BOOL  ; RK_13 #2移载电池顶盖超高检测感应延时[0011.09]
T1188 BOOL  ; RK_13 #1移载有料感应延时[0011.12]
T1189 BOOL  ; RK_13 #2移载有料感应延时[0011.13]
T1190 BOOL  ; RK_14 #1压装吸盘真空感应延时[0011.14]
T1191 BOOL  ; RK_14 #2压装吸盘真空感应延时[0011.15]
T1192 BOOL  ; RK_12 U4_X 预焊上下料X轴报警信号感应延时[0012.00]
T1193 BOOL  ; RK_12 U4_X 预焊上下料X轴准备好了信号感应延时[0012.01]
T1194 BOOL  ; RK_12 U4_Y 预焊上料Z轴报警信号感应延时[0012.02]
T1195 BOOL  ; RK_12 U4_Y 预焊上料Z轴准备好了信号感应延时[0012.03]
T1196 BOOL  ; RK_12 U4_Z 预焊下料Z轴报警信号感应延时[0012.04]
T1197 BOOL  ; RK_12 U4_Z 预焊下料Z轴准备好了信号感应延时[0012.05]
T1198 BOOL  ; RK_13 U4_U #1移载Y轴报警信号感应延时[0012.06]
T1199 BOOL  ; RK_13 U4_U #1移载Y轴准备好了信号感应延时[0012.07]
T1200 BOOL  ; RK_13 U6_X #2移载Y轴报警信号感应延时[0012.08]
T1201 BOOL  ; RK_13 U6_X #2移载Y轴准备好了信号感应延时[0012.09]
T1202 BOOL  ; RK_16 U6_Y 激光焊接X轴报警信号感应延时[0012.10]
T1203 BOOL  ; RK_16 U6_Y 激光焊接X轴准备好了信号感应延时[0012.11]
T1204 BOOL  ; RK_16 U6_Z 激光焊接Z轴报警信号感应延时[0012.12]
T1205 BOOL  ; RK_16 U6_Z 激光焊接Z轴准备好了信号感应延时[0012.13]
T1206 BOOL  ; 0感应延时[0012.14]
T1207 BOOL  ; 0感应延时[0012.15]
T1208 BOOL  ; 0感应延时[0013.00]
T1209 BOOL  ; RK_12 轮廓检测NG料槽#1有料感应感应延时[0013.01]
T1210 BOOL  ; RK_12 轮廓检测NG料槽#1料满感应感应延时[0013.02]
T1211 BOOL  ; RK_12 轮廓检测NG料槽#2有料感应感应延时[0013.03]
T1212 BOOL  ; RK_12 轮廓检测NG料槽#2料满感应感应延时[0013.04]
T1213 BOOL  ; RK_12 OK出料拉带放料位有料感应#1感应延时[0013.05]
T1214 BOOL  ; RK_12 OK出料拉带放料位有料感应#2感应延时[0013.06]
T1215 BOOL  ; RK_12 OK出料拉带出料位有料感应感应延时[0013.07]
T1216 BOOL  ; 0感应延时[0013.08]
T1217 BOOL  ; 0感应延时[0013.09]
T1218 BOOL  ; 0感应延时[0013.10]
T1219 BOOL  ; 0感应延时[0013.11]
T1220 BOOL  ; 0感应延时[0013.12]
T1221 BOOL  ; 0感应延时[0013.13]
T1222 BOOL  ; 0感应延时[0013.14]
T1223 BOOL  ; 0感应延时[0013.15]
T1224 BOOL  ; RK_06 铝壳上料升降气缸下降位感应延时[0014.00]
T1225 BOOL  ; RK_06 铝壳上料升降气缸上升位感应延时[0014.01]
T1226 BOOL  ; RK_06 电池下料升降气缸下降位感应延时[0014.02]
T1227 BOOL  ; RK_06 电池下料升降气缸上升位感应延时[0014.03]
T1228 BOOL  ; RK_06 铝壳上料夹爪气缸夹紧位感应延时[0014.04]
T1229 BOOL  ; RK_06 铝壳上料夹爪气缸张开位感应延时[0014.05]
T1230 BOOL  ; RK_06 电池下料夹爪气缸夹紧位感应延时[0014.06]
T1231 BOOL  ; RK_06 电池下料夹爪气缸张开位感应延时[0014.07]
T1232 BOOL  ; RK_07 #1铝壳上料车定位升降气缸上升位感应延时[0014.08]
T1233 BOOL  ; RK_07 #1铝壳上料车定位升降气缸下降位感应延时[0014.09]
T1234 BOOL  ; RK_07 #2铝壳上料车定位升降气缸上升位感应延时[0014.10]
T1235 BOOL  ; RK_07 #2铝壳上料车定位升降气缸下降位感应延时[0014.11]
T1236 BOOL  ; RK_07 #3托盘下料车定位升降气缸上升位感应延时[0014.12]
T1237 BOOL  ; RK_07 #3托盘下料车定位升降气缸下降位感应延时[0014.13]
T1238 BOOL  ; RK_07 铝壳进料机械手升降气缸下降位感应延时[0014.14]
T1239 BOOL  ; RK_07 铝壳进料机械手升降气缸上升位感应延时[0014.15]
T1240 BOOL  ; RK_08 铝壳除尘旋转伸缩气缸原位感应延时[0015.00]
T1241 BOOL  ; RK_08 铝壳除尘旋转伸缩气缸到位感应延时[0015.01]
T1242 BOOL  ; RK_08 铝壳除尘伸缩气缸伸出位感应延时[0015.02]
T1243 BOOL  ; RK_08 铝壳除尘伸缩气缸缩回位感应延时[0015.03]
T1244 BOOL  ; RK_08 铝壳除尘夹爪气缸夹紧位感应延时[0015.04]
T1245 BOOL  ; RK_08 铝壳除尘夹爪气缸张开位感应延时[0015.05]
T1246 BOOL  ; RK_09 #1Hipot测试旋转伸缩气缸到位感应延时[0015.06]
T1247 BOOL  ; RK_09 #1Hipot测试旋转伸缩气缸原位感应延时[0015.07]
T1248 BOOL  ; RK_09 #1Hipot测试平台伸缩气缸缩回位感应延时[0015.08]
T1249 BOOL  ; RK_09 #1Hipot测试平台伸缩气缸伸出位感应延时[0015.09]
T1250 BOOL  ; RK_09 #1Hipot测试伸缩气缸伸出位感应延时[0015.10]
T1251 BOOL  ; RK_09 #1Hipot测试伸缩气缸缩回位感应延时[0015.11]
T1252 BOOL  ; RK_09 #2Hipot测试旋转伸缩气缸到位感应延时[0015.12]
T1253 BOOL  ; RK_09 #2Hipot测试旋转伸缩气缸原位感应延时[0015.13]
T1254 BOOL  ; RK_09 #2Hipot测试平台伸缩气缸缩回位感应延时[0015.14]
T1255 BOOL  ; RK_09 #2Hipot测试平台伸缩气缸伸出位感应延时[0015.15]
T1256 BOOL  ; RK_09 #2Hipot测试伸缩气缸伸出位感应延时[0016.00]
T1257 BOOL  ; RK_09 #2Hipot测试伸缩气缸缩回位感应延时[0016.01]
T1258 BOOL  ; RK_10 电池除尘上料机械手升降气缸下降位感应延时[0016.02]
T1259 BOOL  ; RK_10 电池除尘上料机械手升降气缸上升位感应延时[0016.03]
T1260 BOOL  ; RK_10 电池除尘上料机械手夹爪气缸夹紧位感应延时[0016.04]
T1261 BOOL  ; RK_10 电池除尘上料机械手夹爪气缸张开位感应延时[0016.05]
T1262 BOOL  ; RK_06 U8_X 电池上下料X轴报警信号感应延时[0016.06]
T1263 BOOL  ; RK_06 U8_X 电池上下料X轴准备好了信号感应延时[0016.07]
T1264 BOOL  ; RK_07 U8_Y 铝壳进料X轴报警信号感应延时[0016.08]
T1265 BOOL  ; RK_07 U8_Y 铝壳进料X轴准备好了信号感应延时[0016.09]
T1266 BOOL  ; RK_07 U8_Z 铝壳上料移载Y轴报警信号感应延时[0016.10]
T1267 BOOL  ; RK_07 U8_Z 铝壳上料移载Y轴准备好了信号感应延时[0016.11]
T1268 BOOL  ; RK_10 U8_U 电池除尘上料X轴报警信号感应延时[0016.12]
T1269 BOOL  ; RK_10 U8_U 电池除尘上料X轴准备好了信号感应延时[0016.13]
T1270 BOOL  ; RK_09 Hipot测试完成信号感应延时[0016.14]
T1271 BOOL  ; RK_07 #1铝壳上料启动按钮感应延时[0016.15]
T1272 BOOL  ; RK_07 #2铝壳上料启动按钮感应延时[0017.00]
T1273 BOOL  ; RK_07 #3托盘下料启动按钮感应延时[0017.01]
T1274 BOOL  ; RK_07 铝壳上料移载吸盘真空感应延时[0017.02]
T1275 BOOL  ; RK_07 铝壳进料吸盘真空感应延时[0017.03]
T1276 BOOL  ; RK_07 #1铝壳上料托盘到位感应感应延时[0017.04]
T1277 BOOL  ; RK_07 #1铝壳上料位物料车到位感应感应延时[0017.05]
T1278 BOOL  ; RK_07 #1铝壳上料初始位（#1）感应延时[0017.06]
T1279 BOOL  ; RK_07 #1铝壳上料一个托盘位（#2）感应延时[0017.07]
T1280 BOOL  ; RK_07 #1铝壳上料高限位（#3）感应延时[0017.08]
T1281 BOOL  ; RK_07 #2铝壳上料托盘到位感应感应延时[0017.09]
T1282 BOOL  ; RK_07 #2铝壳上料位物料车到位感应感应延时[0017.10]
T1283 BOOL  ; RK_07 #2铝壳上料初始位（#1）感应延时[0017.11]
T1284 BOOL  ; RK_07 #2铝壳上料一个托盘位（#2）感应延时[0017.12]
T1285 BOOL  ; RK_07 #2铝壳上料高限位（#3）感应延时[0017.13]
T1286 BOOL  ; RK_07 #3托盘下料上升到位感应感应延时[0017.14]
T1287 BOOL  ; RK_07 #3托盘下料位物料车到位感应感应延时[0017.15]
T1288 BOOL  ; RK_07 #3托盘下料初始位（#1）感应延时[0018.00]
T1289 BOOL  ; RK_07 #3托盘下料满托盘位（#2）感应延时[0018.01]
T1290 BOOL  ; RK_07 #3托盘下料高限位（#3）感应延时[0018.02]
T1291 BOOL  ; RK_07 铝壳上料移载托盘到位感应感应延时[0018.03]
T1292 BOOL  ; RK_08 铝壳除尘有料感应感应延时[0018.04]
T1293 BOOL  ; RK_09 #1Hipot测试有料感应感应延时[0018.05]
T1294 BOOL  ; RK_09 #2Hipot测试有料感应感应延时[0018.06]
T1295 BOOL  ; RK_10 Hipot检测NG拉带有料感应#1感应延时[0018.07]
T1296 BOOL  ; RK_10 Hipot检测NG拉带有料感应#2感应延时[0018.08]
T1297 BOOL  ; RK_10 Hipot检测NG拉带料满感应感应延时[0018.09]
T1298 BOOL  ; RK_06 铝壳上料夹爪柔性报警感应延时[0018.10]
T1299 BOOL  ; RK_06 电池下料夹爪柔性报警感应延时[0018.11]
T1300 BOOL  ; RK_07 铝壳进料机械手柔性报警感应延时[0018.12]
T1301 BOOL  ; RK_10 电池除尘上料机械手夹爪柔性报警感应延时[0018.13]
T1302 BOOL  ; 手/自动选择（公共）感应延时[0018.14]
T1303 BOOL  ; 启动按钮_绿（公共）感应延时[0018.15]
T1304 BOOL  ; 停止按钮_红（公共）感应延时[0019.00]
T1305 BOOL  ; 复位按钮_黄（公共）感应延时[0019.01]
T1306 BOOL  ; 机台进气压力（正压）（公共）感应延时[0019.02]
T1307 BOOL  ; 机台进气压力（负压）（公共）感应延时[0019.03]
T1308 BOOL  ; 主屏急停（公共）感应延时[0019.04]
T1309 BOOL  ; 铝壳上料端急停（公共）感应延时[0019.05]
T1310 BOOL  ; HipotNG端急停（公共）感应延时[0019.06]
T1311 BOOL  ; B机架#1门磁（公共）感应延时[0019.07]
T1312 BOOL  ; B机架#2门磁（公共）感应延时[0019.08]
